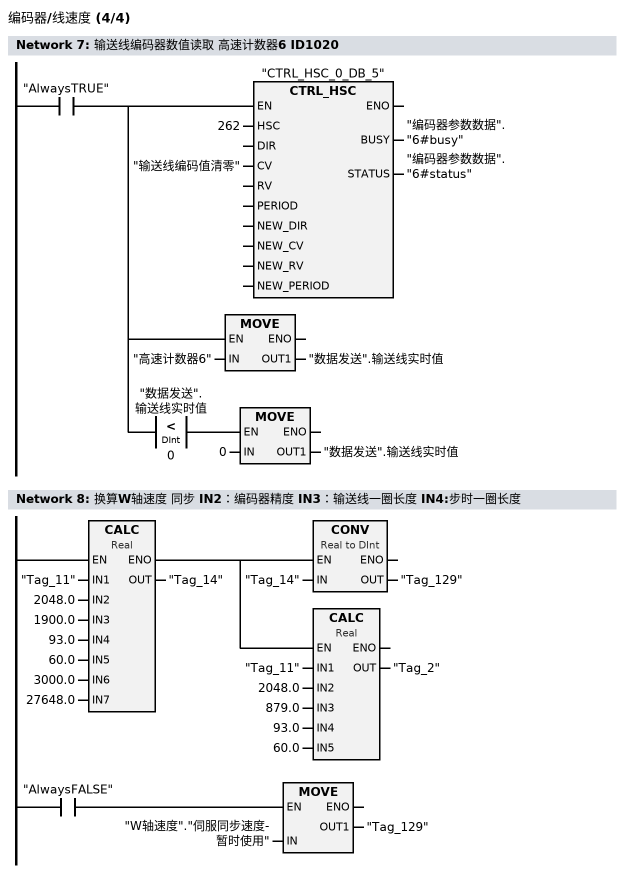
   #_w1 := "AlwaysTRUE";
   IF #_w1 THEN
       "CTRL_HSC_0_DB_5"(HSC := 262, CV := "输送线编码值清零", BUSY => "编码器参数数据"."6#busy", STATUS => "编码器参数数据"."6#status");   // CTRL_HSC
       "数据发送".输送线实时值 := "高速计数器6";
   END_IF;
   IF #_w1 AND ("数据发送".输送线实时值 < 0) THEN "数据发送".输送线实时值 := 0; END_IF;
END_REGION

REGION Network 8: 换算W轴速度 同步 IN2：编码器精度 IN3：输送线一圈长度 IN4:步时一圈长度
   CALC(in1 := "Tag_11",
        in2 := 2048.0,
        in3 := 1900.0,
        in4 := 93.0,
        in5 := 60.0,
        in6 := 3000.0,
        in7 := 27648.0,
        out => "Tag_14");
   "Tag_129" := REAL_TO_DINT("Tag_14");
   CALC(in1 := "Tag_11", in2 := 2048.0, in3 := 879.0, in4 := 93.0, in5 := 60.0, out => "Tag_2");
   IF "AlwaysFALSE" THEN "Tag_129" := "W轴速度"."伺服同步速度-暂时使用"; END_IF;
END_REGION
END_FUNCTION

FUNCTION "2#手" : Void   // FC13, LAD
{ S7_Optimized_Access := 'TRUE' }
VERSION : 0.1
   VAR_TEMP   // added for the SCL form of the ladder/FBD networks
      _w1 : Bool;
   END_VAR
BEGIN

REGION Network 1: 2#机械手库位动作流程
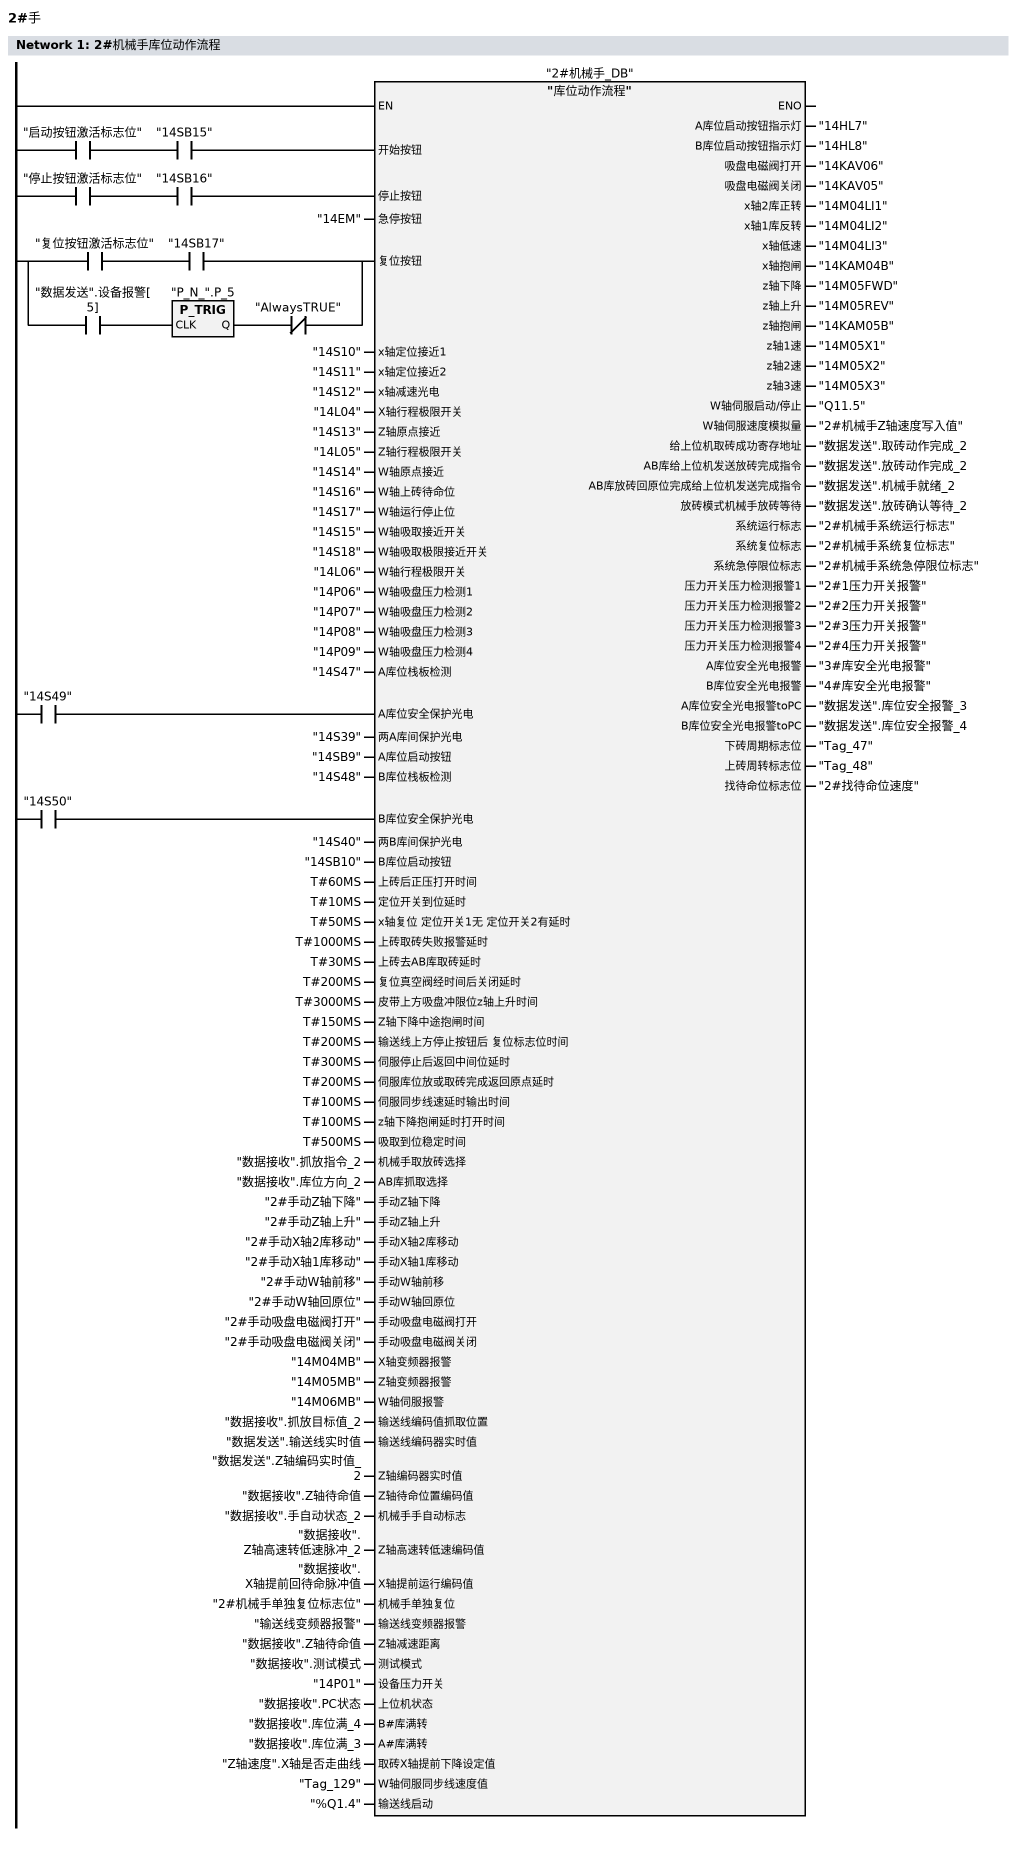
   RUNG wire#powerrail
      "2#机械手_DB"(开始按钮 := wire#w1, 停止按钮 := wire#w2, 复位按钮 := wire#w3, A库位安全保护光电 := wire#w4, B库位安全保护光电 := wire#w5, 急停按钮 := "14EM", x轴定位接近1 := "14S10", x轴定位接近2 := "14S11", x轴减速光电 := "14S12", X轴行程极限开关 := "14L04", Z轴原点接近 := "14S13", Z轴行程极限开关 := "14L05", W轴原点接近 := "14S14", W轴上砖待命位 := "14S16", W轴运行停止位 := "14S17", W轴吸取接近开关 := "14S15", W轴吸取极限接近开关 := "14S18", W轴行程极限开关 := "14L06", W轴吸盘压力检测1 := "14P06", W轴吸盘压力检测2 := "14P07", W轴吸盘压力检测3 := "14P08", W轴吸盘压力检测4 := "14P09", A库位栈板检测 := "14S47", 两A库间保护光电 := "14S39", A库位启动按钮 := "14SB9", B库位栈板检测 := "14S48", 两B库间保护光电 := "14S40", B库位启动按钮 := "14SB10", 上砖后正压打开时间 := T#60MS, 定位开关到位延时 := T#10MS, "x轴复位 定位开关1无 定位开关2有延时" := T#50MS, 上砖取砖失败报警延时 := T#1000MS, 上砖去AB库取砖延时 := T#30MS, 复位真空阀经时间后关闭延时 := T#200MS, 皮带上方吸盘冲限位z轴上升时间 := T#3000MS, Z轴下降中途抱闸时间 := T#150MS, "输送线上方停止按钮后 复位标志位时间" := T#200MS, 伺服停止后返回中间位延时 := T#300MS, 伺服库位放或取砖完成返回原点延时 := T#200MS, 伺服同步线速延时输出时间 := T#100MS, z轴下降抱闸延时打开时间 := T#100MS, 吸取到位稳定时间 := T#500MS, 机械手取放砖选择 := "数据接收".抓放指令_2, AB库抓取选择 := "数据接收".库位方向_2, 手动Z轴下降 := "2#手动Z轴下降", 手动Z轴上升 := "2#手动Z轴上升", 手动X轴2库移动 := "2#手动X轴2库移动", 手动X轴1库移动 := "2#手动X轴1库移动", 手动W轴前移 := "2#手动W轴前移", 手动W轴回原位 := "2#手动W轴回原位", 手动吸盘电磁阀打开 := "2#手动吸盘电磁阀打开", 手动吸盘电磁阀关闭 := "2#手动吸盘电磁阀关闭", X轴变频器报警 := "14M04MB", Z轴变频器报警 := "14M05MB", W轴伺服报警 := "14M06MB", 输送线编码值抓取位置 := "数据接收".抓放目标值_2, 输送线编码器实时值 := "数据发送".输送线实时值, Z轴编码器实时值 := "数据发送".Z轴编码实时值_2, Z轴待命位置编码值 := "数据接收".Z轴待命值, 机械手手自动标志 := "数据接收".手自动状态_2, Z轴高速转低速编码值 := "数据接收".Z轴高速转低速脉冲_2, X轴提前运行编码值 := "数据接收".X轴提前回待命脉冲值, 机械手单独复位 := "2#机械手单独复位标志位", 输送线变频器报警 := "输送线变频器报警", Z轴减速距离 := "数据接收".Z轴待命值, 测试模式 := "数据接收".测试模式, 设备压力开关 := "14P01", 上位机状态 := "数据接收".PC状态, "B#库满转" := "数据接收".库位满_4, "A#库满转" := "数据接收".库位满_3, 取砖X轴提前下降设定值 := "Z轴速度".X轴是否走曲线, W轴伺服同步线速度值 := "Tag_129", 输送线启动 := "%Q1.4", A库位启动按钮指示灯 => "14HL7", B库位启动按钮指示灯 => "14HL8", 吸盘电磁阀打开 => "14KAV06", 吸盘电磁阀关闭 => "14KAV05", x轴2库正转 => "14M04LI1", x轴1库反转 => "14M04LI2", x轴低速 => "14M04LI3", x轴抱闸 => "14KAM04B", z轴下降 => "14M05FWD", z轴上升 => "14M05REV", z轴抱闸 => "14KAM05B", z轴1速 => "14M05X1", z轴2速 => "14M05X2", z轴3速 => "14M05X3", "W轴伺服启动/停止" => "Q11.5", W轴伺服速度模拟量 => "2#机械手Z轴速度写入值", 给上位机取砖成功寄存地址 => "数据发送".取砖动作完成_2, AB库给上位机发送放砖完成指令 => "数据发送".放砖动作完成_2, AB库放砖回原位完成给上位机发送完成指令 => "数据发送".机械手就绪_2, 放砖模式机械手放砖等待 => "数据发送".放砖确认等待_2, 系统运行标志 => "2#机械手系统运行标志", 系统复位标志 => "2#机械手系统复位标志", 系统急停限位标志 => "2#机械手系统急停限位标志", 压力开关压力检测报警1 => "2#1压力开关报警", 压力开关压力检测报警2 => "2#2压力开关报警", 压力开关压力检测报警3 => "2#3压力开关报警", 压力开关压力检测报警4 => "2#4压力开关报警", A库位安全光电报警 => "3#库安全光电报警", B库位安全光电报警 => "4#库安全光电报警", A库位安全光电报警toPC => "数据发送".库位安全报警_3, B库位安全光电报警toPC => "数据发送".库位安全报警_4, 下砖周期标志位 => "Tag_47", 上砖周转标志位 => "Tag_48", 找待命位标志位 => "2#找待命位速度")
   END_RUNG
   RUNG wire#powerrail
      Contact( "启动按钮激活标志位" )
      Contact( "14SB15" )
   END_RUNG wire#w1
   RUNG wire#powerrail
      Contact( "停止按钮激活标志位" )
      Contact( "14SB16" )
   END_RUNG wire#w2
   RUNG wire#powerrail
      Contact( "复位按钮激活标志位" )
      Contact( "14SB17" )
   END_RUNG wire#w3
   RUNG wire#powerrail
      Contact( "数据发送".设备报警[5] )
      P_Trig( "P_N_".P_5 )
      I_Contact( "AlwaysTRUE" )
   END_RUNG wire#w3
   RUNG wire#powerrail
      Contact( "14S49" )
   END_RUNG wire#w4
   RUNG wire#powerrail
      Contact( "14S50" )
   END_RUNG wire#w5
   // the same network as SCL:
   #_w1 := "数据发送".设备报警[5] AND NOT "P_N_".P_5;   // rising edge
   "P_N_".P_5 := "数据发送".设备报警[5];
   "2#机械手_DB"(开始按钮 := "启动按钮激活标志位" AND "14SB15",   // "库位动作流程"
              停止按钮 := "停止按钮激活标志位" AND "14SB16",
              急停按钮 := "14EM",
              复位按钮 := ("复位按钮激活标志位" AND "14SB17") OR (#_w1 AND NOT "AlwaysTRUE"),
              x轴定位接近1 := "14S10",
              x轴定位接近2 := "14S11",
              x轴减速光电 := "14S12",
              X轴行程极限开关 := "14L04",
              Z轴原点接近 := "14S13",
              Z轴行程极限开关 := "14L05",
              W轴原点接近 := "14S14",
              W轴上砖待命位 := "14S16",
              W轴运行停止位 := "14S17",
              W轴吸取接近开关 := "14S15",
              W轴吸取极限接近开关 := "14S18",
              W轴行程极限开关 := "14L06",
              W轴吸盘压力检测1 := "14P06",
              W轴吸盘压力检测2 := "14P07",
              W轴吸盘压力检测3 := "14P08",
              W轴吸盘压力检测4 := "14P09",
              A库位栈板检测 := "14S47",
              A库位安全保护光电 := "14S49",
              两A库间保护光电 := "14S39",
              A库位启动按钮 := "14SB9",
              B库位栈板检测 := "14S48",
              B库位安全保护光电 := "14S50",
              两B库间保护光电 := "14S40",
              B库位启动按钮 := "14SB10",
              上砖后正压打开时间 := T#60MS,
              定位开关到位延时 := T#10MS,
              "x轴复位 定位开关1无 定位开关2有延时" := T#50MS,
              上砖取砖失败报警延时 := T#1000MS,
              上砖去AB库取砖延时 := T#30MS,
              复位真空阀经时间后关闭延时 := T#200MS,
              皮带上方吸盘冲限位z轴上升时间 := T#3000MS,
              Z轴下降中途抱闸时间 := T#150MS,
              "输送线上方停止按钮后 复位标志位时间" := T#200MS,
              伺服停止后返回中间位延时 := T#300MS,
              伺服库位放或取砖完成返回原点延时 := T#200MS,
              伺服同步线速延时输出时间 := T#100MS,
              z轴下降抱闸延时打开时间 := T#100MS,
              吸取到位稳定时间 := T#500MS,
              机械手取放砖选择 := "数据接收".抓放指令_2,
              AB库抓取选择 := "数据接收".库位方向_2,
              手动Z轴下降 := "2#手动Z轴下降",
              手动Z轴上升 := "2#手动Z轴上升",
              手动X轴2库移动 := "2#手动X轴2库移动",
              手动X轴1库移动 := "2#手动X轴1库移动",
              手动W轴前移 := "2#手动W轴前移",
              手动W轴回原位 := "2#手动W轴回原位",
              手动吸盘电磁阀打开 := "2#手动吸盘电磁阀打开",
              手动吸盘电磁阀关闭 := "2#手动吸盘电磁阀关闭",
              X轴变频器报警 := "14M04MB",
              Z轴变频器报警 := "14M05MB",
              W轴伺服报警 := "14M06MB",
              输送线编码值抓取位置 := "数据接收".抓放目标值_2,
              输送线编码器实时值 := "数据发送".输送线实时值,
              Z轴编码器实时值 := "数据发送".Z轴编码实时值_2,
              Z轴待命位置编码值 := "数据接收".Z轴待命值,
              机械手手自动标志 := "数据接收".手自动状态_2,
              Z轴高速转低速编码值 := "数据接收".Z轴高速转低速脉冲_2,
              X轴提前运行编码值 := "数据接收".X轴提前回待命脉冲值,
              机械手单独复位 := "2#机械手单独复位标志位",
              输送线变频器报警 := "输送线变频器报警",
              Z轴减速距离 := "数据接收".Z轴待命值,
              测试模式 := "数据接收".测试模式,
              设备压力开关 := "14P01",
              上位机状态 := "数据接收".PC状态,
              "B#库满转" := "数据接收".库位满_4,
              "A#库满转" := "数据接收".库位满_3,
              取砖X轴提前下降设定值 := "Z轴速度".X轴是否走曲线,
              W轴伺服同步线速度值 := "Tag_129",
              输送线启动 := "%Q1.4",
              A库位启动按钮指示灯 => "14HL7",
              B库位启动按钮指示灯 => "14HL8",
              吸盘电磁阀打开 => "14KAV06",
              吸盘电磁阀关闭 => "14KAV05",
              x轴2库正转 => "14M04LI1",
              x轴1库反转 => "14M04LI2",
              x轴低速 => "14M04LI3",
              x轴抱闸 => "14KAM04B",
              z轴下降 => "14M05FWD",
              z轴上升 => "14M05REV",
              z轴抱闸 => "14KAM05B",
              z轴1速 => "14M05X1",
              z轴2速 => "14M05X2",
              z轴3速 => "14M05X3",
              "W轴伺服启动/停止" => "Q11.5",
              W轴伺服速度模拟量 => "2#机械手Z轴速度写入值",
              给上位机取砖成功寄存地址 => "数据发送".取砖动作完成_2,
              AB库给上位机发送放砖完成指令 => "数据发送".放砖动作完成_2,
              AB库放砖回原位完成给上位机发送完成指令 => "数据发送".机械手就绪_2,
              放砖模式机械手放砖等待 => "数据发送".放砖确认等待_2,
              系统运行标志 => "2#机械手系统运行标志",
              系统复位标志 => "2#机械手系统复位标志",
              系统急停限位标志 => "2#机械手系统急停限位标志",
              压力开关压力检测报警1 => "2#1压力开关报警",
              压力开关压力检测报警2 => "2#2压力开关报警",
              压力开关压力检测报警3 => "2#3压力开关报警",
              压力开关压力检测报警4 => "2#4压力开关报警",
              A库位安全光电报警 => "3#库安全光电报警",
              B库位安全光电报警 => "4#库安全光电报警",
              A库位安全光电报警toPC => "数据发送".库位安全报警_3,
              B库位安全光电报警toPC => "数据发送".库位安全报警_4,
              下砖周期标志位 => "Tag_47",
              上砖周转标志位 => "Tag_48",
              找待命位标志位 => "2#找待命位速度");
END_REGION
END_FUNCTION

FUNCTION "3#手" : Void   // FC14, LAD
{ S7_Optimized_Access := 'TRUE' }
VERSION : 0.1
   VAR_TEMP   // added for the SCL form of the ladder/FBD networks
      _w1 : Bool;
   END_VAR
BEGIN

REGION Network 1: 3#机械手库位动作流程
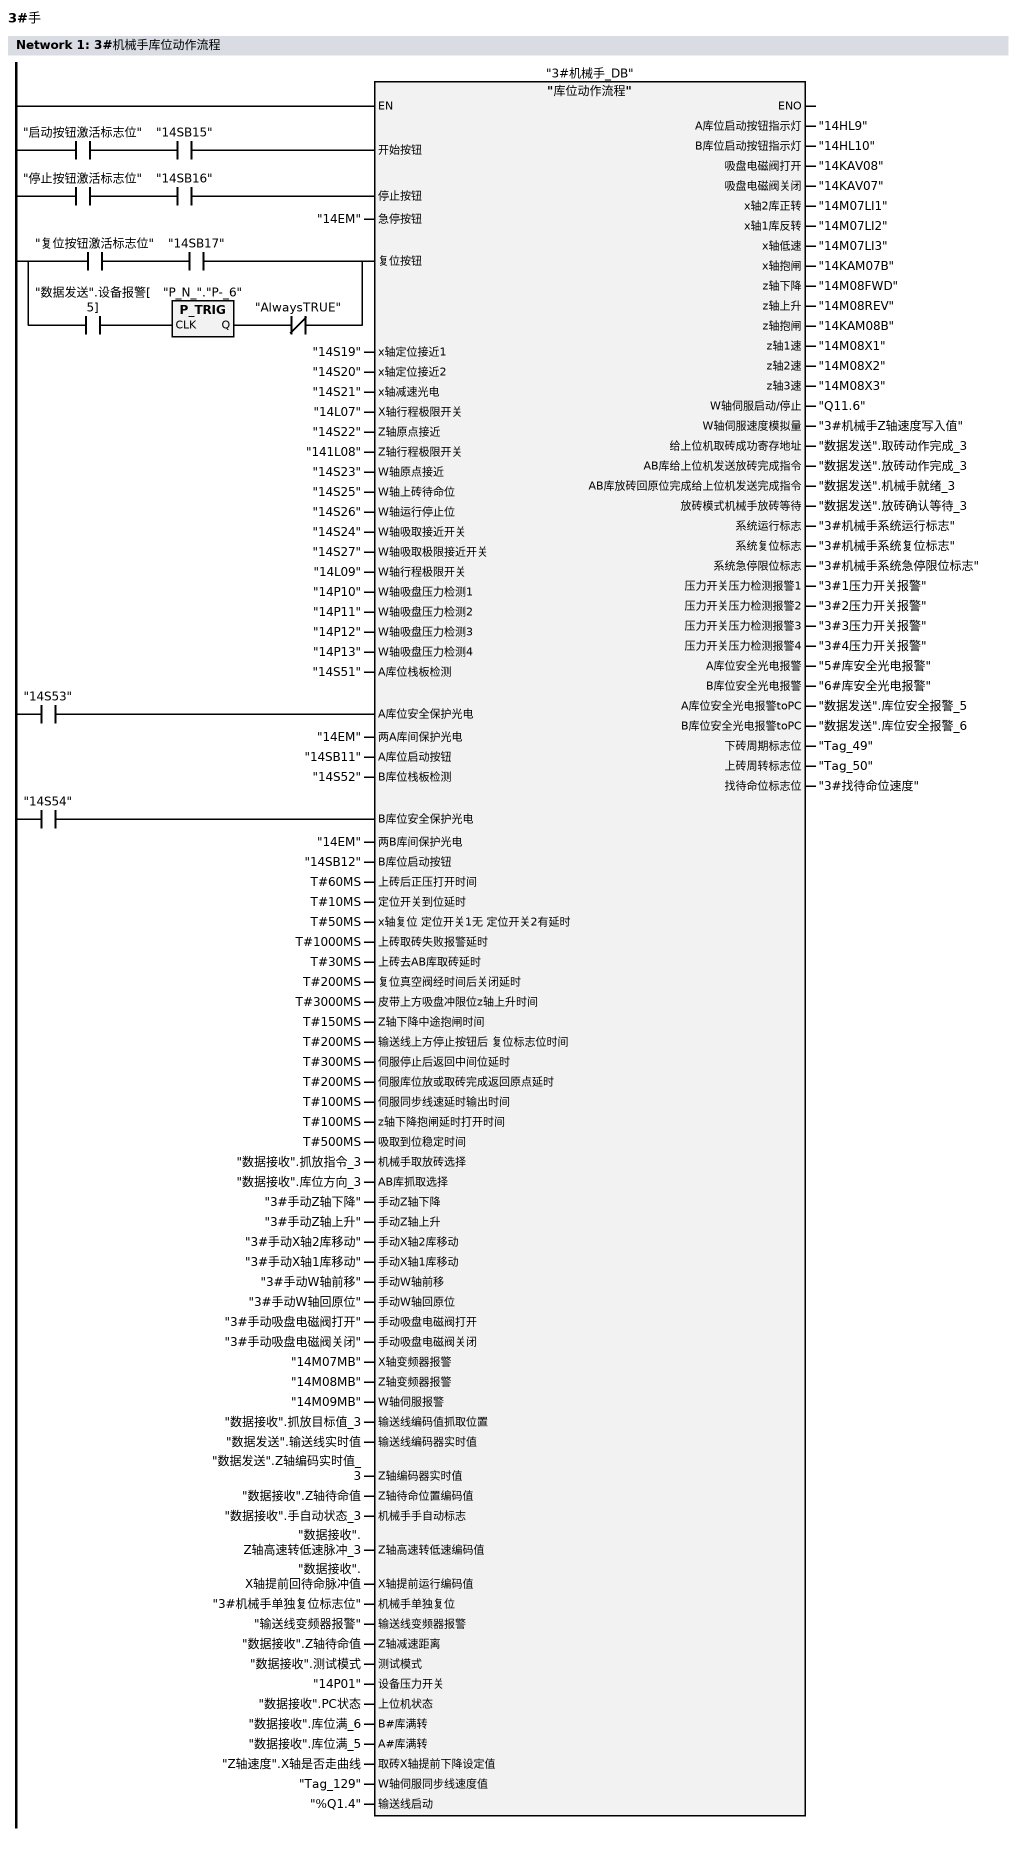
   RUNG wire#powerrail
      "3#机械手_DB"(开始按钮 := wire#w1, 停止按钮 := wire#w2, 复位按钮 := wire#w3, A库位安全保护光电 := wire#w4, B库位安全保护光电 := wire#w5, 急停按钮 := "14EM", x轴定位接近1 := "14S19", x轴定位接近2 := "14S20", x轴减速光电 := "14S21", X轴行程极限开关 := "14L07", Z轴原点接近 := "14S22", Z轴行程极限开关 := "141L08", W轴原点接近 := "14S23", W轴上砖待命位 := "14S25", W轴运行停止位 := "14S26", W轴吸取接近开关 := "14S24", W轴吸取极限接近开关 := "14S27", W轴行程极限开关 := "14L09", W轴吸盘压力检测1 := "14P10", W轴吸盘压力检测2 := "14P11", W轴吸盘压力检测3 := "14P12", W轴吸盘压力检测4 := "14P13", A库位栈板检测 := "14S51", 两A库间保护光电 := "14EM", A库位启动按钮 := "14SB11", B库位栈板检测 := "14S52", 两B库间保护光电 := "14EM", B库位启动按钮 := "14SB12", 上砖后正压打开时间 := T#60MS, 定位开关到位延时 := T#10MS, "x轴复位 定位开关1无 定位开关2有延时" := T#50MS, 上砖取砖失败报警延时 := T#1000MS, 上砖去AB库取砖延时 := T#30MS, 复位真空阀经时间后关闭延时 := T#200MS, 皮带上方吸盘冲限位z轴上升时间 := T#3000MS, Z轴下降中途抱闸时间 := T#150MS, "输送线上方停止按钮后 复位标志位时间" := T#200MS, 伺服停止后返回中间位延时 := T#300MS, 伺服库位放或取砖完成返回原点延时 := T#200MS, 伺服同步线速延时输出时间 := T#100MS, z轴下降抱闸延时打开时间 := T#100MS, 吸取到位稳定时间 := T#500MS, 机械手取放砖选择 := "数据接收".抓放指令_3, AB库抓取选择 := "数据接收".库位方向_3, 手动Z轴下降 := "3#手动Z轴下降", 手动Z轴上升 := "3#手动Z轴上升", 手动X轴2库移动 := "3#手动X轴2库移动", 手动X轴1库移动 := "3#手动X轴1库移动", 手动W轴前移 := "3#手动W轴前移", 手动W轴回原位 := "3#手动W轴回原位", 手动吸盘电磁阀打开 := "3#手动吸盘电磁阀打开", 手动吸盘电磁阀关闭 := "3#手动吸盘电磁阀关闭", X轴变频器报警 := "14M07MB", Z轴变频器报警 := "14M08MB", W轴伺服报警 := "14M09MB", 输送线编码值抓取位置 := "数据接收".抓放目标值_3, 输送线编码器实时值 := "数据发送".输送线实时值, Z轴编码器实时值 := "数据发送".Z轴编码实时值_3, Z轴待命位置编码值 := "数据接收".Z轴待命值, 机械手手自动标志 := "数据接收".手自动状态_3, Z轴高速转低速编码值 := "数据接收".Z轴高速转低速脉冲_3, X轴提前运行编码值 := "数据接收".X轴提前回待命脉冲值, 机械手单独复位 := "3#机械手单独复位标志位", 输送线变频器报警 := "输送线变频器报警", Z轴减速距离 := "数据接收".Z轴待命值, 测试模式 := "数据接收".测试模式, 设备压力开关 := "14P01", 上位机状态 := "数据接收".PC状态, "B#库满转" := "数据接收".库位满_6, "A#库满转" := "数据接收".库位满_5, 取砖X轴提前下降设定值 := "Z轴速度".X轴是否走曲线, W轴伺服同步线速度值 := "Tag_129", 输送线启动 := "%Q1.4", A库位启动按钮指示灯 => "14HL9", B库位启动按钮指示灯 => "14HL10", 吸盘电磁阀打开 => "14KAV08", 吸盘电磁阀关闭 => "14KAV07", x轴2库正转 => "14M07LI1", x轴1库反转 => "14M07LI2", x轴低速 => "14M07LI3", x轴抱闸 => "14KAM07B", z轴下降 => "14M08FWD", z轴上升 => "14M08REV", z轴抱闸 => "14KAM08B", z轴1速 => "14M08X1", z轴2速 => "14M08X2", z轴3速 => "14M08X3", "W轴伺服启动/停止" => "Q11.6", W轴伺服速度模拟量 => "3#机械手Z轴速度写入值", 给上位机取砖成功寄存地址 => "数据发送".取砖动作完成_3, AB库给上位机发送放砖完成指令 => "数据发送".放砖动作完成_3, AB库放砖回原位完成给上位机发送完成指令 => "数据发送".机械手就绪_3, 放砖模式机械手放砖等待 => "数据发送".放砖确认等待_3, 系统运行标志 => "3#机械手系统运行标志", 系统复位标志 => "3#机械手系统复位标志", 系统急停限位标志 => "3#机械手系统急停限位标志", 压力开关压力检测报警1 => "3#1压力开关报警", 压力开关压力检测报警2 => "3#2压力开关报警", 压力开关压力检测报警3 => "3#3压力开关报警", 压力开关压力检测报警4 => "3#4压力开关报警", A库位安全光电报警 => "5#库安全光电报警", B库位安全光电报警 => "6#库安全光电报警", A库位安全光电报警toPC => "数据发送".库位安全报警_5, B库位安全光电报警toPC => "数据发送".库位安全报警_6, 下砖周期标志位 => "Tag_49", 上砖周转标志位 => "Tag_50", 找待命位标志位 => "3#找待命位速度")
   END_RUNG
   RUNG wire#powerrail
      Contact( "启动按钮激活标志位" )
      Contact( "14SB15" )
   END_RUNG wire#w1
   RUNG wire#powerrail
      Contact( "停止按钮激活标志位" )
      Contact( "14SB16" )
   END_RUNG wire#w2
   RUNG wire#powerrail
      Contact( "复位按钮激活标志位" )
      Contact( "14SB17" )
   END_RUNG wire#w3
   RUNG wire#powerrail
      Contact( "数据发送".设备报警[5] )
      P_Trig( "P_N_"."P-_6" )
      I_Contact( "AlwaysTRUE" )
   END_RUNG wire#w3
   RUNG wire#powerrail
      Contact( "14S53" )
   END_RUNG wire#w4
   RUNG wire#powerrail
      Contact( "14S54" )
   END_RUNG wire#w5
   // the same network as SCL:
   #_w1 := "数据发送".设备报警[5] AND NOT "P_N_"."P-_6";   // rising edge
   "P_N_"."P-_6" := "数据发送".设备报警[5];
   "3#机械手_DB"(开始按钮 := "启动按钮激活标志位" AND "14SB15",   // "库位动作流程"
              停止按钮 := "停止按钮激活标志位" AND "14SB16",
              急停按钮 := "14EM",
              复位按钮 := ("复位按钮激活标志位" AND "14SB17") OR (#_w1 AND NOT "AlwaysTRUE"),
              x轴定位接近1 := "14S19",
              x轴定位接近2 := "14S20",
              x轴减速光电 := "14S21",
              X轴行程极限开关 := "14L07",
              Z轴原点接近 := "14S22",
              Z轴行程极限开关 := "141L08",
              W轴原点接近 := "14S23",
              W轴上砖待命位 := "14S25",
              W轴运行停止位 := "14S26",
              W轴吸取接近开关 := "14S24",
              W轴吸取极限接近开关 := "14S27",
              W轴行程极限开关 := "14L09",
              W轴吸盘压力检测1 := "14P10",
              W轴吸盘压力检测2 := "14P11",
              W轴吸盘压力检测3 := "14P12",
              W轴吸盘压力检测4 := "14P13",
              A库位栈板检测 := "14S51",
              A库位安全保护光电 := "14S53",
              两A库间保护光电 := "14EM",
              A库位启动按钮 := "14SB11",
              B库位栈板检测 := "14S52",
              B库位安全保护光电 := "14S54",
              两B库间保护光电 := "14EM",
              B库位启动按钮 := "14SB12",
              上砖后正压打开时间 := T#60MS,
              定位开关到位延时 := T#10MS,
              "x轴复位 定位开关1无 定位开关2有延时" := T#50MS,
              上砖取砖失败报警延时 := T#1000MS,
              上砖去AB库取砖延时 := T#30MS,
              复位真空阀经时间后关闭延时 := T#200MS,
              皮带上方吸盘冲限位z轴上升时间 := T#3000MS,
              Z轴下降中途抱闸时间 := T#150MS,
              "输送线上方停止按钮后 复位标志位时间" := T#200MS,
              伺服停止后返回中间位延时 := T#300MS,
              伺服库位放或取砖完成返回原点延时 := T#200MS,
              伺服同步线速延时输出时间 := T#100MS,
              z轴下降抱闸延时打开时间 := T#100MS,
              吸取到位稳定时间 := T#500MS,
              机械手取放砖选择 := "数据接收".抓放指令_3,
              AB库抓取选择 := "数据接收".库位方向_3,
              手动Z轴下降 := "3#手动Z轴下降",
              手动Z轴上升 := "3#手动Z轴上升",
              手动X轴2库移动 := "3#手动X轴2库移动",
              手动X轴1库移动 := "3#手动X轴1库移动",
              手动W轴前移 := "3#手动W轴前移",
              手动W轴回原位 := "3#手动W轴回原位",
              手动吸盘电磁阀打开 := "3#手动吸盘电磁阀打开",
              手动吸盘电磁阀关闭 := "3#手动吸盘电磁阀关闭",
              X轴变频器报警 := "14M07MB",
              Z轴变频器报警 := "14M08MB",
              W轴伺服报警 := "14M09MB",
              输送线编码值抓取位置 := "数据接收".抓放目标值_3,
              输送线编码器实时值 := "数据发送".输送线实时值,
              Z轴编码器实时值 := "数据发送".Z轴编码实时值_3,
              Z轴待命位置编码值 := "数据接收".Z轴待命值,
              机械手手自动标志 := "数据接收".手自动状态_3,
              Z轴高速转低速编码值 := "数据接收".Z轴高速转低速脉冲_3,
              X轴提前运行编码值 := "数据接收".X轴提前回待命脉冲值,
              机械手单独复位 := "3#机械手单独复位标志位",
              输送线变频器报警 := "输送线变频器报警",
              Z轴减速距离 := "数据接收".Z轴待命值,
              测试模式 := "数据接收".测试模式,
              设备压力开关 := "14P01",
              上位机状态 := "数据接收".PC状态,
              "B#库满转" := "数据接收".库位满_6,
              "A#库满转" := "数据接收".库位满_5,
              取砖X轴提前下降设定值 := "Z轴速度".X轴是否走曲线,
              W轴伺服同步线速度值 := "Tag_129",
              输送线启动 := "%Q1.4",
              A库位启动按钮指示灯 => "14HL9",
              B库位启动按钮指示灯 => "14HL10",
              吸盘电磁阀打开 => "14KAV08",
              吸盘电磁阀关闭 => "14KAV07",
              x轴2库正转 => "14M07LI1",
              x轴1库反转 => "14M07LI2",
              x轴低速 => "14M07LI3",
              x轴抱闸 => "14KAM07B",
              z轴下降 => "14M08FWD",
              z轴上升 => "14M08REV",
              z轴抱闸 => "14KAM08B",
              z轴1速 => "14M08X1",
              z轴2速 => "14M08X2",
              z轴3速 => "14M08X3",
              "W轴伺服启动/停止" => "Q11.6",
              W轴伺服速度模拟量 => "3#机械手Z轴速度写入值",
              给上位机取砖成功寄存地址 => "数据发送".取砖动作完成_3,
              AB库给上位机发送放砖完成指令 => "数据发送".放砖动作完成_3,
              AB库放砖回原位完成给上位机发送完成指令 => "数据发送".机械手就绪_3,
              放砖模式机械手放砖等待 => "数据发送".放砖确认等待_3,
              系统运行标志 => "3#机械手系统运行标志",
              系统复位标志 => "3#机械手系统复位标志",
              系统急停限位标志 => "3#机械手系统急停限位标志",
              压力开关压力检测报警1 => "3#1压力开关报警",
              压力开关压力检测报警2 => "3#2压力开关报警",
              压力开关压力检测报警3 => "3#3压力开关报警",
              压力开关压力检测报警4 => "3#4压力开关报警",
              A库位安全光电报警 => "5#库安全光电报警",
              B库位安全光电报警 => "6#库安全光电报警",
              A库位安全光电报警toPC => "数据发送".库位安全报警_5,
              B库位安全光电报警toPC => "数据发送".库位安全报警_6,
              下砖周期标志位 => "Tag_49",
              上砖周转标志位 => "Tag_50",
              找待命位标志位 => "3#找待命位速度");
END_REGION
END_FUNCTION

FUNCTION "4#手" : Void   // FC15, LAD
{ S7_Optimized_Access := 'TRUE' }
VERSION : 0.1
   VAR_TEMP   // added for the SCL form of the ladder/FBD networks
      _w1 : Bool;
   END_VAR
BEGIN

REGION Network 1: 4#机械手库位动作流程
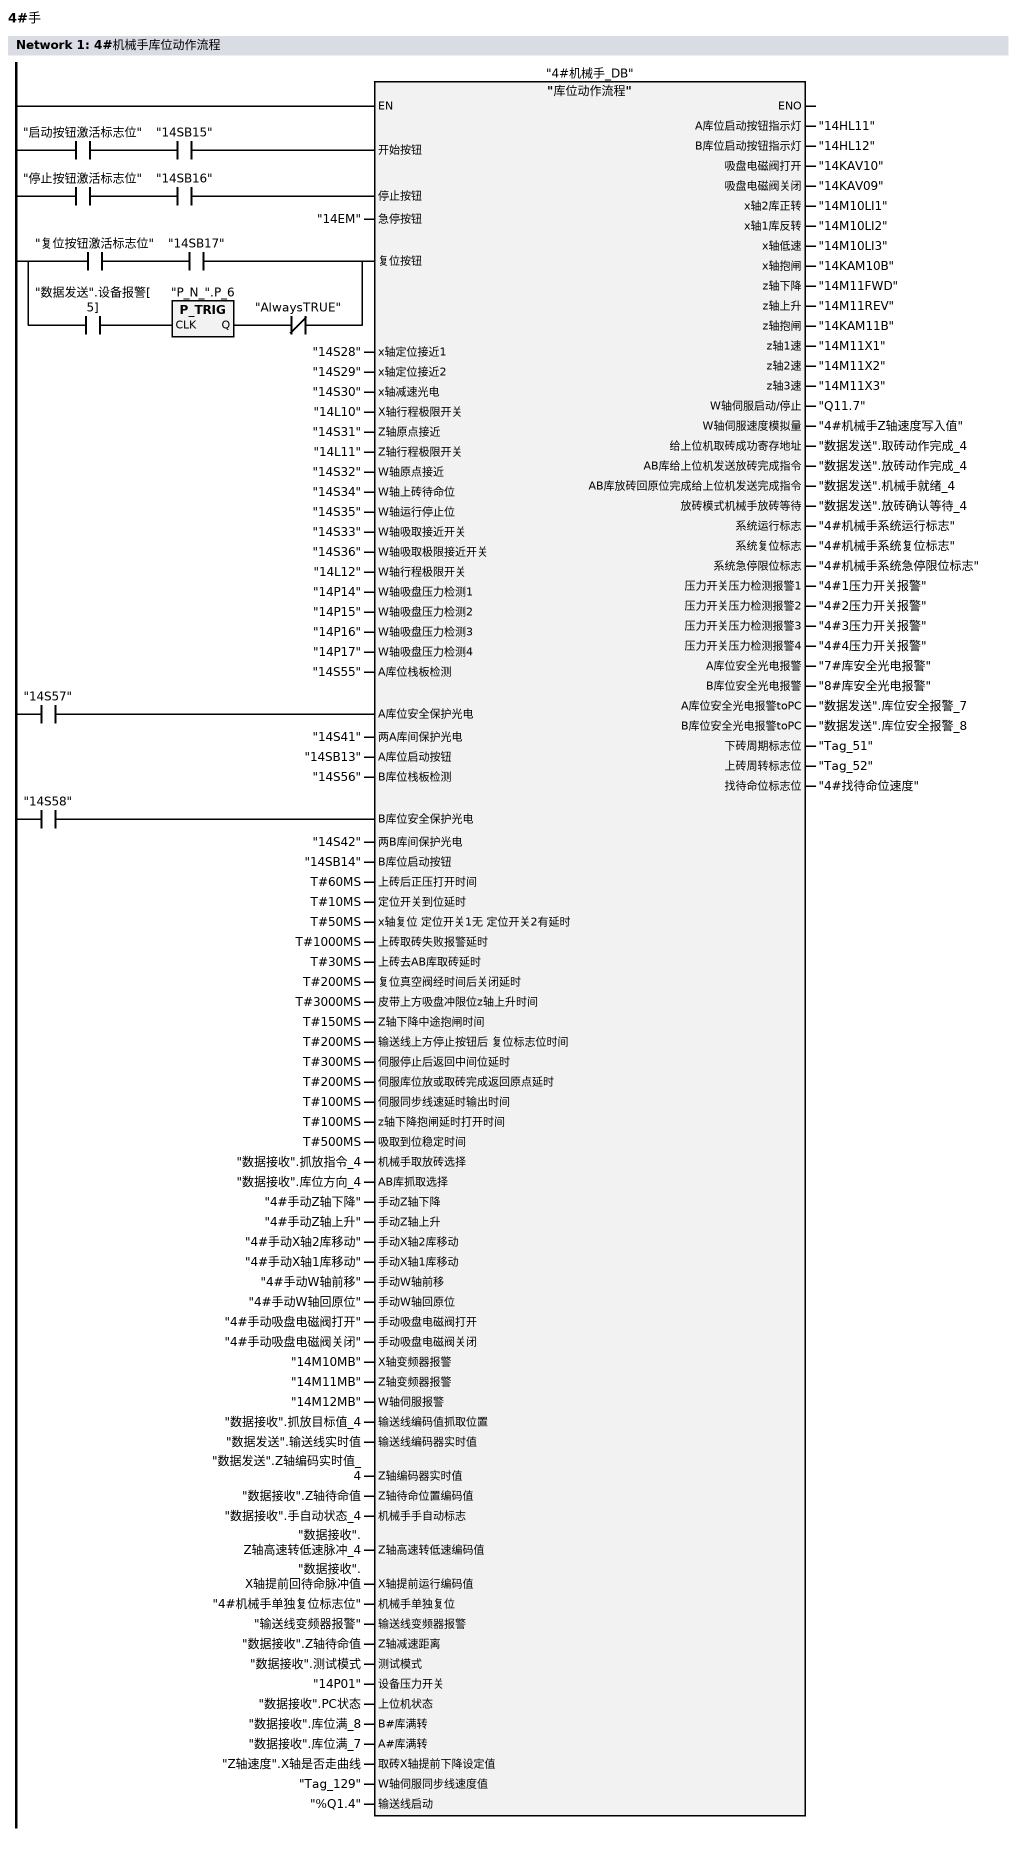
   RUNG wire#powerrail
      "4#机械手_DB"(开始按钮 := wire#w1, 停止按钮 := wire#w2, 复位按钮 := wire#w3, A库位安全保护光电 := wire#w4, B库位安全保护光电 := wire#w5, 急停按钮 := "14EM", x轴定位接近1 := "14S28", x轴定位接近2 := "14S29", x轴减速光电 := "14S30", X轴行程极限开关 := "14L10", Z轴原点接近 := "14S31", Z轴行程极限开关 := "14L11", W轴原点接近 := "14S32", W轴上砖待命位 := "14S34", W轴运行停止位 := "14S35", W轴吸取接近开关 := "14S33", W轴吸取极限接近开关 := "14S36", W轴行程极限开关 := "14L12", W轴吸盘压力检测1 := "14P14", W轴吸盘压力检测2 := "14P15", W轴吸盘压力检测3 := "14P16", W轴吸盘压力检测4 := "14P17", A库位栈板检测 := "14S55", 两A库间保护光电 := "14S41", A库位启动按钮 := "14SB13", B库位栈板检测 := "14S56", 两B库间保护光电 := "14S42", B库位启动按钮 := "14SB14", 上砖后正压打开时间 := T#60MS, 定位开关到位延时 := T#10MS, "x轴复位 定位开关1无 定位开关2有延时" := T#50MS, 上砖取砖失败报警延时 := T#1000MS, 上砖去AB库取砖延时 := T#30MS, 复位真空阀经时间后关闭延时 := T#200MS, 皮带上方吸盘冲限位z轴上升时间 := T#3000MS, Z轴下降中途抱闸时间 := T#150MS, "输送线上方停止按钮后 复位标志位时间" := T#200MS, 伺服停止后返回中间位延时 := T#300MS, 伺服库位放或取砖完成返回原点延时 := T#200MS, 伺服同步线速延时输出时间 := T#100MS, z轴下降抱闸延时打开时间 := T#100MS, 吸取到位稳定时间 := T#500MS, 机械手取放砖选择 := "数据接收".抓放指令_4, AB库抓取选择 := "数据接收".库位方向_4, 手动Z轴下降 := "4#手动Z轴下降", 手动Z轴上升 := "4#手动Z轴上升", 手动X轴2库移动 := "4#手动X轴2库移动", 手动X轴1库移动 := "4#手动X轴1库移动", 手动W轴前移 := "4#手动W轴前移", 手动W轴回原位 := "4#手动W轴回原位", 手动吸盘电磁阀打开 := "4#手动吸盘电磁阀打开", 手动吸盘电磁阀关闭 := "4#手动吸盘电磁阀关闭", X轴变频器报警 := "14M10MB", Z轴变频器报警 := "14M11MB", W轴伺服报警 := "14M12MB", 输送线编码值抓取位置 := "数据接收".抓放目标值_4, 输送线编码器实时值 := "数据发送".输送线实时值, Z轴编码器实时值 := "数据发送".Z轴编码实时值_4, Z轴待命位置编码值 := "数据接收".Z轴待命值, 机械手手自动标志 := "数据接收".手自动状态_4, Z轴高速转低速编码值 := "数据接收".Z轴高速转低速脉冲_4, X轴提前运行编码值 := "数据接收".X轴提前回待命脉冲值, 机械手单独复位 := "4#机械手单独复位标志位", 输送线变频器报警 := "输送线变频器报警", Z轴减速距离 := "数据接收".Z轴待命值, 测试模式 := "数据接收".测试模式, 设备压力开关 := "14P01", 上位机状态 := "数据接收".PC状态, "B#库满转" := "数据接收".库位满_8, "A#库满转" := "数据接收".库位满_7, 取砖X轴提前下降设定值 := "Z轴速度".X轴是否走曲线, W轴伺服同步线速度值 := "Tag_129", 输送线启动 := "%Q1.4", A库位启动按钮指示灯 => "14HL11", B库位启动按钮指示灯 => "14HL12", 吸盘电磁阀打开 => "14KAV10", 吸盘电磁阀关闭 => "14KAV09", x轴2库正转 => "14M10LI1", x轴1库反转 => "14M10LI2", x轴低速 => "14M10LI3", x轴抱闸 => "14KAM10B", z轴下降 => "14M11FWD", z轴上升 => "14M11REV", z轴抱闸 => "14KAM11B", z轴1速 => "14M11X1", z轴2速 => "14M11X2", z轴3速 => "14M11X3", "W轴伺服启动/停止" => "Q11.7", W轴伺服速度模拟量 => "4#机械手Z轴速度写入值", 给上位机取砖成功寄存地址 => "数据发送".取砖动作完成_4, AB库给上位机发送放砖完成指令 => "数据发送".放砖动作完成_4, AB库放砖回原位完成给上位机发送完成指令 => "数据发送".机械手就绪_4, 放砖模式机械手放砖等待 => "数据发送".放砖确认等待_4, 系统运行标志 => "4#机械手系统运行标志", 系统复位标志 => "4#机械手系统复位标志", 系统急停限位标志 => "4#机械手系统急停限位标志", 压力开关压力检测报警1 => "4#1压力开关报警", 压力开关压力检测报警2 => "4#2压力开关报警", 压力开关压力检测报警3 => "4#3压力开关报警", 压力开关压力检测报警4 => "4#4压力开关报警", A库位安全光电报警 => "7#库安全光电报警", B库位安全光电报警 => "8#库安全光电报警", A库位安全光电报警toPC => "数据发送".库位安全报警_7, B库位安全光电报警toPC => "数据发送".库位安全报警_8, 下砖周期标志位 => "Tag_51", 上砖周转标志位 => "Tag_52", 找待命位标志位 => "4#找待命位速度")
   END_RUNG
   RUNG wire#powerrail
      Contact( "启动按钮激活标志位" )
      Contact( "14SB15" )
   END_RUNG wire#w1
   RUNG wire#powerrail
      Contact( "停止按钮激活标志位" )
      Contact( "14SB16" )
   END_RUNG wire#w2
   RUNG wire#powerrail
      Contact( "复位按钮激活标志位" )
      Contact( "14SB17" )
   END_RUNG wire#w3
   RUNG wire#powerrail
      Contact( "数据发送".设备报警[5] )
      P_Trig( "P_N_".P_6 )
      I_Contact( "AlwaysTRUE" )
   END_RUNG wire#w3
   RUNG wire#powerrail
      Contact( "14S57" )
   END_RUNG wire#w4
   RUNG wire#powerrail
      Contact( "14S58" )
   END_RUNG wire#w5
   // the same network as SCL:
   #_w1 := "数据发送".设备报警[5] AND NOT "P_N_".P_6;   // rising edge
   "P_N_".P_6 := "数据发送".设备报警[5];
   "4#机械手_DB"(开始按钮 := "启动按钮激活标志位" AND "14SB15",   // "库位动作流程"
              停止按钮 := "停止按钮激活标志位" AND "14SB16",
              急停按钮 := "14EM",
              复位按钮 := ("复位按钮激活标志位" AND "14SB17") OR (#_w1 AND NOT "AlwaysTRUE"),
              x轴定位接近1 := "14S28",
              x轴定位接近2 := "14S29",
              x轴减速光电 := "14S30",
              X轴行程极限开关 := "14L10",
              Z轴原点接近 := "14S31",
              Z轴行程极限开关 := "14L11",
              W轴原点接近 := "14S32",
              W轴上砖待命位 := "14S34",
              W轴运行停止位 := "14S35",
              W轴吸取接近开关 := "14S33",
              W轴吸取极限接近开关 := "14S36",
              W轴行程极限开关 := "14L12",
              W轴吸盘压力检测1 := "14P14",
              W轴吸盘压力检测2 := "14P15",
              W轴吸盘压力检测3 := "14P16",
              W轴吸盘压力检测4 := "14P17",
              A库位栈板检测 := "14S55",
              A库位安全保护光电 := "14S57",
              两A库间保护光电 := "14S41",
              A库位启动按钮 := "14SB13",
              B库位栈板检测 := "14S56",
              B库位安全保护光电 := "14S58",
              两B库间保护光电 := "14S42",
              B库位启动按钮 := "14SB14",
              上砖后正压打开时间 := T#60MS,
              定位开关到位延时 := T#10MS,
              "x轴复位 定位开关1无 定位开关2有延时" := T#50MS,
              上砖取砖失败报警延时 := T#1000MS,
              上砖去AB库取砖延时 := T#30MS,
              复位真空阀经时间后关闭延时 := T#200MS,
              皮带上方吸盘冲限位z轴上升时间 := T#3000MS,
              Z轴下降中途抱闸时间 := T#150MS,
              "输送线上方停止按钮后 复位标志位时间" := T#200MS,
              伺服停止后返回中间位延时 := T#300MS,
              伺服库位放或取砖完成返回原点延时 := T#200MS,
              伺服同步线速延时输出时间 := T#100MS,
              z轴下降抱闸延时打开时间 := T#100MS,
              吸取到位稳定时间 := T#500MS,
              机械手取放砖选择 := "数据接收".抓放指令_4,
              AB库抓取选择 := "数据接收".库位方向_4,
              手动Z轴下降 := "4#手动Z轴下降",
              手动Z轴上升 := "4#手动Z轴上升",
              手动X轴2库移动 := "4#手动X轴2库移动",
              手动X轴1库移动 := "4#手动X轴1库移动",
              手动W轴前移 := "4#手动W轴前移",
              手动W轴回原位 := "4#手动W轴回原位",
              手动吸盘电磁阀打开 := "4#手动吸盘电磁阀打开",
              手动吸盘电磁阀关闭 := "4#手动吸盘电磁阀关闭",
              X轴变频器报警 := "14M10MB",
              Z轴变频器报警 := "14M11MB",
              W轴伺服报警 := "14M12MB",
              输送线编码值抓取位置 := "数据接收".抓放目标值_4,
              输送线编码器实时值 := "数据发送".输送线实时值,
              Z轴编码器实时值 := "数据发送".Z轴编码实时值_4,
              Z轴待命位置编码值 := "数据接收".Z轴待命值,
              机械手手自动标志 := "数据接收".手自动状态_4,
              Z轴高速转低速编码值 := "数据接收".Z轴高速转低速脉冲_4,
              X轴提前运行编码值 := "数据接收".X轴提前回待命脉冲值,
              机械手单独复位 := "4#机械手单独复位标志位",
              输送线变频器报警 := "输送线变频器报警",
              Z轴减速距离 := "数据接收".Z轴待命值,
              测试模式 := "数据接收".测试模式,
              设备压力开关 := "14P01",
              上位机状态 := "数据接收".PC状态,
              "B#库满转" := "数据接收".库位满_8,
              "A#库满转" := "数据接收".库位满_7,
              取砖X轴提前下降设定值 := "Z轴速度".X轴是否走曲线,
              W轴伺服同步线速度值 := "Tag_129",
              输送线启动 := "%Q1.4",
              A库位启动按钮指示灯 => "14HL11",
              B库位启动按钮指示灯 => "14HL12",
              吸盘电磁阀打开 => "14KAV10",
              吸盘电磁阀关闭 => "14KAV09",
              x轴2库正转 => "14M10LI1",
              x轴1库反转 => "14M10LI2",
              x轴低速 => "14M10LI3",
              x轴抱闸 => "14KAM10B",
              z轴下降 => "14M11FWD",
              z轴上升 => "14M11REV",
              z轴抱闸 => "14KAM11B",
              z轴1速 => "14M11X1",
              z轴2速 => "14M11X2",
              z轴3速 => "14M11X3",
              "W轴伺服启动/停止" => "Q11.7",
              W轴伺服速度模拟量 => "4#机械手Z轴速度写入值",
              给上位机取砖成功寄存地址 => "数据发送".取砖动作完成_4,
              AB库给上位机发送放砖完成指令 => "数据发送".放砖动作完成_4,
              AB库放砖回原位完成给上位机发送完成指令 => "数据发送".机械手就绪_4,
              放砖模式机械手放砖等待 => "数据发送".放砖确认等待_4,
              系统运行标志 => "4#机械手系统运行标志",
              系统复位标志 => "4#机械手系统复位标志",
              系统急停限位标志 => "4#机械手系统急停限位标志",
              压力开关压力检测报警1 => "4#1压力开关报警",
              压力开关压力检测报警2 => "4#2压力开关报警",
              压力开关压力检测报警3 => "4#3压力开关报警",
              压力开关压力检测报警4 => "4#4压力开关报警",
              A库位安全光电报警 => "7#库安全光电报警",
              B库位安全光电报警 => "8#库安全光电报警",
              A库位安全光电报警toPC => "数据发送".库位安全报警_7,
              B库位安全光电报警toPC => "数据发送".库位安全报警_8,
              下砖周期标志位 => "Tag_51",
              上砖周转标志位 => "Tag_52",
              找待命位标志位 => "4#找待命位速度");
END_REGION
END_FUNCTION

FUNCTION "手动位转换" : Void   // FC17, LAD
TITLE = M位 10-20位手动
{ S7_Optimized_Access := 'TRUE' }
VERSION : 0.1
   VAR_TEMP   // added for the SCL form of the ladder/FBD networks
      _w1 : Bool;
   END_VAR
BEGIN

REGION Network 1: 1#机械手 手动
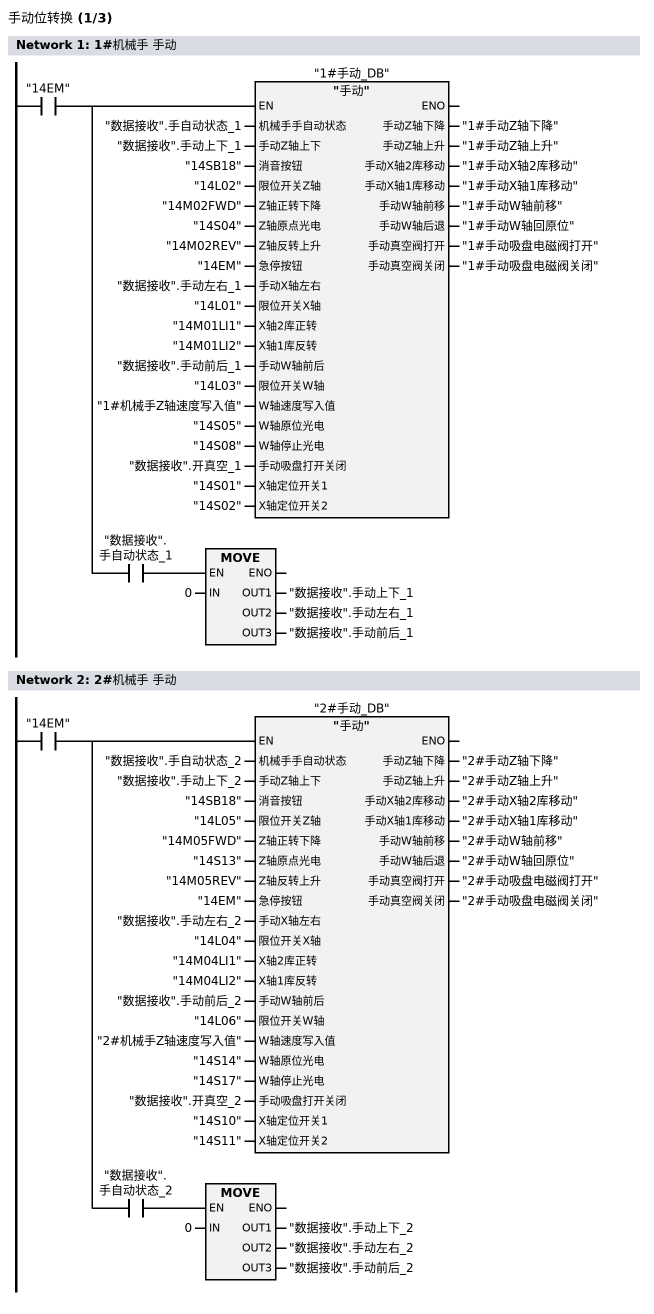
   RUNG wire#powerrail
      Contact( "14EM" )
      wire#w1
      "1#手动_DB"(机械手手自动状态 := "数据接收".手自动状态_1, 手动Z轴上下 := "数据接收".手动上下_1, 消音按钮 := "14SB18", 限位开关Z轴 := "14L02", Z轴正转下降 := "14M02FWD", Z轴原点光电 := "14S04", Z轴反转上升 := "14M02REV", 急停按钮 := "14EM", 手动X轴左右 := "数据接收".手动左右_1, 限位开关X轴 := "14L01", X轴2库正转 := "14M01LI1", X轴1库反转 := "14M01LI2", 手动W轴前后 := "数据接收".手动前后_1, 限位开关W轴 := "14L03", W轴速度写入值 := "1#机械手Z轴速度写入值", W轴原位光电 := "14S05", W轴停止光电 := "14S08", 手动吸盘打开关闭 := "数据接收".开真空_1, X轴定位开关1 := "14S01", X轴定位开关2 := "14S02", 手动Z轴下降 => "1#手动Z轴下降", 手动Z轴上升 => "1#手动Z轴上升", 手动X轴2库移动 => "1#手动X轴2库移动", 手动X轴1库移动 => "1#手动X轴1库移动", 手动W轴前移 => "1#手动W轴前移", 手动W轴后退 => "1#手动W轴回原位", 手动真空阀打开 => "1#手动吸盘电磁阀打开", 手动真空阀关闭 => "1#手动吸盘电磁阀关闭")
   END_RUNG
   RUNG wire#w1
      Contact( "数据接收".手自动状态_1 )
      Move(in := 0, out1 => "数据接收".手动上下_1, out2 => "数据接收".手动左右_1, out3 => "数据接收".手动前后_1)
   END_RUNG
   // the same network as SCL:
   #_w1 := "14EM";
   IF #_w1 THEN
       "1#手动_DB"(机械手手自动状态 := "数据接收".手自动状态_1,   // "手动"
                 手动Z轴上下 := "数据接收".手动上下_1,
                 消音按钮 := "14SB18",
                 限位开关Z轴 := "14L02",
                 Z轴正转下降 := "14M02FWD",
                 Z轴原点光电 := "14S04",
                 Z轴反转上升 := "14M02REV",
                 急停按钮 := "14EM",
                 手动X轴左右 := "数据接收".手动左右_1,
                 限位开关X轴 := "14L01",
                 X轴2库正转 := "14M01LI1",
                 X轴1库反转 := "14M01LI2",
                 手动W轴前后 := "数据接收".手动前后_1,
                 限位开关W轴 := "14L03",
                 W轴速度写入值 := "1#机械手Z轴速度写入值",
                 W轴原位光电 := "14S05",
                 W轴停止光电 := "14S08",
                 手动吸盘打开关闭 := "数据接收".开真空_1,
                 X轴定位开关1 := "14S01",
                 X轴定位开关2 := "14S02",
                 手动Z轴下降 => "1#手动Z轴下降",
                 手动Z轴上升 => "1#手动Z轴上升",
                 手动X轴2库移动 => "1#手动X轴2库移动",
                 手动X轴1库移动 => "1#手动X轴1库移动",
                 手动W轴前移 => "1#手动W轴前移",
                 手动W轴后退 => "1#手动W轴回原位",
                 手动真空阀打开 => "1#手动吸盘电磁阀打开",
                 手动真空阀关闭 => "1#手动吸盘电磁阀关闭");
   END_IF;
   IF #_w1 AND "数据接收".手自动状态_1 THEN
       "数据接收".手动上下_1 := 0;
       "数据接收".手动左右_1 := 0;
       "数据接收".手动前后_1 := 0;
   END_IF;
END_REGION

REGION Network 2: 2#机械手 手动
   RUNG wire#powerrail
      Contact( "14EM" )
      wire#w1
      "2#手动_DB"(机械手手自动状态 := "数据接收".手自动状态_2, 手动Z轴上下 := "数据接收".手动上下_2, 消音按钮 := "14SB18", 限位开关Z轴 := "14L05", Z轴正转下降 := "14M05FWD", Z轴原点光电 := "14S13", Z轴反转上升 := "14M05REV", 急停按钮 := "14EM", 手动X轴左右 := "数据接收".手动左右_2, 限位开关X轴 := "14L04", X轴2库正转 := "14M04LI1", X轴1库反转 := "14M04LI2", 手动W轴前后 := "数据接收".手动前后_2, 限位开关W轴 := "14L06", W轴速度写入值 := "2#机械手Z轴速度写入值", W轴原位光电 := "14S14", W轴停止光电 := "14S17", 手动吸盘打开关闭 := "数据接收".开真空_2, X轴定位开关1 := "14S10", X轴定位开关2 := "14S11", 手动Z轴下降 => "2#手动Z轴下降", 手动Z轴上升 => "2#手动Z轴上升", 手动X轴2库移动 => "2#手动X轴2库移动", 手动X轴1库移动 => "2#手动X轴1库移动", 手动W轴前移 => "2#手动W轴前移", 手动W轴后退 => "2#手动W轴回原位", 手动真空阀打开 => "2#手动吸盘电磁阀打开", 手动真空阀关闭 => "2#手动吸盘电磁阀关闭")
   END_RUNG
   RUNG wire#w1
      Contact( "数据接收".手自动状态_2 )
      Move(in := 0, out1 => "数据接收".手动上下_2, out2 => "数据接收".手动左右_2, out3 => "数据接收".手动前后_2)
   END_RUNG
   // the same network as SCL:
   #_w1 := "14EM";
   IF #_w1 THEN
       "2#手动_DB"(机械手手自动状态 := "数据接收".手自动状态_2,   // "手动"
                 手动Z轴上下 := "数据接收".手动上下_2,
                 消音按钮 := "14SB18",
                 限位开关Z轴 := "14L05",
                 Z轴正转下降 := "14M05FWD",
                 Z轴原点光电 := "14S13",
                 Z轴反转上升 := "14M05REV",
                 急停按钮 := "14EM",
                 手动X轴左右 := "数据接收".手动左右_2,
                 限位开关X轴 := "14L04",
                 X轴2库正转 := "14M04LI1",
                 X轴1库反转 := "14M04LI2",
                 手动W轴前后 := "数据接收".手动前后_2,
                 限位开关W轴 := "14L06",
                 W轴速度写入值 := "2#机械手Z轴速度写入值",
                 W轴原位光电 := "14S14",
                 W轴停止光电 := "14S17",
                 手动吸盘打开关闭 := "数据接收".开真空_2,
                 X轴定位开关1 := "14S10",
                 X轴定位开关2 := "14S11",
                 手动Z轴下降 => "2#手动Z轴下降",
                 手动Z轴上升 => "2#手动Z轴上升",
                 手动X轴2库移动 => "2#手动X轴2库移动",
                 手动X轴1库移动 => "2#手动X轴1库移动",
                 手动W轴前移 => "2#手动W轴前移",
                 手动W轴后退 => "2#手动W轴回原位",
                 手动真空阀打开 => "2#手动吸盘电磁阀打开",
                 手动真空阀关闭 => "2#手动吸盘电磁阀关闭");
   END_IF;
   IF #_w1 AND "数据接收".手自动状态_2 THEN
       "数据接收".手动上下_2 := 0;
       "数据接收".手动左右_2 := 0;
       "数据接收".手动前后_2 := 0;
   END_IF;
END_REGION

REGION Network 3: 3#机械手 手动
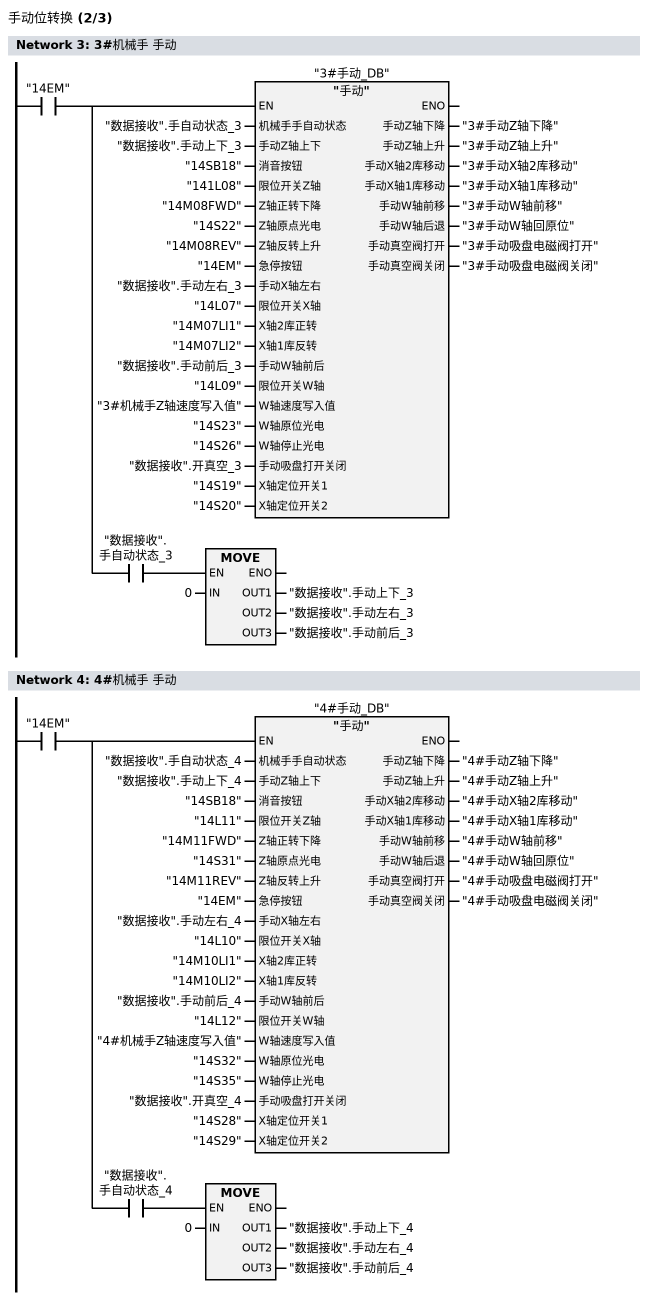
   RUNG wire#powerrail
      Contact( "14EM" )
      wire#w1
      "3#手动_DB"(机械手手自动状态 := "数据接收".手自动状态_3, 手动Z轴上下 := "数据接收".手动上下_3, 消音按钮 := "14SB18", 限位开关Z轴 := "141L08", Z轴正转下降 := "14M08FWD", Z轴原点光电 := "14S22", Z轴反转上升 := "14M08REV", 急停按钮 := "14EM", 手动X轴左右 := "数据接收".手动左右_3, 限位开关X轴 := "14L07", X轴2库正转 := "14M07LI1", X轴1库反转 := "14M07LI2", 手动W轴前后 := "数据接收".手动前后_3, 限位开关W轴 := "14L09", W轴速度写入值 := "3#机械手Z轴速度写入值", W轴原位光电 := "14S23", W轴停止光电 := "14S26", 手动吸盘打开关闭 := "数据接收".开真空_3, X轴定位开关1 := "14S19", X轴定位开关2 := "14S20", 手动Z轴下降 => "3#手动Z轴下降", 手动Z轴上升 => "3#手动Z轴上升", 手动X轴2库移动 => "3#手动X轴2库移动", 手动X轴1库移动 => "3#手动X轴1库移动", 手动W轴前移 => "3#手动W轴前移", 手动W轴后退 => "3#手动W轴回原位", 手动真空阀打开 => "3#手动吸盘电磁阀打开", 手动真空阀关闭 => "3#手动吸盘电磁阀关闭")
   END_RUNG
   RUNG wire#w1
      Contact( "数据接收".手自动状态_3 )
      Move(in := 0, out1 => "数据接收".手动上下_3, out2 => "数据接收".手动左右_3, out3 => "数据接收".手动前后_3)
   END_RUNG
   // the same network as SCL:
   #_w1 := "14EM";
   IF #_w1 THEN
       "3#手动_DB"(机械手手自动状态 := "数据接收".手自动状态_3,   // "手动"
                 手动Z轴上下 := "数据接收".手动上下_3,
                 消音按钮 := "14SB18",
                 限位开关Z轴 := "141L08",
                 Z轴正转下降 := "14M08FWD",
                 Z轴原点光电 := "14S22",
                 Z轴反转上升 := "14M08REV",
                 急停按钮 := "14EM",
                 手动X轴左右 := "数据接收".手动左右_3,
                 限位开关X轴 := "14L07",
                 X轴2库正转 := "14M07LI1",
                 X轴1库反转 := "14M07LI2",
                 手动W轴前后 := "数据接收".手动前后_3,
                 限位开关W轴 := "14L09",
                 W轴速度写入值 := "3#机械手Z轴速度写入值",
                 W轴原位光电 := "14S23",
                 W轴停止光电 := "14S26",
                 手动吸盘打开关闭 := "数据接收".开真空_3,
                 X轴定位开关1 := "14S19",
                 X轴定位开关2 := "14S20",
                 手动Z轴下降 => "3#手动Z轴下降",
                 手动Z轴上升 => "3#手动Z轴上升",
                 手动X轴2库移动 => "3#手动X轴2库移动",
                 手动X轴1库移动 => "3#手动X轴1库移动",
                 手动W轴前移 => "3#手动W轴前移",
                 手动W轴后退 => "3#手动W轴回原位",
                 手动真空阀打开 => "3#手动吸盘电磁阀打开",
                 手动真空阀关闭 => "3#手动吸盘电磁阀关闭");
   END_IF;
   IF #_w1 AND "数据接收".手自动状态_3 THEN
       "数据接收".手动上下_3 := 0;
       "数据接收".手动左右_3 := 0;
       "数据接收".手动前后_3 := 0;
   END_IF;
END_REGION

REGION Network 4: 4#机械手 手动
   RUNG wire#powerrail
      Contact( "14EM" )
      wire#w1
      "4#手动_DB"(机械手手自动状态 := "数据接收".手自动状态_4, 手动Z轴上下 := "数据接收".手动上下_4, 消音按钮 := "14SB18", 限位开关Z轴 := "14L11", Z轴正转下降 := "14M11FWD", Z轴原点光电 := "14S31", Z轴反转上升 := "14M11REV", 急停按钮 := "14EM", 手动X轴左右 := "数据接收".手动左右_4, 限位开关X轴 := "14L10", X轴2库正转 := "14M10LI1", X轴1库反转 := "14M10LI2", 手动W轴前后 := "数据接收".手动前后_4, 限位开关W轴 := "14L12", W轴速度写入值 := "4#机械手Z轴速度写入值", W轴原位光电 := "14S32", W轴停止光电 := "14S35", 手动吸盘打开关闭 := "数据接收".开真空_4, X轴定位开关1 := "14S28", X轴定位开关2 := "14S29", 手动Z轴下降 => "4#手动Z轴下降", 手动Z轴上升 => "4#手动Z轴上升", 手动X轴2库移动 => "4#手动X轴2库移动", 手动X轴1库移动 => "4#手动X轴1库移动", 手动W轴前移 => "4#手动W轴前移", 手动W轴后退 => "4#手动W轴回原位", 手动真空阀打开 => "4#手动吸盘电磁阀打开", 手动真空阀关闭 => "4#手动吸盘电磁阀关闭")
   END_RUNG
   RUNG wire#w1
      Contact( "数据接收".手自动状态_4 )
      Move(in := 0, out1 => "数据接收".手动上下_4, out2 => "数据接收".手动左右_4, out3 => "数据接收".手动前后_4)
   END_RUNG
   // the same network as SCL:
   #_w1 := "14EM";
   IF #_w1 THEN
       "4#手动_DB"(机械手手自动状态 := "数据接收".手自动状态_4,   // "手动"
                 手动Z轴上下 := "数据接收".手动上下_4,
                 消音按钮 := "14SB18",
                 限位开关Z轴 := "14L11",
                 Z轴正转下降 := "14M11FWD",
                 Z轴原点光电 := "14S31",
                 Z轴反转上升 := "14M11REV",
                 急停按钮 := "14EM",
                 手动X轴左右 := "数据接收".手动左右_4,
                 限位开关X轴 := "14L10",
                 X轴2库正转 := "14M10LI1",
                 X轴1库反转 := "14M10LI2",
                 手动W轴前后 := "数据接收".手动前后_4,
                 限位开关W轴 := "14L12",
                 W轴速度写入值 := "4#机械手Z轴速度写入值",
                 W轴原位光电 := "14S32",
                 W轴停止光电 := "14S35",
                 手动吸盘打开关闭 := "数据接收".开真空_4,
                 X轴定位开关1 := "14S28",
                 X轴定位开关2 := "14S29",
                 手动Z轴下降 => "4#手动Z轴下降",
                 手动Z轴上升 => "4#手动Z轴上升",
                 手动X轴2库移动 => "4#手动X轴2库移动",
                 手动X轴1库移动 => "4#手动X轴1库移动",
                 手动W轴前移 => "4#手动W轴前移",
                 手动W轴后退 => "4#手动W轴回原位",
                 手动真空阀打开 => "4#手动吸盘电磁阀打开",
                 手动真空阀关闭 => "4#手动吸盘电磁阀关闭");
   END_IF;
   IF #_w1 AND "数据接收".手自动状态_4 THEN
       "数据接收".手动上下_4 := 0;
       "数据接收".手动左右_4 := 0;
       "数据接收".手动前后_4 := 0;
   END_IF;
END_REGION

REGION Network 5: 5#机械手 手动
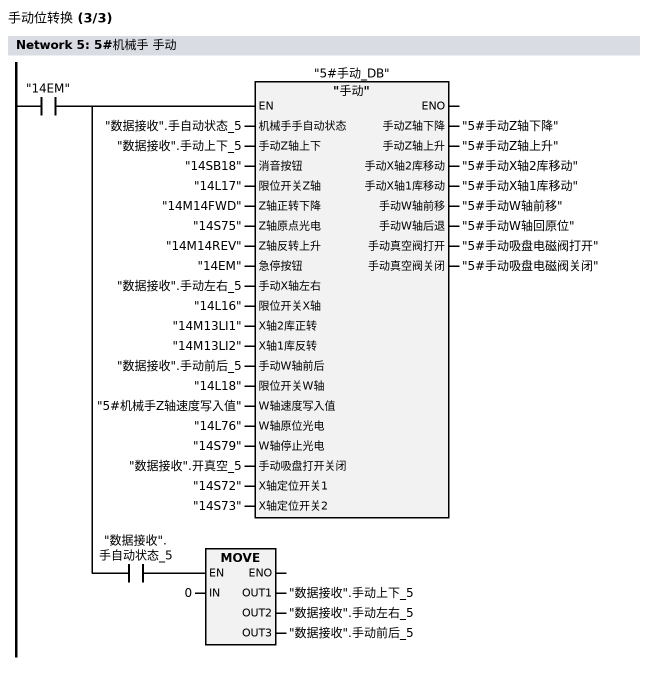
   RUNG wire#powerrail
      Contact( "14EM" )
      wire#w1
      "5#手动_DB"(机械手手自动状态 := "数据接收".手自动状态_5, 手动Z轴上下 := "数据接收".手动上下_5, 消音按钮 := "14SB18", 限位开关Z轴 := "14L17", Z轴正转下降 := "14M14FWD", Z轴原点光电 := "14S75", Z轴反转上升 := "14M14REV", 急停按钮 := "14EM", 手动X轴左右 := "数据接收".手动左右_5, 限位开关X轴 := "14L16", X轴2库正转 := "14M13LI1", X轴1库反转 := "14M13LI2", 手动W轴前后 := "数据接收".手动前后_5, 限位开关W轴 := "14L18", W轴速度写入值 := "5#机械手Z轴速度写入值", W轴原位光电 := "14L76", W轴停止光电 := "14S79", 手动吸盘打开关闭 := "数据接收".开真空_5, X轴定位开关1 := "14S72", X轴定位开关2 := "14S73", 手动Z轴下降 => "5#手动Z轴下降", 手动Z轴上升 => "5#手动Z轴上升", 手动X轴2库移动 => "5#手动X轴2库移动", 手动X轴1库移动 => "5#手动X轴1库移动", 手动W轴前移 => "5#手动W轴前移", 手动W轴后退 => "5#手动W轴回原位", 手动真空阀打开 => "5#手动吸盘电磁阀打开", 手动真空阀关闭 => "5#手动吸盘电磁阀关闭")
   END_RUNG
   RUNG wire#w1
      Contact( "数据接收".手自动状态_5 )
      Move(in := 0, out1 => "数据接收".手动上下_5, out2 => "数据接收".手动左右_5, out3 => "数据接收".手动前后_5)
   END_RUNG
   // the same network as SCL:
   #_w1 := "14EM";
   IF #_w1 THEN
       "5#手动_DB"(机械手手自动状态 := "数据接收".手自动状态_5,   // "手动"
                 手动Z轴上下 := "数据接收".手动上下_5,
                 消音按钮 := "14SB18",
                 限位开关Z轴 := "14L17",
                 Z轴正转下降 := "14M14FWD",
                 Z轴原点光电 := "14S75",
                 Z轴反转上升 := "14M14REV",
                 急停按钮 := "14EM",
                 手动X轴左右 := "数据接收".手动左右_5,
                 限位开关X轴 := "14L16",
                 X轴2库正转 := "14M13LI1",
                 X轴1库反转 := "14M13LI2",
                 手动W轴前后 := "数据接收".手动前后_5,
                 限位开关W轴 := "14L18",
                 W轴速度写入值 := "5#机械手Z轴速度写入值",
                 W轴原位光电 := "14L76",
                 W轴停止光电 := "14S79",
                 手动吸盘打开关闭 := "数据接收".开真空_5,
                 X轴定位开关1 := "14S72",
                 X轴定位开关2 := "14S73",
                 手动Z轴下降 => "5#手动Z轴下降",
                 手动Z轴上升 => "5#手动Z轴上升",
                 手动X轴2库移动 => "5#手动X轴2库移动",
                 手动X轴1库移动 => "5#手动X轴1库移动",
                 手动W轴前移 => "5#手动W轴前移",
                 手动W轴后退 => "5#手动W轴回原位",
                 手动真空阀打开 => "5#手动吸盘电磁阀打开",
                 手动真空阀关闭 => "5#手动吸盘电磁阀关闭");
   END_IF;
   IF #_w1 AND "数据接收".手自动状态_5 THEN
       "数据接收".手动上下_5 := 0;
       "数据接收".手动左右_5 := 0;
       "数据接收".手动前后_5 := 0;
   END_IF;
END_REGION
END_FUNCTION

FUNCTION "灯定义/按钮激活" : Void   // FC18, LAD
{ S7_Optimized_Access := 'TRUE' }
VERSION : 0.1
   VAR_TEMP   // added for the SCL form of the ladder/FBD networks
      _w1 : Bool;
      _w2 : Bool;
      _w3 : Bool;
   END_VAR
BEGIN

REGION Network 1: 设备急停 上位机断开连接
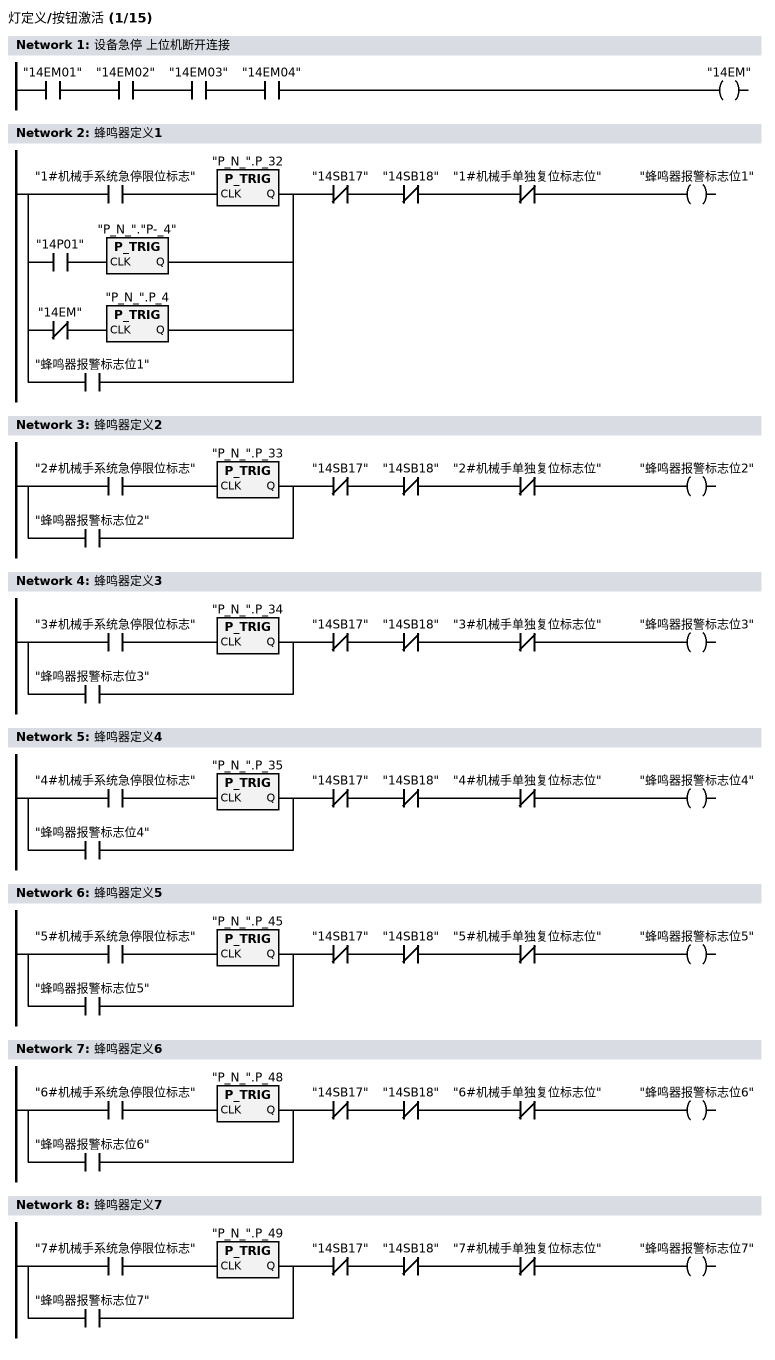
   RUNG wire#powerrail
      Contact( "14EM01" )
      Contact( "14EM02" )
      Contact( "14EM03" )
      Contact( "14EM04" )
      Coil( "14EM" )
   END_RUNG
   // the same network as SCL:
   "14EM" := "14EM01" AND "14EM02" AND "14EM03" AND "14EM04";
END_REGION

REGION Network 2: 蜂鸣器定义1
   RUNG wire#powerrail
      Contact( "1#机械手系统急停限位标志" )
      P_Trig( "P_N_".P_32 )
      wire#w1
      I_Contact( "14SB17" )
      I_Contact( "14SB18" )
      I_Contact( "1#机械手单独复位标志位" )
      Coil( "蜂鸣器报警标志位1" )
   END_RUNG
   RUNG wire#powerrail
      Contact( "14P01" )
      P_Trig( "P_N_"."P-_4" )
   END_RUNG wire#w1
   RUNG wire#powerrail
      I_Contact( "14EM" )
      P_Trig( "P_N_".P_4 )
   END_RUNG wire#w1
   RUNG wire#powerrail
      Contact( "蜂鸣器报警标志位1" )
   END_RUNG wire#w1
   // the same network as SCL:
   #_w1 := "1#机械手系统急停限位标志" AND NOT "P_N_".P_32;   // rising edge
   "P_N_".P_32 := "1#机械手系统急停限位标志";
   #_w2 := "14P01" AND NOT "P_N_"."P-_4";   // rising edge
   "P_N_"."P-_4" := "14P01";
   #_w3 := NOT "14EM" AND NOT "P_N_".P_4;   // rising edge
   "P_N_".P_4 := NOT "14EM";
   "蜂鸣器报警标志位1" := (#_w1 OR #_w2 OR #_w3 OR "蜂鸣器报警标志位1") AND NOT "14SB17" AND NOT "14SB18" AND NOT "1#机械手单独复位标志位";
END_REGION

REGION Network 3: 蜂鸣器定义2
   RUNG wire#powerrail
      Contact( "2#机械手系统急停限位标志" )
      P_Trig( "P_N_".P_33 )
      wire#w1
      I_Contact( "14SB17" )
      I_Contact( "14SB18" )
      I_Contact( "2#机械手单独复位标志位" )
      Coil( "蜂鸣器报警标志位2" )
   END_RUNG
   RUNG wire#powerrail
      Contact( "蜂鸣器报警标志位2" )
   END_RUNG wire#w1
   // the same network as SCL:
   #_w1 := "2#机械手系统急停限位标志" AND NOT "P_N_".P_33;   // rising edge
   "P_N_".P_33 := "2#机械手系统急停限位标志";
   "蜂鸣器报警标志位2" := (#_w1 OR "蜂鸣器报警标志位2") AND NOT "14SB17" AND NOT "14SB18" AND NOT "2#机械手单独复位标志位";
END_REGION

REGION Network 4: 蜂鸣器定义3
   RUNG wire#powerrail
      Contact( "3#机械手系统急停限位标志" )
      P_Trig( "P_N_".P_34 )
      wire#w1
      I_Contact( "14SB17" )
      I_Contact( "14SB18" )
      I_Contact( "3#机械手单独复位标志位" )
      Coil( "蜂鸣器报警标志位3" )
   END_RUNG
   RUNG wire#powerrail
      Contact( "蜂鸣器报警标志位3" )
   END_RUNG wire#w1
   // the same network as SCL:
   #_w1 := "3#机械手系统急停限位标志" AND NOT "P_N_".P_34;   // rising edge
   "P_N_".P_34 := "3#机械手系统急停限位标志";
   "蜂鸣器报警标志位3" := (#_w1 OR "蜂鸣器报警标志位3") AND NOT "14SB17" AND NOT "14SB18" AND NOT "3#机械手单独复位标志位";
END_REGION

REGION Network 5: 蜂鸣器定义4
   RUNG wire#powerrail
      Contact( "4#机械手系统急停限位标志" )
      P_Trig( "P_N_".P_35 )
      wire#w1
      I_Contact( "14SB17" )
      I_Contact( "14SB18" )
      I_Contact( "4#机械手单独复位标志位" )
      Coil( "蜂鸣器报警标志位4" )
   END_RUNG
   RUNG wire#powerrail
      Contact( "蜂鸣器报警标志位4" )
   END_RUNG wire#w1
   // the same network as SCL:
   #_w1 := "4#机械手系统急停限位标志" AND NOT "P_N_".P_35;   // rising edge
   "P_N_".P_35 := "4#机械手系统急停限位标志";
   "蜂鸣器报警标志位4" := (#_w1 OR "蜂鸣器报警标志位4") AND NOT "14SB17" AND NOT "14SB18" AND NOT "4#机械手单独复位标志位";
END_REGION

REGION Network 6: 蜂鸣器定义5
   RUNG wire#powerrail
      Contact( "5#机械手系统急停限位标志" )
      P_Trig( "P_N_".P_45 )
      wire#w1
      I_Contact( "14SB17" )
      I_Contact( "14SB18" )
      I_Contact( "5#机械手单独复位标志位" )
      Coil( "蜂鸣器报警标志位5" )
   END_RUNG
   RUNG wire#powerrail
      Contact( "蜂鸣器报警标志位5" )
   END_RUNG wire#w1
   // the same network as SCL:
   #_w1 := "5#机械手系统急停限位标志" AND NOT "P_N_".P_45;   // rising edge
   "P_N_".P_45 := "5#机械手系统急停限位标志";
   "蜂鸣器报警标志位5" := (#_w1 OR "蜂鸣器报警标志位5") AND NOT "14SB17" AND NOT "14SB18" AND NOT "5#机械手单独复位标志位";
END_REGION

REGION Network 7: 蜂鸣器定义6
   RUNG wire#powerrail
      Contact( "6#机械手系统急停限位标志" )
      P_Trig( "P_N_".P_48 )
      wire#w1
      I_Contact( "14SB17" )
      I_Contact( "14SB18" )
      I_Contact( "6#机械手单独复位标志位" )
      Coil( "蜂鸣器报警标志位6" )
   END_RUNG
   RUNG wire#powerrail
      Contact( "蜂鸣器报警标志位6" )
   END_RUNG wire#w1
   // the same network as SCL:
   #_w1 := "6#机械手系统急停限位标志" AND NOT "P_N_".P_48;   // rising edge
   "P_N_".P_48 := "6#机械手系统急停限位标志";
   "蜂鸣器报警标志位6" := (#_w1 OR "蜂鸣器报警标志位6") AND NOT "14SB17" AND NOT "14SB18" AND NOT "6#机械手单独复位标志位";
END_REGION

REGION Network 8: 蜂鸣器定义7
   RUNG wire#powerrail
      Contact( "7#机械手系统急停限位标志" )
      P_Trig( "P_N_".P_49 )
      wire#w1
      I_Contact( "14SB17" )
      I_Contact( "14SB18" )
      I_Contact( "7#机械手单独复位标志位" )
      Coil( "蜂鸣器报警标志位7" )
   END_RUNG
   RUNG wire#powerrail
      Contact( "蜂鸣器报警标志位7" )
   END_RUNG wire#w1
   // the same network as SCL:
   #_w1 := "7#机械手系统急停限位标志" AND NOT "P_N_".P_49;   // rising edge
   "P_N_".P_49 := "7#机械手系统急停限位标志";
   "蜂鸣器报警标志位7" := (#_w1 OR "蜂鸣器报警标志位7") AND NOT "14SB17" AND NOT "14SB18" AND NOT "7#机械手单独复位标志位";
END_REGION

REGION Network 9: 启动按钮激活
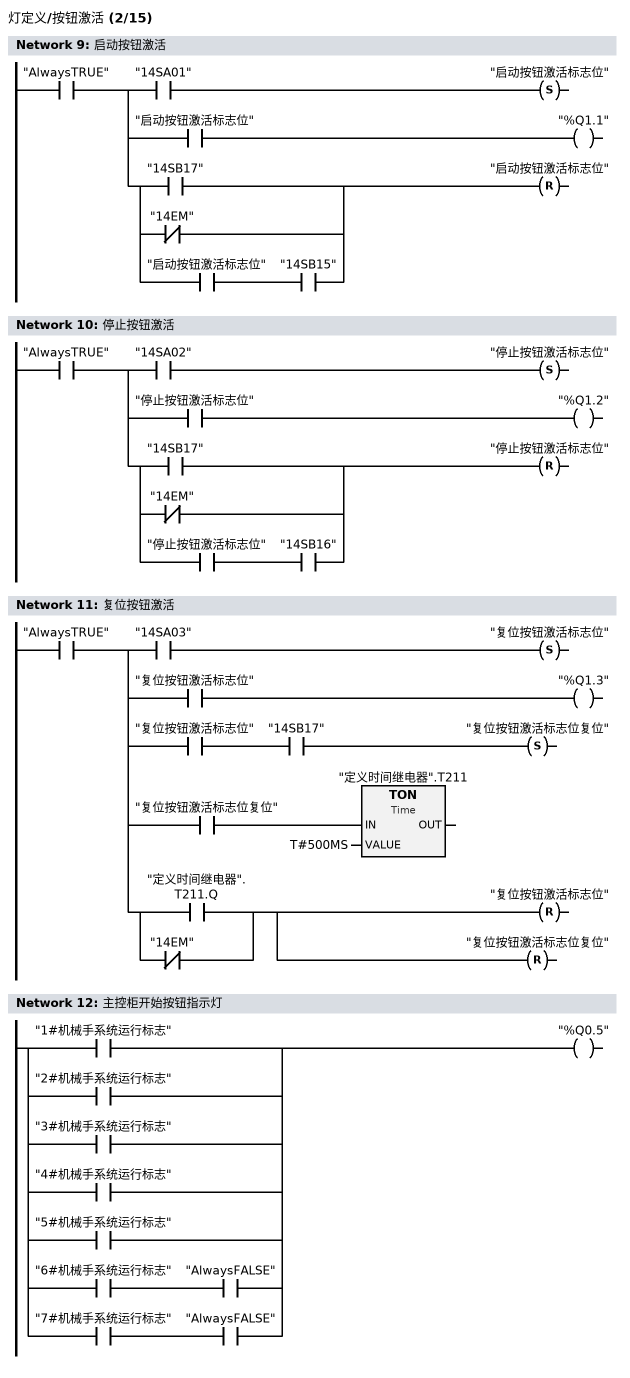
   RUNG wire#powerrail
      Contact( "AlwaysTRUE" )
      wire#w1
      Contact( "14SA01" )
      S_Coil( "启动按钮激活标志位" )
   END_RUNG
   RUNG wire#w1
      Contact( "启动按钮激活标志位" )
      Coil( "%Q1.1" )
   END_RUNG
   RUNG wire#w1
      Contact( "14SB17" )
      wire#w2
      R_Coil( "启动按钮激活标志位" )
   END_RUNG
   RUNG wire#w1
      I_Contact( "14EM" )
   END_RUNG wire#w2
   RUNG wire#w1
      Contact( "启动按钮激活标志位" )
      Contact( "14SB15" )
   END_RUNG wire#w2
   // the same network as SCL:
   IF "AlwaysTRUE" AND "14SA01" THEN "启动按钮激活标志位" := TRUE; END_IF;
   "%Q1.1" := "AlwaysTRUE" AND "启动按钮激活标志位";
   IF "AlwaysTRUE" AND ("14SB17" OR NOT "14EM" OR ("启动按钮激活标志位" AND "14SB15")) THEN
       "启动按钮激活标志位" := FALSE;
   END_IF;
END_REGION

REGION Network 10: 停止按钮激活
   RUNG wire#powerrail
      Contact( "AlwaysTRUE" )
      wire#w1
      Contact( "14SA02" )
      S_Coil( "停止按钮激活标志位" )
   END_RUNG
   RUNG wire#w1
      Contact( "停止按钮激活标志位" )
      Coil( "%Q1.2" )
   END_RUNG
   RUNG wire#w1
      Contact( "14SB17" )
      wire#w2
      R_Coil( "停止按钮激活标志位" )
   END_RUNG
   RUNG wire#w1
      I_Contact( "14EM" )
   END_RUNG wire#w2
   RUNG wire#w1
      Contact( "停止按钮激活标志位" )
      Contact( "14SB16" )
   END_RUNG wire#w2
   // the same network as SCL:
   IF "AlwaysTRUE" AND "14SA02" THEN "停止按钮激活标志位" := TRUE; END_IF;
   "%Q1.2" := "AlwaysTRUE" AND "停止按钮激活标志位";
   IF "AlwaysTRUE" AND ("14SB17" OR NOT "14EM" OR ("停止按钮激活标志位" AND "14SB16")) THEN
       "停止按钮激活标志位" := FALSE;
   END_IF;
END_REGION

REGION Network 11: 复位按钮激活
   IF "AlwaysTRUE" AND "14SA03" THEN "复位按钮激活标志位" := TRUE; END_IF;
   "%Q1.3" := "AlwaysTRUE" AND "复位按钮激活标志位";
   IF "AlwaysTRUE" AND "复位按钮激活标志位" AND "14SB17" THEN "复位按钮激活标志位复位" := TRUE; END_IF;
   "定义时间继电器".T211.TON(IN := "AlwaysTRUE" AND "复位按钮激活标志位复位", PT := T#500MS);   // TON coil
   IF "AlwaysTRUE" AND ("定义时间继电器".T211.Q OR NOT "14EM") THEN
       "复位按钮激活标志位" := FALSE;
       "复位按钮激活标志位复位" := FALSE;
   END_IF;
END_REGION

REGION Network 12: 主控柜开始按钮指示灯
   RUNG wire#powerrail
      Contact( "1#机械手系统运行标志" )
      wire#w1
      Coil( "%Q0.5" )
   END_RUNG
   RUNG wire#powerrail
      Contact( "2#机械手系统运行标志" )
   END_RUNG wire#w1
   RUNG wire#powerrail
      Contact( "3#机械手系统运行标志" )
   END_RUNG wire#w1
   RUNG wire#powerrail
      Contact( "4#机械手系统运行标志" )
   END_RUNG wire#w1
   RUNG wire#powerrail
      Contact( "5#机械手系统运行标志" )
   END_RUNG wire#w1
   RUNG wire#powerrail
      Contact( "6#机械手系统运行标志" )
      Contact( "AlwaysFALSE" )
   END_RUNG wire#w1
   RUNG wire#powerrail
      Contact( "7#机械手系统运行标志" )
      Contact( "AlwaysFALSE" )
   END_RUNG wire#w1
   // the same network as SCL:
   "%Q0.5" := "1#机械手系统运行标志" OR "2#机械手系统运行标志" OR "3#机械手系统运行标志" OR "4#机械手系统运行标志" OR "5#机械手系统运行标志" OR ("6#机械手系统运行标志" AND "AlwaysFALSE") OR ("7#机械手系统运行标志" AND "AlwaysFALSE");
END_REGION

REGION Network 13: 主控柜停止按钮指示灯
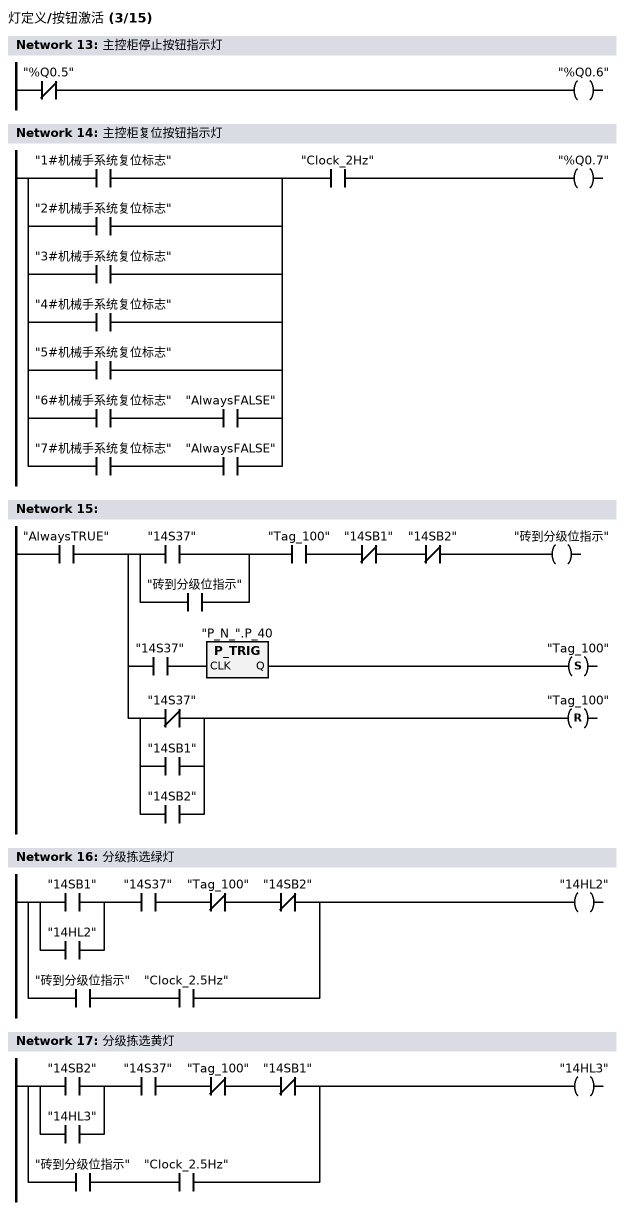
   RUNG wire#powerrail
      I_Contact( "%Q0.5" )
      Coil( "%Q0.6" )
   END_RUNG
   // the same network as SCL:
   "%Q0.6" := NOT "%Q0.5";
END_REGION

REGION Network 14: 主控柜复位按钮指示灯
   RUNG wire#powerrail
      Contact( "1#机械手系统复位标志" )
      wire#w1
      Contact( "Clock_2Hz" )
      Coil( "%Q0.7" )
   END_RUNG
   RUNG wire#powerrail
      Contact( "2#机械手系统复位标志" )
   END_RUNG wire#w1
   RUNG wire#powerrail
      Contact( "3#机械手系统复位标志" )
   END_RUNG wire#w1
   RUNG wire#powerrail
      Contact( "4#机械手系统复位标志" )
   END_RUNG wire#w1
   RUNG wire#powerrail
      Contact( "5#机械手系统复位标志" )
   END_RUNG wire#w1
   RUNG wire#powerrail
      Contact( "6#机械手系统复位标志" )
      Contact( "AlwaysFALSE" )
   END_RUNG wire#w1
   RUNG wire#powerrail
      Contact( "7#机械手系统复位标志" )
      Contact( "AlwaysFALSE" )
   END_RUNG wire#w1
   // the same network as SCL:
   "%Q0.7" := ("1#机械手系统复位标志" OR "2#机械手系统复位标志" OR "3#机械手系统复位标志" OR "4#机械手系统复位标志" OR "5#机械手系统复位标志" OR ("6#机械手系统复位标志" AND "AlwaysFALSE") OR ("7#机械手系统复位标志" AND "AlwaysFALSE")) AND "Clock_2Hz";
END_REGION

REGION Network 15
   RUNG wire#powerrail
      Contact( "AlwaysTRUE" )
      wire#w1
      Contact( "14S37" )
      wire#w2
      Contact( "Tag_100" )
      I_Contact( "14SB1" )
      I_Contact( "14SB2" )
      Coil( "砖到分级位指示" )
   END_RUNG
   RUNG wire#w1
      Contact( "砖到分级位指示" )
   END_RUNG wire#w2
   RUNG wire#w1
      Contact( "14S37" )
      P_Trig( "P_N_".P_40 )
      S_Coil( "Tag_100" )
   END_RUNG
   RUNG wire#w1
      I_Contact( "14S37" )
      wire#w3
      R_Coil( "Tag_100" )
   END_RUNG
   RUNG wire#w1
      Contact( "14SB1" )
   END_RUNG wire#w3
   RUNG wire#w1
      Contact( "14SB2" )
   END_RUNG wire#w3
   // the same network as SCL:
   "砖到分级位指示" := "AlwaysTRUE" AND ("14S37" OR "砖到分级位指示") AND "Tag_100" AND NOT "14SB1" AND NOT "14SB2";
   #_w1 := "AlwaysTRUE" AND "14S37";
   #_w2 := #_w1 AND NOT "P_N_".P_40;   // rising edge
   "P_N_".P_40 := #_w1;
   IF #_w2 THEN "Tag_100" := TRUE; END_IF;
   IF "AlwaysTRUE" AND (NOT "14S37" OR "14SB1" OR "14SB2") THEN "Tag_100" := FALSE; END_IF;
END_REGION

REGION Network 16: 分级拣选绿灯
   RUNG wire#powerrail
      Contact( "14SB1" )
      wire#w1
      Contact( "14S37" )
      I_Contact( "Tag_100" )
      I_Contact( "14SB2" )
      wire#w2
      Coil( "14HL2" )
   END_RUNG
   RUNG wire#powerrail
      Contact( "14HL2" )
   END_RUNG wire#w1
   RUNG wire#powerrail
      Contact( "砖到分级位指示" )
      Contact( "Clock_2.5Hz" )
   END_RUNG wire#w2
   // the same network as SCL:
   "14HL2" := (("14SB1" OR "14HL2") AND "14S37" AND NOT "Tag_100" AND NOT "14SB2") OR ("砖到分级位指示" AND "Clock_2.5Hz");
END_REGION

REGION Network 17: 分级拣选黄灯
   RUNG wire#powerrail
      Contact( "14SB2" )
      wire#w1
      Contact( "14S37" )
      I_Contact( "Tag_100" )
      I_Contact( "14SB1" )
      wire#w2
      Coil( "14HL3" )
   END_RUNG
   RUNG wire#powerrail
      Contact( "14HL3" )
   END_RUNG wire#w1
   RUNG wire#powerrail
      Contact( "砖到分级位指示" )
      Contact( "Clock_2.5Hz" )
   END_RUNG wire#w2
   // the same network as SCL:
   "14HL3" := (("14SB2" OR "14HL3") AND "14S37" AND NOT "Tag_100" AND NOT "14SB1") OR ("砖到分级位指示" AND "Clock_2.5Hz");
END_REGION

REGION Network 18: 换花色红色指示灯
END_REGION

REGION Network 19: 四色红灯 DB2.DBX16.5 上位机通讯断开 DB2.DBX16.6与18PLC断开
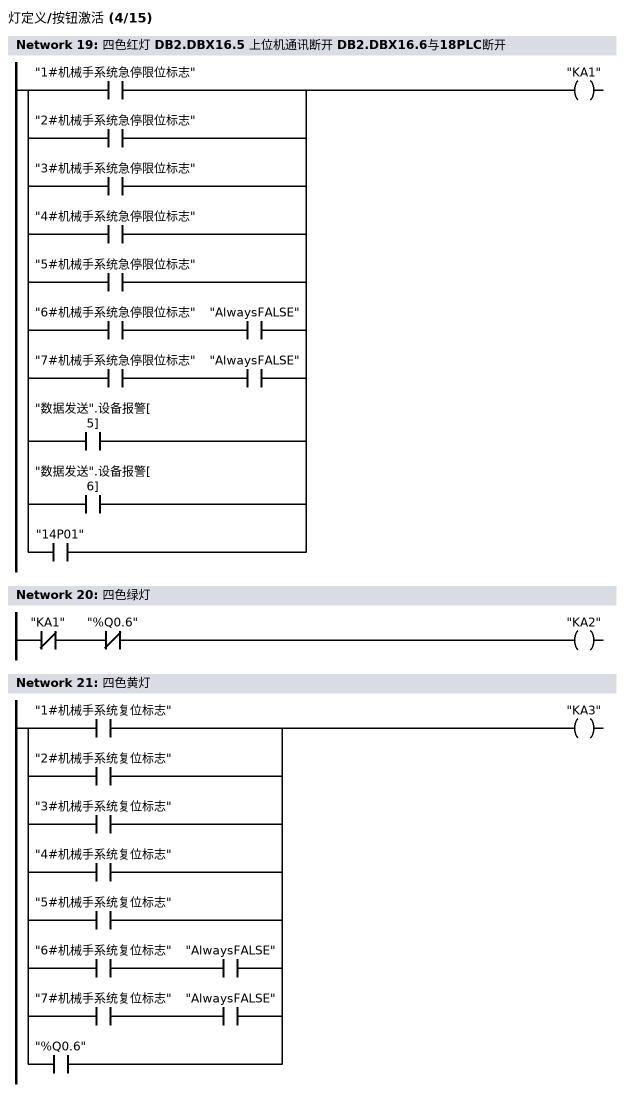
   RUNG wire#powerrail
      Contact( "1#机械手系统急停限位标志" )
      wire#w1
      Coil( "KA1" )
   END_RUNG
   RUNG wire#powerrail
      Contact( "2#机械手系统急停限位标志" )
   END_RUNG wire#w1
   RUNG wire#powerrail
      Contact( "3#机械手系统急停限位标志" )
   END_RUNG wire#w1
   RUNG wire#powerrail
      Contact( "4#机械手系统急停限位标志" )
   END_RUNG wire#w1
   RUNG wire#powerrail
      Contact( "5#机械手系统急停限位标志" )
   END_RUNG wire#w1
   RUNG wire#powerrail
      Contact( "6#机械手系统急停限位标志" )
      Contact( "AlwaysFALSE" )
   END_RUNG wire#w1
   RUNG wire#powerrail
      Contact( "7#机械手系统急停限位标志" )
      Contact( "AlwaysFALSE" )
   END_RUNG wire#w1
   RUNG wire#powerrail
      Contact( "数据发送".设备报警[5] )
   END_RUNG wire#w1
   RUNG wire#powerrail
      Contact( "数据发送".设备报警[6] )
   END_RUNG wire#w1
   RUNG wire#powerrail
      Contact( "14P01" )
   END_RUNG wire#w1
   // the same network as SCL:
   "KA1" := "1#机械手系统急停限位标志" OR "2#机械手系统急停限位标志" OR "3#机械手系统急停限位标志" OR "4#机械手系统急停限位标志" OR "5#机械手系统急停限位标志" OR ("6#机械手系统急停限位标志" AND "AlwaysFALSE") OR ("7#机械手系统急停限位标志" AND "AlwaysFALSE") OR "数据发送".设备报警[5] OR "数据发送".设备报警[6] OR "14P01";
END_REGION

REGION Network 20: 四色绿灯
   RUNG wire#powerrail
      I_Contact( "KA1" )
      I_Contact( "%Q0.6" )
      Coil( "KA2" )
   END_RUNG
   // the same network as SCL:
   "KA2" := NOT "KA1" AND NOT "%Q0.6";
END_REGION

REGION Network 21: 四色黄灯
   RUNG wire#powerrail
      Contact( "1#机械手系统复位标志" )
      wire#w1
      Coil( "KA3" )
   END_RUNG
   RUNG wire#powerrail
      Contact( "2#机械手系统复位标志" )
   END_RUNG wire#w1
   RUNG wire#powerrail
      Contact( "3#机械手系统复位标志" )
   END_RUNG wire#w1
   RUNG wire#powerrail
      Contact( "4#机械手系统复位标志" )
   END_RUNG wire#w1
   RUNG wire#powerrail
      Contact( "5#机械手系统复位标志" )
   END_RUNG wire#w1
   RUNG wire#powerrail
      Contact( "6#机械手系统复位标志" )
      Contact( "AlwaysFALSE" )
   END_RUNG wire#w1
   RUNG wire#powerrail
      Contact( "7#机械手系统复位标志" )
      Contact( "AlwaysFALSE" )
   END_RUNG wire#w1
   RUNG wire#powerrail
      Contact( "%Q0.6" )
   END_RUNG wire#w1
   // the same network as SCL:
   "KA3" := "1#机械手系统复位标志" OR "2#机械手系统复位标志" OR "3#机械手系统复位标志" OR "4#机械手系统复位标志" OR "5#机械手系统复位标志" OR ("6#机械手系统复位标志" AND "AlwaysFALSE") OR ("7#机械手系统复位标志" AND "AlwaysFALSE") OR "%Q0.6";
END_REGION

REGION Network 22: 四色蓝灯
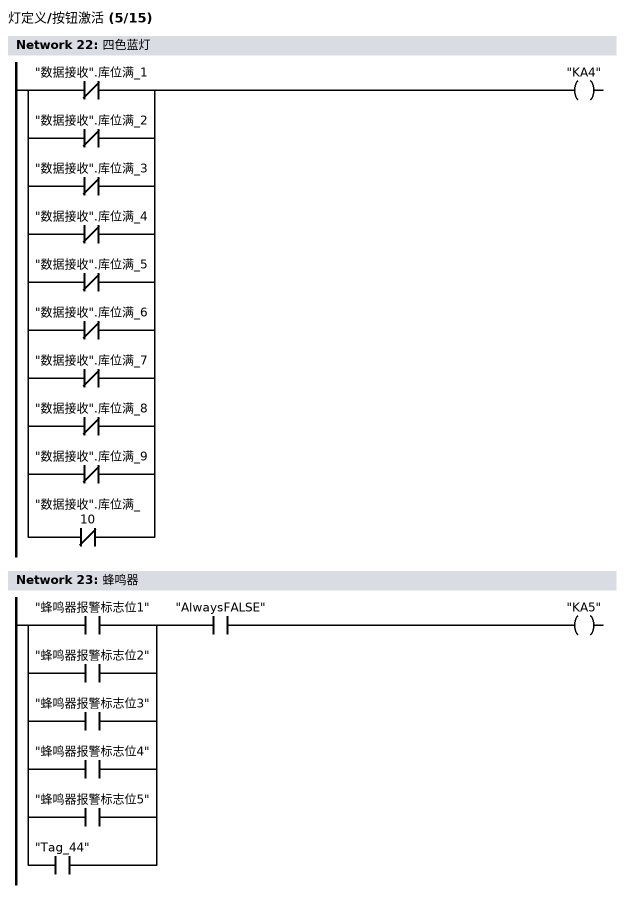
   RUNG wire#powerrail
      I_Contact( "数据接收".库位满_1 )
      wire#w1
      Coil( "KA4" )
   END_RUNG
   RUNG wire#powerrail
      I_Contact( "数据接收".库位满_2 )
   END_RUNG wire#w1
   RUNG wire#powerrail
      I_Contact( "数据接收".库位满_3 )
   END_RUNG wire#w1
   RUNG wire#powerrail
      I_Contact( "数据接收".库位满_4 )
   END_RUNG wire#w1
   RUNG wire#powerrail
      I_Contact( "数据接收".库位满_5 )
   END_RUNG wire#w1
   RUNG wire#powerrail
      I_Contact( "数据接收".库位满_6 )
   END_RUNG wire#w1
   RUNG wire#powerrail
      I_Contact( "数据接收".库位满_7 )
   END_RUNG wire#w1
   RUNG wire#powerrail
      I_Contact( "数据接收".库位满_8 )
   END_RUNG wire#w1
   RUNG wire#powerrail
      I_Contact( "数据接收".库位满_9 )
   END_RUNG wire#w1
   RUNG wire#powerrail
      I_Contact( "数据接收".库位满_10 )
   END_RUNG wire#w1
   // the same network as SCL:
   "KA4" := NOT "数据接收".库位满_1 OR NOT "数据接收".库位满_2 OR NOT "数据接收".库位满_3 OR NOT "数据接收".库位满_4 OR NOT "数据接收".库位满_5 OR NOT "数据接收".库位满_6 OR NOT "数据接收".库位满_7 OR NOT "数据接收".库位满_8 OR NOT "数据接收".库位满_9 OR NOT "数据接收".库位满_10;
END_REGION

REGION Network 23: 蜂鸣器
   RUNG wire#powerrail
      Contact( "蜂鸣器报警标志位1" )
      wire#w1
      Contact( "AlwaysFALSE" )
      Coil( "KA5" )
   END_RUNG
   RUNG wire#powerrail
      Contact( "蜂鸣器报警标志位2" )
   END_RUNG wire#w1
   RUNG wire#powerrail
      Contact( "蜂鸣器报警标志位3" )
   END_RUNG wire#w1
   RUNG wire#powerrail
      Contact( "蜂鸣器报警标志位4" )
   END_RUNG wire#w1
   RUNG wire#powerrail
      Contact( "蜂鸣器报警标志位5" )
   END_RUNG wire#w1
   RUNG wire#powerrail
      Contact( "Tag_44" )
   END_RUNG wire#w1
   // the same network as SCL:
   "KA5" := ("蜂鸣器报警标志位1" OR "蜂鸣器报警标志位2" OR "蜂鸣器报警标志位3" OR "蜂鸣器报警标志位4" OR "蜂鸣器报警标志位5" OR "Tag_44") AND "AlwaysFALSE";
END_REGION

REGION Network 24: 1号库位红灯
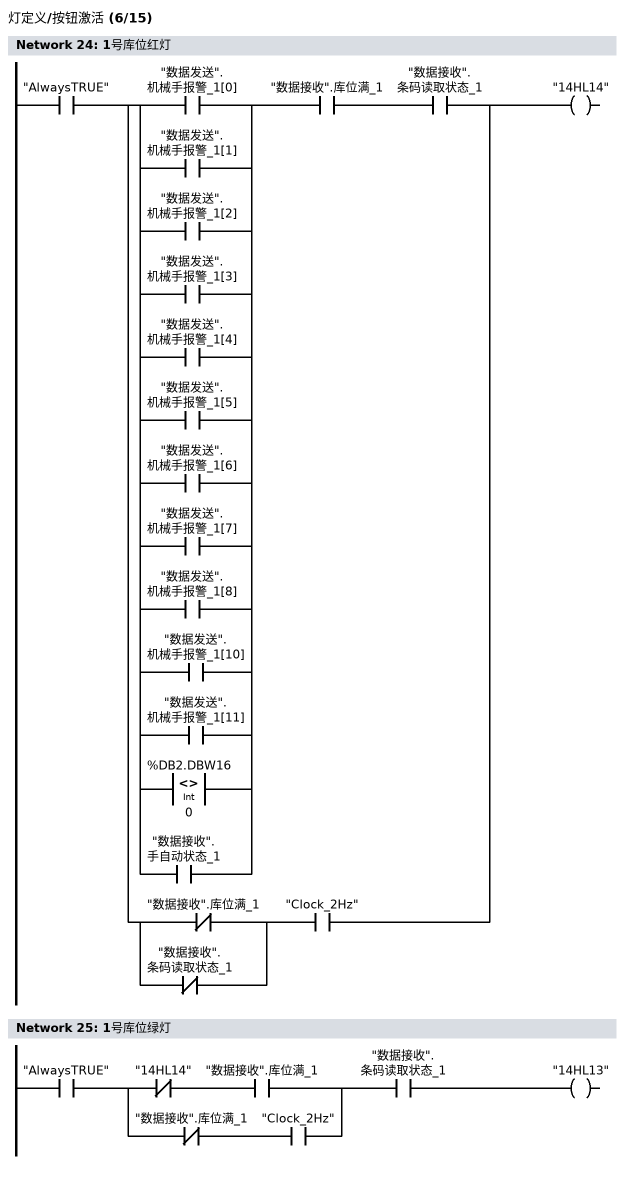
   RUNG wire#powerrail
      Contact( "AlwaysTRUE" )
      wire#w1
      Contact( "数据发送".机械手报警_1[0] )
      wire#w2
      Contact( "数据接收".库位满_1 )
      Contact( "数据接收".条码读取状态_1 )
      wire#w3
      Coil( "14HL14" )
   END_RUNG
   RUNG wire#w1
      Contact( "数据发送".机械手报警_1[1] )
   END_RUNG wire#w2
   RUNG wire#w1
      Contact( "数据发送".机械手报警_1[2] )
   END_RUNG wire#w2
   RUNG wire#w1
      Contact( "数据发送".机械手报警_1[3] )
   END_RUNG wire#w2
   RUNG wire#w1
      Contact( "数据发送".机械手报警_1[4] )
   END_RUNG wire#w2
   RUNG wire#w1
      Contact( "数据发送".机械手报警_1[5] )
   END_RUNG wire#w2
   RUNG wire#w1
      Contact( "数据发送".机械手报警_1[6] )
   END_RUNG wire#w2
   RUNG wire#w1
      Contact( "数据发送".机械手报警_1[7] )
   END_RUNG wire#w2
   RUNG wire#w1
      Contact( "数据发送".机械手报警_1[8] )
   END_RUNG wire#w2
   RUNG wire#w1
      Contact( "数据发送".机械手报警_1[10] )
   END_RUNG wire#w2
   RUNG wire#w1
      Contact( "数据发送".机械手报警_1[11] )
   END_RUNG wire#w2
   RUNG wire#w1
      { S7_Templates := "SrcType := Int" } NE_Contact(in1 := %DB2.DBW16, in2 := 0)
   END_RUNG wire#w2
   RUNG wire#w1
      Contact( "数据接收".手自动状态_1 )
   END_RUNG wire#w2
   RUNG wire#w1
      I_Contact( "数据接收".库位满_1 )
      wire#w4
      Contact( "Clock_2Hz" )
   END_RUNG wire#w3
   RUNG wire#w1
      I_Contact( "数据接收".条码读取状态_1 )
   END_RUNG wire#w4
   // the same network as SCL:
   "14HL14" := "AlwaysTRUE" AND ((("数据发送".机械手报警_1[0] OR "数据发送".机械手报警_1[1] OR "数据发送".机械手报警_1[2] OR "数据发送".机械手报警_1[3] OR "数据发送".机械手报警_1[4] OR "数据发送".机械手报警_1[5] OR "数据发送".机械手报警_1[6] OR "数据发送".机械手报警_1[7] OR "数据发送".机械手报警_1[8] OR "数据发送".机械手报警_1[10] OR "数据发送".机械手报警_1[11] OR (%DB2.DBW16 <> 0) OR "数据接收".手自动状态_1) AND "数据接收".库位满_1 AND "数据接收".条码读取状态_1) OR ((NOT "数据接收".库位满_1 OR NOT "数据接收".条码读取状态_1) AND "Clock_2Hz"));
END_REGION

REGION Network 25: 1号库位绿灯
   RUNG wire#powerrail
      Contact( "AlwaysTRUE" )
      wire#w1
      I_Contact( "14HL14" )
      Contact( "数据接收".库位满_1 )
      wire#w2
      Contact( "数据接收".条码读取状态_1 )
      Coil( "14HL13" )
   END_RUNG
   RUNG wire#w1
      I_Contact( "数据接收".库位满_1 )
      Contact( "Clock_2Hz" )
   END_RUNG wire#w2
   // the same network as SCL:
   "14HL13" := "AlwaysTRUE" AND ((NOT "14HL14" AND "数据接收".库位满_1) OR (NOT "数据接收".库位满_1 AND "Clock_2Hz")) AND "数据接收".条码读取状态_1;
END_REGION

REGION Network 26: 2号库位红灯
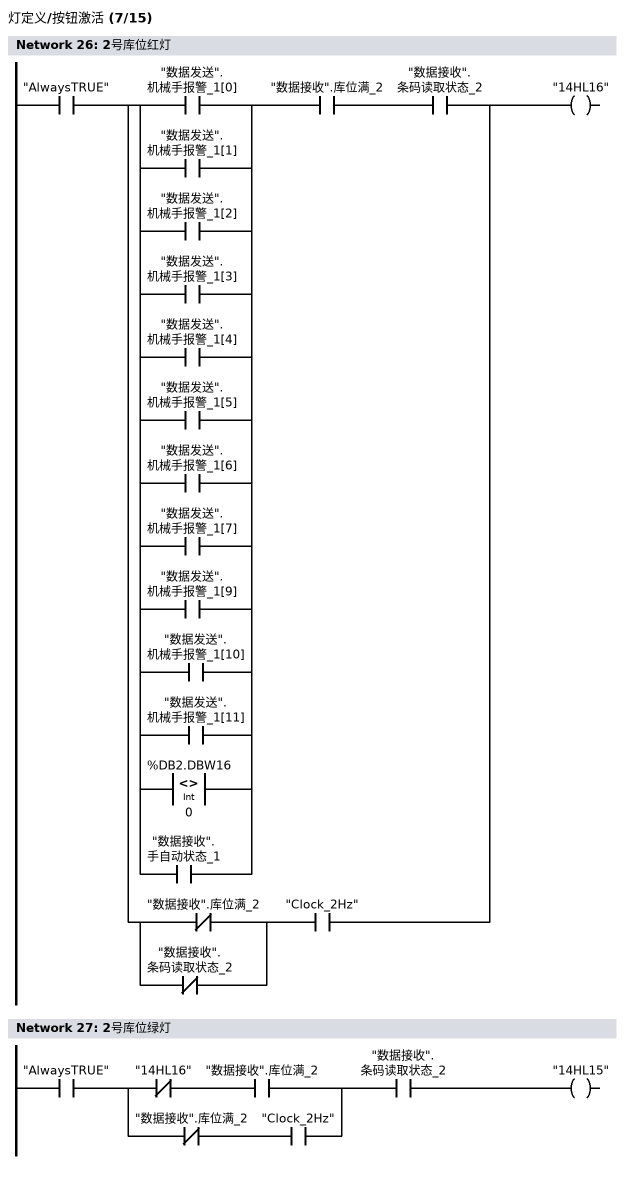
   RUNG wire#powerrail
      Contact( "AlwaysTRUE" )
      wire#w1
      Contact( "数据发送".机械手报警_1[0] )
      wire#w2
      Contact( "数据接收".库位满_2 )
      Contact( "数据接收".条码读取状态_2 )
      wire#w3
      Coil( "14HL16" )
   END_RUNG
   RUNG wire#w1
      Contact( "数据发送".机械手报警_1[1] )
   END_RUNG wire#w2
   RUNG wire#w1
      Contact( "数据发送".机械手报警_1[2] )
   END_RUNG wire#w2
   RUNG wire#w1
      Contact( "数据发送".机械手报警_1[3] )
   END_RUNG wire#w2
   RUNG wire#w1
      Contact( "数据发送".机械手报警_1[4] )
   END_RUNG wire#w2
   RUNG wire#w1
      Contact( "数据发送".机械手报警_1[5] )
   END_RUNG wire#w2
   RUNG wire#w1
      Contact( "数据发送".机械手报警_1[6] )
   END_RUNG wire#w2
   RUNG wire#w1
      Contact( "数据发送".机械手报警_1[7] )
   END_RUNG wire#w2
   RUNG wire#w1
      Contact( "数据发送".机械手报警_1[9] )
   END_RUNG wire#w2
   RUNG wire#w1
      Contact( "数据发送".机械手报警_1[10] )
   END_RUNG wire#w2
   RUNG wire#w1
      Contact( "数据发送".机械手报警_1[11] )
   END_RUNG wire#w2
   RUNG wire#w1
      { S7_Templates := "SrcType := Int" } NE_Contact(in1 := %DB2.DBW16, in2 := 0)
   END_RUNG wire#w2
   RUNG wire#w1
      Contact( "数据接收".手自动状态_1 )
   END_RUNG wire#w2
   RUNG wire#w1
      I_Contact( "数据接收".库位满_2 )
      wire#w4
      Contact( "Clock_2Hz" )
   END_RUNG wire#w3
   RUNG wire#w1
      I_Contact( "数据接收".条码读取状态_2 )
   END_RUNG wire#w4
   // the same network as SCL:
   "14HL16" := "AlwaysTRUE" AND ((("数据发送".机械手报警_1[0] OR "数据发送".机械手报警_1[1] OR "数据发送".机械手报警_1[2] OR "数据发送".机械手报警_1[3] OR "数据发送".机械手报警_1[4] OR "数据发送".机械手报警_1[5] OR "数据发送".机械手报警_1[6] OR "数据发送".机械手报警_1[7] OR "数据发送".机械手报警_1[9] OR "数据发送".机械手报警_1[10] OR "数据发送".机械手报警_1[11] OR (%DB2.DBW16 <> 0) OR "数据接收".手自动状态_1) AND "数据接收".库位满_2 AND "数据接收".条码读取状态_2) OR ((NOT "数据接收".库位满_2 OR NOT "数据接收".条码读取状态_2) AND "Clock_2Hz"));
END_REGION

REGION Network 27: 2号库位绿灯
   RUNG wire#powerrail
      Contact( "AlwaysTRUE" )
      wire#w1
      I_Contact( "14HL16" )
      Contact( "数据接收".库位满_2 )
      wire#w2
      Contact( "数据接收".条码读取状态_2 )
      Coil( "14HL15" )
   END_RUNG
   RUNG wire#w1
      I_Contact( "数据接收".库位满_2 )
      Contact( "Clock_2Hz" )
   END_RUNG wire#w2
   // the same network as SCL:
   "14HL15" := "AlwaysTRUE" AND ((NOT "14HL16" AND "数据接收".库位满_2) OR (NOT "数据接收".库位满_2 AND "Clock_2Hz")) AND "数据接收".条码读取状态_2;
END_REGION

REGION Network 28: 3号库位红灯
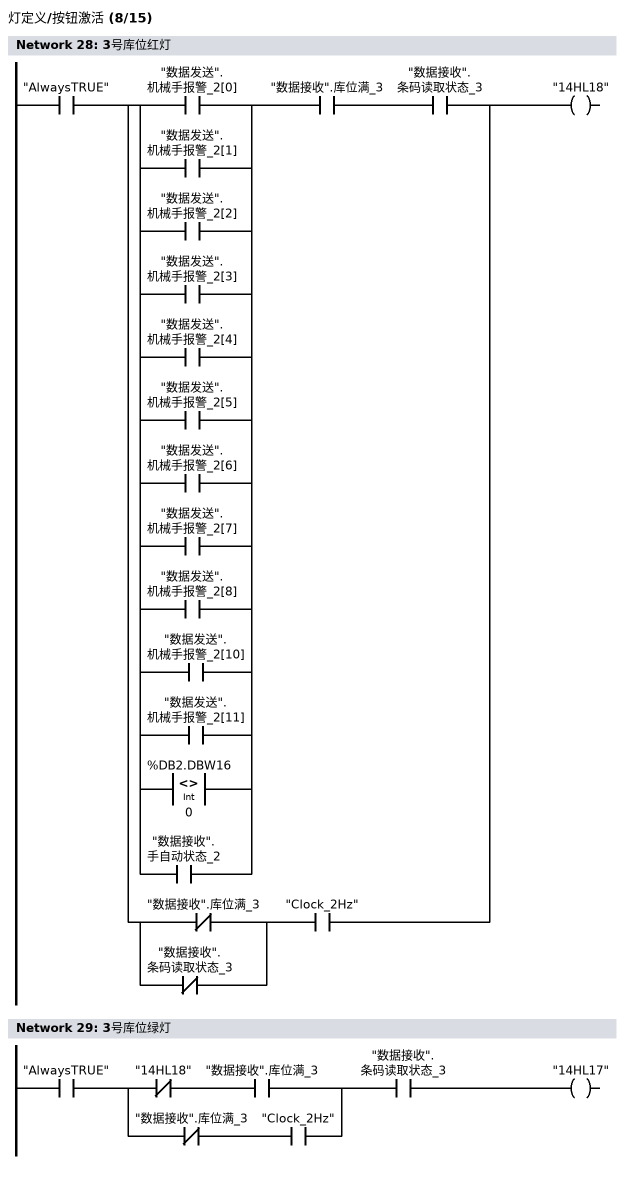
   RUNG wire#powerrail
      Contact( "AlwaysTRUE" )
      wire#w1
      Contact( "数据发送".机械手报警_2[0] )
      wire#w2
      Contact( "数据接收".库位满_3 )
      Contact( "数据接收".条码读取状态_3 )
      wire#w3
      Coil( "14HL18" )
   END_RUNG
   RUNG wire#w1
      Contact( "数据发送".机械手报警_2[1] )
   END_RUNG wire#w2
   RUNG wire#w1
      Contact( "数据发送".机械手报警_2[2] )
   END_RUNG wire#w2
   RUNG wire#w1
      Contact( "数据发送".机械手报警_2[3] )
   END_RUNG wire#w2
   RUNG wire#w1
      Contact( "数据发送".机械手报警_2[4] )
   END_RUNG wire#w2
   RUNG wire#w1
      Contact( "数据发送".机械手报警_2[5] )
   END_RUNG wire#w2
   RUNG wire#w1
      Contact( "数据发送".机械手报警_2[6] )
   END_RUNG wire#w2
   RUNG wire#w1
      Contact( "数据发送".机械手报警_2[7] )
   END_RUNG wire#w2
   RUNG wire#w1
      Contact( "数据发送".机械手报警_2[8] )
   END_RUNG wire#w2
   RUNG wire#w1
      Contact( "数据发送".机械手报警_2[10] )
   END_RUNG wire#w2
   RUNG wire#w1
      Contact( "数据发送".机械手报警_2[11] )
   END_RUNG wire#w2
   RUNG wire#w1
      { S7_Templates := "SrcType := Int" } NE_Contact(in1 := %DB2.DBW16, in2 := 0)
   END_RUNG wire#w2
   RUNG wire#w1
      Contact( "数据接收".手自动状态_2 )
   END_RUNG wire#w2
   RUNG wire#w1
      I_Contact( "数据接收".库位满_3 )
      wire#w4
      Contact( "Clock_2Hz" )
   END_RUNG wire#w3
   RUNG wire#w1
      I_Contact( "数据接收".条码读取状态_3 )
   END_RUNG wire#w4
   // the same network as SCL:
   "14HL18" := "AlwaysTRUE" AND ((("数据发送".机械手报警_2[0] OR "数据发送".机械手报警_2[1] OR "数据发送".机械手报警_2[2] OR "数据发送".机械手报警_2[3] OR "数据发送".机械手报警_2[4] OR "数据发送".机械手报警_2[5] OR "数据发送".机械手报警_2[6] OR "数据发送".机械手报警_2[7] OR "数据发送".机械手报警_2[8] OR "数据发送".机械手报警_2[10] OR "数据发送".机械手报警_2[11] OR (%DB2.DBW16 <> 0) OR "数据接收".手自动状态_2) AND "数据接收".库位满_3 AND "数据接收".条码读取状态_3) OR ((NOT "数据接收".库位满_3 OR NOT "数据接收".条码读取状态_3) AND "Clock_2Hz"));
END_REGION

REGION Network 29: 3号库位绿灯
   RUNG wire#powerrail
      Contact( "AlwaysTRUE" )
      wire#w1
      I_Contact( "14HL18" )
      Contact( "数据接收".库位满_3 )
      wire#w2
      Contact( "数据接收".条码读取状态_3 )
      Coil( "14HL17" )
   END_RUNG
   RUNG wire#w1
      I_Contact( "数据接收".库位满_3 )
      Contact( "Clock_2Hz" )
   END_RUNG wire#w2
   // the same network as SCL:
   "14HL17" := "AlwaysTRUE" AND ((NOT "14HL18" AND "数据接收".库位满_3) OR (NOT "数据接收".库位满_3 AND "Clock_2Hz")) AND "数据接收".条码读取状态_3;
END_REGION

REGION Network 30: 4号库位红灯
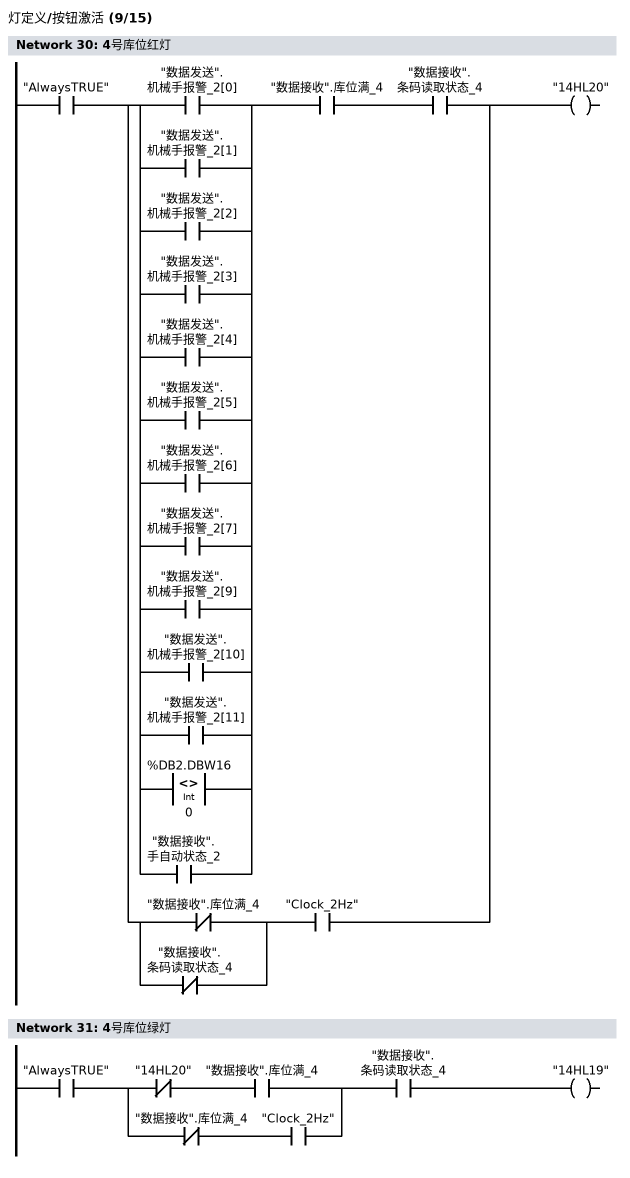
   RUNG wire#powerrail
      Contact( "AlwaysTRUE" )
      wire#w1
      Contact( "数据发送".机械手报警_2[0] )
      wire#w2
      Contact( "数据接收".库位满_4 )
      Contact( "数据接收".条码读取状态_4 )
      wire#w3
      Coil( "14HL20" )
   END_RUNG
   RUNG wire#w1
      Contact( "数据发送".机械手报警_2[1] )
   END_RUNG wire#w2
   RUNG wire#w1
      Contact( "数据发送".机械手报警_2[2] )
   END_RUNG wire#w2
   RUNG wire#w1
      Contact( "数据发送".机械手报警_2[3] )
   END_RUNG wire#w2
   RUNG wire#w1
      Contact( "数据发送".机械手报警_2[4] )
   END_RUNG wire#w2
   RUNG wire#w1
      Contact( "数据发送".机械手报警_2[5] )
   END_RUNG wire#w2
   RUNG wire#w1
      Contact( "数据发送".机械手报警_2[6] )
   END_RUNG wire#w2
   RUNG wire#w1
      Contact( "数据发送".机械手报警_2[7] )
   END_RUNG wire#w2
   RUNG wire#w1
      Contact( "数据发送".机械手报警_2[9] )
   END_RUNG wire#w2
   RUNG wire#w1
      Contact( "数据发送".机械手报警_2[10] )
   END_RUNG wire#w2
   RUNG wire#w1
      Contact( "数据发送".机械手报警_2[11] )
   END_RUNG wire#w2
   RUNG wire#w1
      { S7_Templates := "SrcType := Int" } NE_Contact(in1 := %DB2.DBW16, in2 := 0)
   END_RUNG wire#w2
   RUNG wire#w1
      Contact( "数据接收".手自动状态_2 )
   END_RUNG wire#w2
   RUNG wire#w1
      I_Contact( "数据接收".库位满_4 )
      wire#w4
      Contact( "Clock_2Hz" )
   END_RUNG wire#w3
   RUNG wire#w1
      I_Contact( "数据接收".条码读取状态_4 )
   END_RUNG wire#w4
   // the same network as SCL:
   "14HL20" := "AlwaysTRUE" AND ((("数据发送".机械手报警_2[0] OR "数据发送".机械手报警_2[1] OR "数据发送".机械手报警_2[2] OR "数据发送".机械手报警_2[3] OR "数据发送".机械手报警_2[4] OR "数据发送".机械手报警_2[5] OR "数据发送".机械手报警_2[6] OR "数据发送".机械手报警_2[7] OR "数据发送".机械手报警_2[9] OR "数据发送".机械手报警_2[10] OR "数据发送".机械手报警_2[11] OR (%DB2.DBW16 <> 0) OR "数据接收".手自动状态_2) AND "数据接收".库位满_4 AND "数据接收".条码读取状态_4) OR ((NOT "数据接收".库位满_4 OR NOT "数据接收".条码读取状态_4) AND "Clock_2Hz"));
END_REGION

REGION Network 31: 4号库位绿灯
   RUNG wire#powerrail
      Contact( "AlwaysTRUE" )
      wire#w1
      I_Contact( "14HL20" )
      Contact( "数据接收".库位满_4 )
      wire#w2
      Contact( "数据接收".条码读取状态_4 )
      Coil( "14HL19" )
   END_RUNG
   RUNG wire#w1
      I_Contact( "数据接收".库位满_4 )
      Contact( "Clock_2Hz" )
   END_RUNG wire#w2
   // the same network as SCL:
   "14HL19" := "AlwaysTRUE" AND ((NOT "14HL20" AND "数据接收".库位满_4) OR (NOT "数据接收".库位满_4 AND "Clock_2Hz")) AND "数据接收".条码读取状态_4;
END_REGION

REGION Network 32: 5号库位红灯
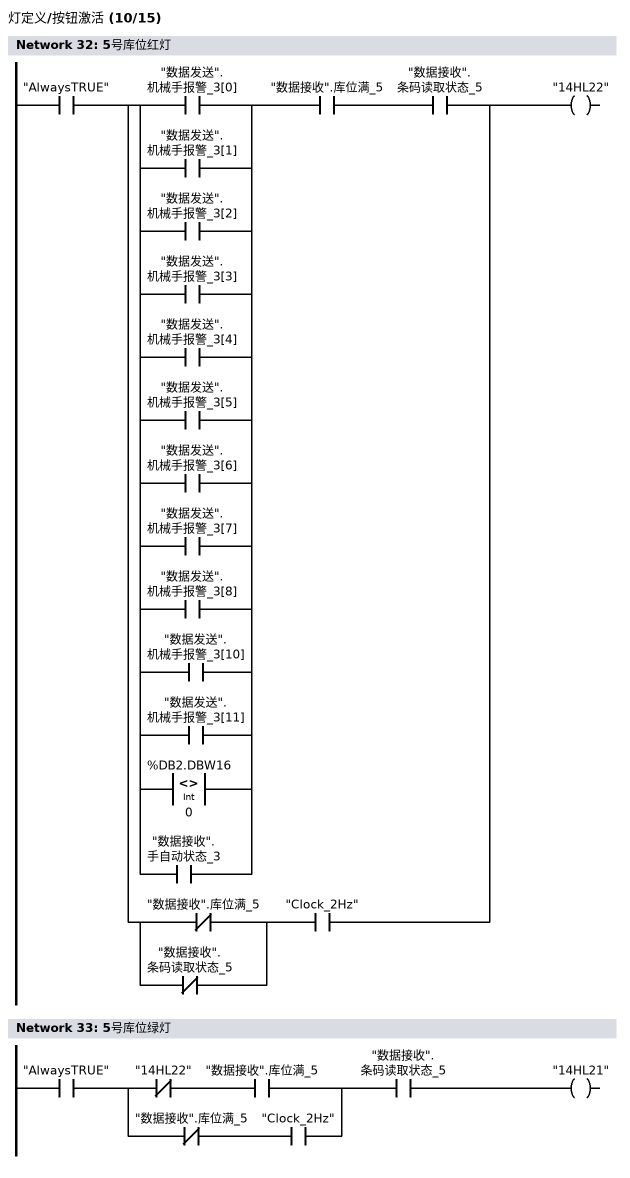
   RUNG wire#powerrail
      Contact( "AlwaysTRUE" )
      wire#w1
      Contact( "数据发送".机械手报警_3[0] )
      wire#w2
      Contact( "数据接收".库位满_5 )
      Contact( "数据接收".条码读取状态_5 )
      wire#w3
      Coil( "14HL22" )
   END_RUNG
   RUNG wire#w1
      Contact( "数据发送".机械手报警_3[1] )
   END_RUNG wire#w2
   RUNG wire#w1
      Contact( "数据发送".机械手报警_3[2] )
   END_RUNG wire#w2
   RUNG wire#w1
      Contact( "数据发送".机械手报警_3[3] )
   END_RUNG wire#w2
   RUNG wire#w1
      Contact( "数据发送".机械手报警_3[4] )
   END_RUNG wire#w2
   RUNG wire#w1
      Contact( "数据发送".机械手报警_3[5] )
   END_RUNG wire#w2
   RUNG wire#w1
      Contact( "数据发送".机械手报警_3[6] )
   END_RUNG wire#w2
   RUNG wire#w1
      Contact( "数据发送".机械手报警_3[7] )
   END_RUNG wire#w2
   RUNG wire#w1
      Contact( "数据发送".机械手报警_3[8] )
   END_RUNG wire#w2
   RUNG wire#w1
      Contact( "数据发送".机械手报警_3[10] )
   END_RUNG wire#w2
   RUNG wire#w1
      Contact( "数据发送".机械手报警_3[11] )
   END_RUNG wire#w2
   RUNG wire#w1
      { S7_Templates := "SrcType := Int" } NE_Contact(in1 := %DB2.DBW16, in2 := 0)
   END_RUNG wire#w2
   RUNG wire#w1
      Contact( "数据接收".手自动状态_3 )
   END_RUNG wire#w2
   RUNG wire#w1
      I_Contact( "数据接收".库位满_5 )
      wire#w4
      Contact( "Clock_2Hz" )
   END_RUNG wire#w3
   RUNG wire#w1
      I_Contact( "数据接收".条码读取状态_5 )
   END_RUNG wire#w4
   // the same network as SCL:
   "14HL22" := "AlwaysTRUE" AND ((("数据发送".机械手报警_3[0] OR "数据发送".机械手报警_3[1] OR "数据发送".机械手报警_3[2] OR "数据发送".机械手报警_3[3] OR "数据发送".机械手报警_3[4] OR "数据发送".机械手报警_3[5] OR "数据发送".机械手报警_3[6] OR "数据发送".机械手报警_3[7] OR "数据发送".机械手报警_3[8] OR "数据发送".机械手报警_3[10] OR "数据发送".机械手报警_3[11] OR (%DB2.DBW16 <> 0) OR "数据接收".手自动状态_3) AND "数据接收".库位满_5 AND "数据接收".条码读取状态_5) OR ((NOT "数据接收".库位满_5 OR NOT "数据接收".条码读取状态_5) AND "Clock_2Hz"));
END_REGION

REGION Network 33: 5号库位绿灯
   RUNG wire#powerrail
      Contact( "AlwaysTRUE" )
      wire#w1
      I_Contact( "14HL22" )
      Contact( "数据接收".库位满_5 )
      wire#w2
      Contact( "数据接收".条码读取状态_5 )
      Coil( "14HL21" )
   END_RUNG
   RUNG wire#w1
      I_Contact( "数据接收".库位满_5 )
      Contact( "Clock_2Hz" )
   END_RUNG wire#w2
   // the same network as SCL:
   "14HL21" := "AlwaysTRUE" AND ((NOT "14HL22" AND "数据接收".库位满_5) OR (NOT "数据接收".库位满_5 AND "Clock_2Hz")) AND "数据接收".条码读取状态_5;
END_REGION

REGION Network 34: 6号库位红灯
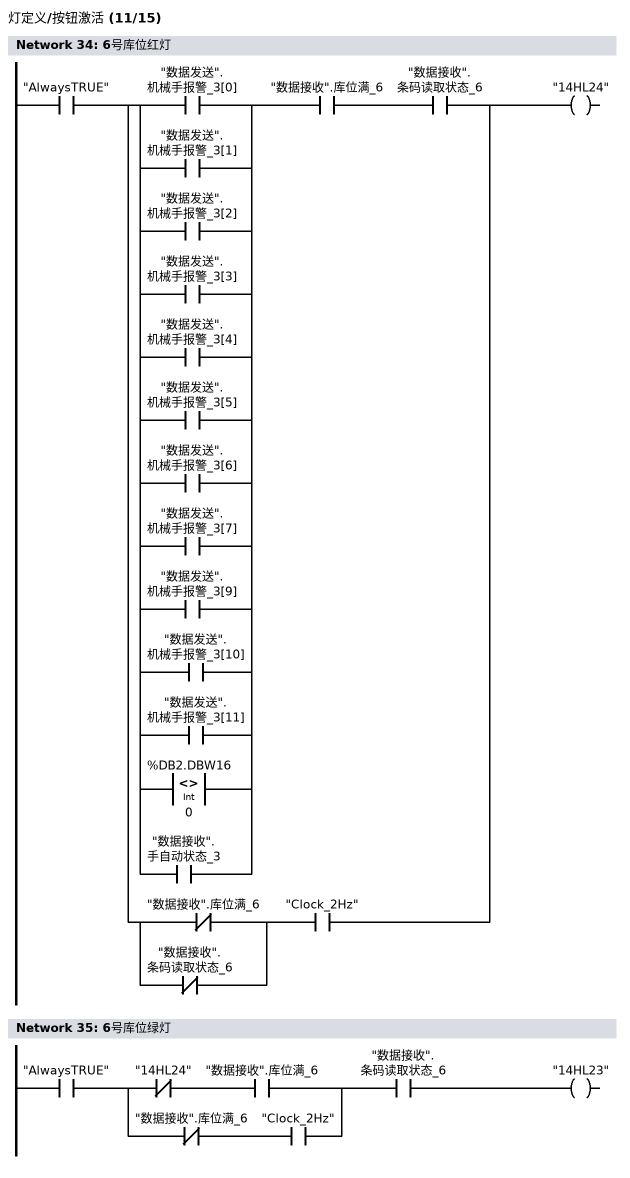
   RUNG wire#powerrail
      Contact( "AlwaysTRUE" )
      wire#w1
      Contact( "数据发送".机械手报警_3[0] )
      wire#w2
      Contact( "数据接收".库位满_6 )
      Contact( "数据接收".条码读取状态_6 )
      wire#w3
      Coil( "14HL24" )
   END_RUNG
   RUNG wire#w1
      Contact( "数据发送".机械手报警_3[1] )
   END_RUNG wire#w2
   RUNG wire#w1
      Contact( "数据发送".机械手报警_3[2] )
   END_RUNG wire#w2
   RUNG wire#w1
      Contact( "数据发送".机械手报警_3[3] )
   END_RUNG wire#w2
   RUNG wire#w1
      Contact( "数据发送".机械手报警_3[4] )
   END_RUNG wire#w2
   RUNG wire#w1
      Contact( "数据发送".机械手报警_3[5] )
   END_RUNG wire#w2
   RUNG wire#w1
      Contact( "数据发送".机械手报警_3[6] )
   END_RUNG wire#w2
   RUNG wire#w1
      Contact( "数据发送".机械手报警_3[7] )
   END_RUNG wire#w2
   RUNG wire#w1
      Contact( "数据发送".机械手报警_3[9] )
   END_RUNG wire#w2
   RUNG wire#w1
      Contact( "数据发送".机械手报警_3[10] )
   END_RUNG wire#w2
   RUNG wire#w1
      Contact( "数据发送".机械手报警_3[11] )
   END_RUNG wire#w2
   RUNG wire#w1
      { S7_Templates := "SrcType := Int" } NE_Contact(in1 := %DB2.DBW16, in2 := 0)
   END_RUNG wire#w2
   RUNG wire#w1
      Contact( "数据接收".手自动状态_3 )
   END_RUNG wire#w2
   RUNG wire#w1
      I_Contact( "数据接收".库位满_6 )
      wire#w4
      Contact( "Clock_2Hz" )
   END_RUNG wire#w3
   RUNG wire#w1
      I_Contact( "数据接收".条码读取状态_6 )
   END_RUNG wire#w4
   // the same network as SCL:
   "14HL24" := "AlwaysTRUE" AND ((("数据发送".机械手报警_3[0] OR "数据发送".机械手报警_3[1] OR "数据发送".机械手报警_3[2] OR "数据发送".机械手报警_3[3] OR "数据发送".机械手报警_3[4] OR "数据发送".机械手报警_3[5] OR "数据发送".机械手报警_3[6] OR "数据发送".机械手报警_3[7] OR "数据发送".机械手报警_3[9] OR "数据发送".机械手报警_3[10] OR "数据发送".机械手报警_3[11] OR (%DB2.DBW16 <> 0) OR "数据接收".手自动状态_3) AND "数据接收".库位满_6 AND "数据接收".条码读取状态_6) OR ((NOT "数据接收".库位满_6 OR NOT "数据接收".条码读取状态_6) AND "Clock_2Hz"));
END_REGION

REGION Network 35: 6号库位绿灯
   RUNG wire#powerrail
      Contact( "AlwaysTRUE" )
      wire#w1
      I_Contact( "14HL24" )
      Contact( "数据接收".库位满_6 )
      wire#w2
      Contact( "数据接收".条码读取状态_6 )
      Coil( "14HL23" )
   END_RUNG
   RUNG wire#w1
      I_Contact( "数据接收".库位满_6 )
      Contact( "Clock_2Hz" )
   END_RUNG wire#w2
   // the same network as SCL:
   "14HL23" := "AlwaysTRUE" AND ((NOT "14HL24" AND "数据接收".库位满_6) OR (NOT "数据接收".库位满_6 AND "Clock_2Hz")) AND "数据接收".条码读取状态_6;
END_REGION

REGION Network 36: 7号库位红灯
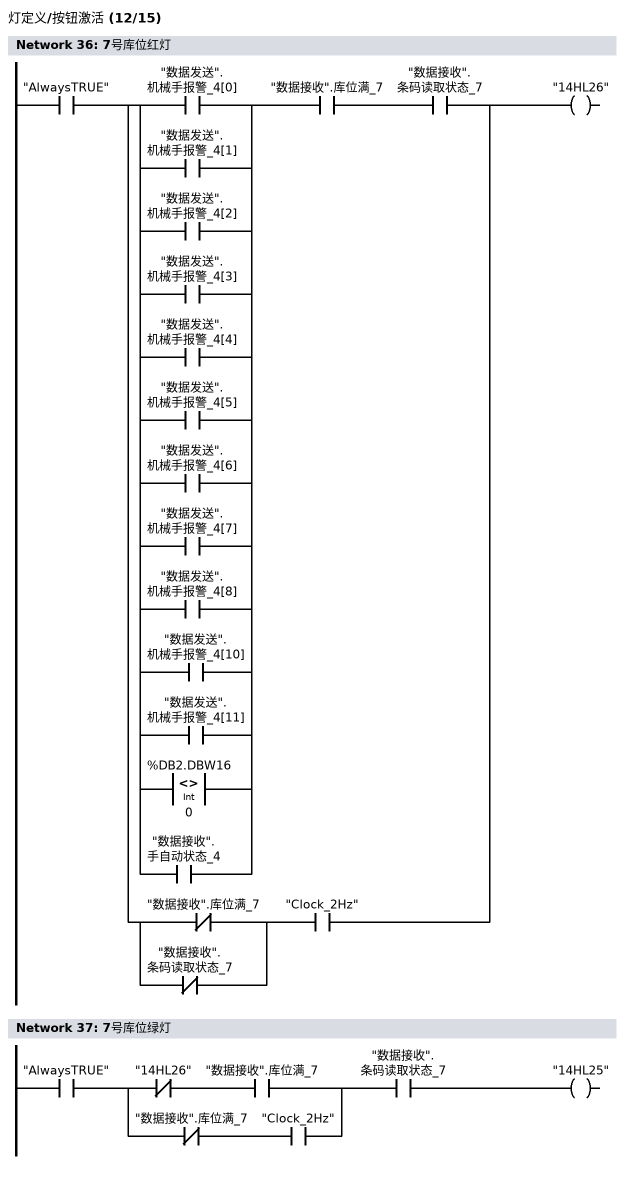
   RUNG wire#powerrail
      Contact( "AlwaysTRUE" )
      wire#w1
      Contact( "数据发送".机械手报警_4[0] )
      wire#w2
      Contact( "数据接收".库位满_7 )
      Contact( "数据接收".条码读取状态_7 )
      wire#w3
      Coil( "14HL26" )
   END_RUNG
   RUNG wire#w1
      Contact( "数据发送".机械手报警_4[1] )
   END_RUNG wire#w2
   RUNG wire#w1
      Contact( "数据发送".机械手报警_4[2] )
   END_RUNG wire#w2
   RUNG wire#w1
      Contact( "数据发送".机械手报警_4[3] )
   END_RUNG wire#w2
   RUNG wire#w1
      Contact( "数据发送".机械手报警_4[4] )
   END_RUNG wire#w2
   RUNG wire#w1
      Contact( "数据发送".机械手报警_4[5] )
   END_RUNG wire#w2
   RUNG wire#w1
      Contact( "数据发送".机械手报警_4[6] )
   END_RUNG wire#w2
   RUNG wire#w1
      Contact( "数据发送".机械手报警_4[7] )
   END_RUNG wire#w2
   RUNG wire#w1
      Contact( "数据发送".机械手报警_4[8] )
   END_RUNG wire#w2
   RUNG wire#w1
      Contact( "数据发送".机械手报警_4[10] )
   END_RUNG wire#w2
   RUNG wire#w1
      Contact( "数据发送".机械手报警_4[11] )
   END_RUNG wire#w2
   RUNG wire#w1
      { S7_Templates := "SrcType := Int" } NE_Contact(in1 := %DB2.DBW16, in2 := 0)
   END_RUNG wire#w2
   RUNG wire#w1
      Contact( "数据接收".手自动状态_4 )
   END_RUNG wire#w2
   RUNG wire#w1
      I_Contact( "数据接收".库位满_7 )
      wire#w4
      Contact( "Clock_2Hz" )
   END_RUNG wire#w3
   RUNG wire#w1
      I_Contact( "数据接收".条码读取状态_7 )
   END_RUNG wire#w4
   // the same network as SCL:
   "14HL26" := "AlwaysTRUE" AND ((("数据发送".机械手报警_4[0] OR "数据发送".机械手报警_4[1] OR "数据发送".机械手报警_4[2] OR "数据发送".机械手报警_4[3] OR "数据发送".机械手报警_4[4] OR "数据发送".机械手报警_4[5] OR "数据发送".机械手报警_4[6] OR "数据发送".机械手报警_4[7] OR "数据发送".机械手报警_4[8] OR "数据发送".机械手报警_4[10] OR "数据发送".机械手报警_4[11] OR (%DB2.DBW16 <> 0) OR "数据接收".手自动状态_4) AND "数据接收".库位满_7 AND "数据接收".条码读取状态_7) OR ((NOT "数据接收".库位满_7 OR NOT "数据接收".条码读取状态_7) AND "Clock_2Hz"));
END_REGION

REGION Network 37: 7号库位绿灯
   RUNG wire#powerrail
      Contact( "AlwaysTRUE" )
      wire#w1
      I_Contact( "14HL26" )
      Contact( "数据接收".库位满_7 )
      wire#w2
      Contact( "数据接收".条码读取状态_7 )
      Coil( "14HL25" )
   END_RUNG
   RUNG wire#w1
      I_Contact( "数据接收".库位满_7 )
      Contact( "Clock_2Hz" )
   END_RUNG wire#w2
   // the same network as SCL:
   "14HL25" := "AlwaysTRUE" AND ((NOT "14HL26" AND "数据接收".库位满_7) OR (NOT "数据接收".库位满_7 AND "Clock_2Hz")) AND "数据接收".条码读取状态_7;
END_REGION

REGION Network 38: 8号库位红灯
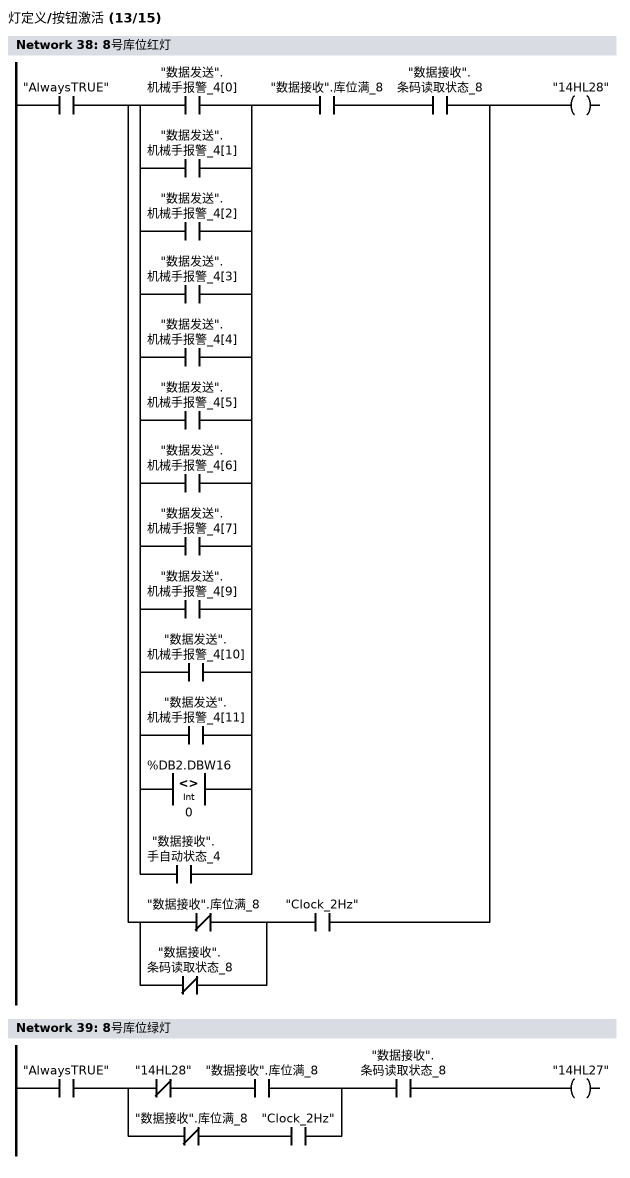
   RUNG wire#powerrail
      Contact( "AlwaysTRUE" )
      wire#w1
      Contact( "数据发送".机械手报警_4[0] )
      wire#w2
      Contact( "数据接收".库位满_8 )
      Contact( "数据接收".条码读取状态_8 )
      wire#w3
      Coil( "14HL28" )
   END_RUNG
   RUNG wire#w1
      Contact( "数据发送".机械手报警_4[1] )
   END_RUNG wire#w2
   RUNG wire#w1
      Contact( "数据发送".机械手报警_4[2] )
   END_RUNG wire#w2
   RUNG wire#w1
      Contact( "数据发送".机械手报警_4[3] )
   END_RUNG wire#w2
   RUNG wire#w1
      Contact( "数据发送".机械手报警_4[4] )
   END_RUNG wire#w2
   RUNG wire#w1
      Contact( "数据发送".机械手报警_4[5] )
   END_RUNG wire#w2
   RUNG wire#w1
      Contact( "数据发送".机械手报警_4[6] )
   END_RUNG wire#w2
   RUNG wire#w1
      Contact( "数据发送".机械手报警_4[7] )
   END_RUNG wire#w2
   RUNG wire#w1
      Contact( "数据发送".机械手报警_4[9] )
   END_RUNG wire#w2
   RUNG wire#w1
      Contact( "数据发送".机械手报警_4[10] )
   END_RUNG wire#w2
   RUNG wire#w1
      Contact( "数据发送".机械手报警_4[11] )
   END_RUNG wire#w2
   RUNG wire#w1
      { S7_Templates := "SrcType := Int" } NE_Contact(in1 := %DB2.DBW16, in2 := 0)
   END_RUNG wire#w2
   RUNG wire#w1
      Contact( "数据接收".手自动状态_4 )
   END_RUNG wire#w2
   RUNG wire#w1
      I_Contact( "数据接收".库位满_8 )
      wire#w4
      Contact( "Clock_2Hz" )
   END_RUNG wire#w3
   RUNG wire#w1
      I_Contact( "数据接收".条码读取状态_8 )
   END_RUNG wire#w4
   // the same network as SCL:
   "14HL28" := "AlwaysTRUE" AND ((("数据发送".机械手报警_4[0] OR "数据发送".机械手报警_4[1] OR "数据发送".机械手报警_4[2] OR "数据发送".机械手报警_4[3] OR "数据发送".机械手报警_4[4] OR "数据发送".机械手报警_4[5] OR "数据发送".机械手报警_4[6] OR "数据发送".机械手报警_4[7] OR "数据发送".机械手报警_4[9] OR "数据发送".机械手报警_4[10] OR "数据发送".机械手报警_4[11] OR (%DB2.DBW16 <> 0) OR "数据接收".手自动状态_4) AND "数据接收".库位满_8 AND "数据接收".条码读取状态_8) OR ((NOT "数据接收".库位满_8 OR NOT "数据接收".条码读取状态_8) AND "Clock_2Hz"));
END_REGION

REGION Network 39: 8号库位绿灯
   RUNG wire#powerrail
      Contact( "AlwaysTRUE" )
      wire#w1
      I_Contact( "14HL28" )
      Contact( "数据接收".库位满_8 )
      wire#w2
      Contact( "数据接收".条码读取状态_8 )
      Coil( "14HL27" )
   END_RUNG
   RUNG wire#w1
      I_Contact( "数据接收".库位满_8 )
      Contact( "Clock_2Hz" )
   END_RUNG wire#w2
   // the same network as SCL:
   "14HL27" := "AlwaysTRUE" AND ((NOT "14HL28" AND "数据接收".库位满_8) OR (NOT "数据接收".库位满_8 AND "Clock_2Hz")) AND "数据接收".条码读取状态_8;
END_REGION

REGION Network 40: 9号库位红灯
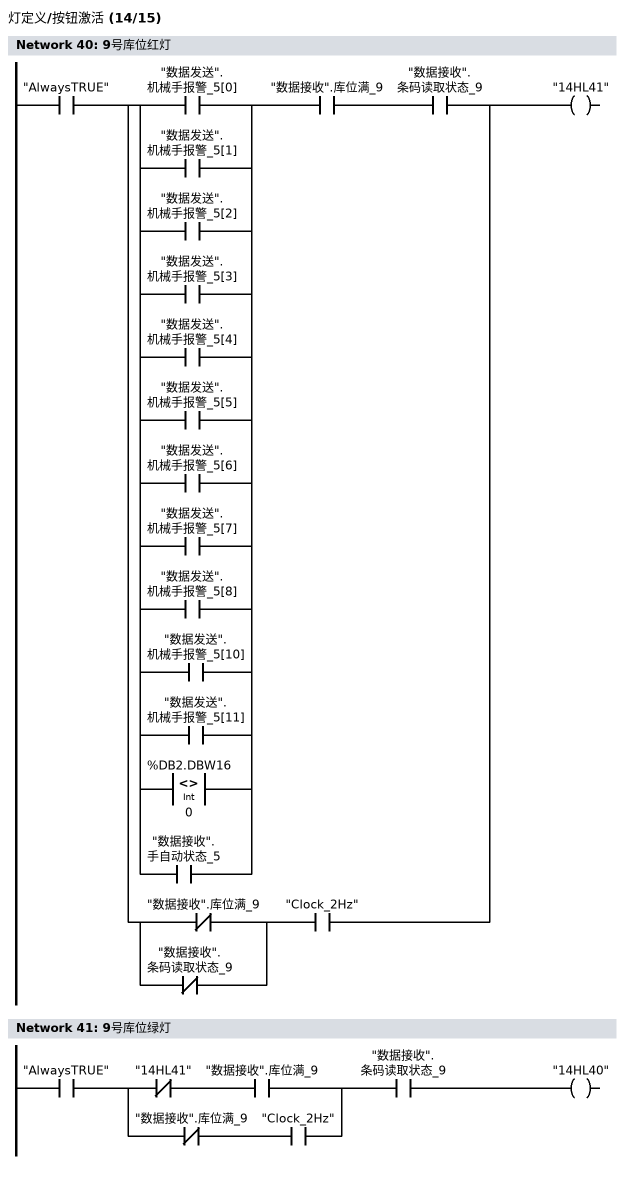
   RUNG wire#powerrail
      Contact( "AlwaysTRUE" )
      wire#w1
      Contact( "数据发送".机械手报警_5[0] )
      wire#w2
      Contact( "数据接收".库位满_9 )
      Contact( "数据接收".条码读取状态_9 )
      wire#w3
      Coil( "14HL41" )
   END_RUNG
   RUNG wire#w1
      Contact( "数据发送".机械手报警_5[1] )
   END_RUNG wire#w2
   RUNG wire#w1
      Contact( "数据发送".机械手报警_5[2] )
   END_RUNG wire#w2
   RUNG wire#w1
      Contact( "数据发送".机械手报警_5[3] )
   END_RUNG wire#w2
   RUNG wire#w1
      Contact( "数据发送".机械手报警_5[4] )
   END_RUNG wire#w2
   RUNG wire#w1
      Contact( "数据发送".机械手报警_5[5] )
   END_RUNG wire#w2
   RUNG wire#w1
      Contact( "数据发送".机械手报警_5[6] )
   END_RUNG wire#w2
   RUNG wire#w1
      Contact( "数据发送".机械手报警_5[7] )
   END_RUNG wire#w2
   RUNG wire#w1
      Contact( "数据发送".机械手报警_5[8] )
   END_RUNG wire#w2
   RUNG wire#w1
      Contact( "数据发送".机械手报警_5[10] )
   END_RUNG wire#w2
   RUNG wire#w1
      Contact( "数据发送".机械手报警_5[11] )
   END_RUNG wire#w2
   RUNG wire#w1
      { S7_Templates := "SrcType := Int" } NE_Contact(in1 := %DB2.DBW16, in2 := 0)
   END_RUNG wire#w2
   RUNG wire#w1
      Contact( "数据接收".手自动状态_5 )
   END_RUNG wire#w2
   RUNG wire#w1
      I_Contact( "数据接收".库位满_9 )
      wire#w4
      Contact( "Clock_2Hz" )
   END_RUNG wire#w3
   RUNG wire#w1
      I_Contact( "数据接收".条码读取状态_9 )
   END_RUNG wire#w4
   // the same network as SCL:
   "14HL41" := "AlwaysTRUE" AND ((("数据发送".机械手报警_5[0] OR "数据发送".机械手报警_5[1] OR "数据发送".机械手报警_5[2] OR "数据发送".机械手报警_5[3] OR "数据发送".机械手报警_5[4] OR "数据发送".机械手报警_5[5] OR "数据发送".机械手报警_5[6] OR "数据发送".机械手报警_5[7] OR "数据发送".机械手报警_5[8] OR "数据发送".机械手报警_5[10] OR "数据发送".机械手报警_5[11] OR (%DB2.DBW16 <> 0) OR "数据接收".手自动状态_5) AND "数据接收".库位满_9 AND "数据接收".条码读取状态_9) OR ((NOT "数据接收".库位满_9 OR NOT "数据接收".条码读取状态_9) AND "Clock_2Hz"));
END_REGION

REGION Network 41: 9号库位绿灯
   RUNG wire#powerrail
      Contact( "AlwaysTRUE" )
      wire#w1
      I_Contact( "14HL41" )
      Contact( "数据接收".库位满_9 )
      wire#w2
      Contact( "数据接收".条码读取状态_9 )
      Coil( "14HL40" )
   END_RUNG
   RUNG wire#w1
      I_Contact( "数据接收".库位满_9 )
      Contact( "Clock_2Hz" )
   END_RUNG wire#w2
   // the same network as SCL:
   "14HL40" := "AlwaysTRUE" AND ((NOT "14HL41" AND "数据接收".库位满_9) OR (NOT "数据接收".库位满_9 AND "Clock_2Hz")) AND "数据接收".条码读取状态_9;
END_REGION

REGION Network 42: 10号库位红灯
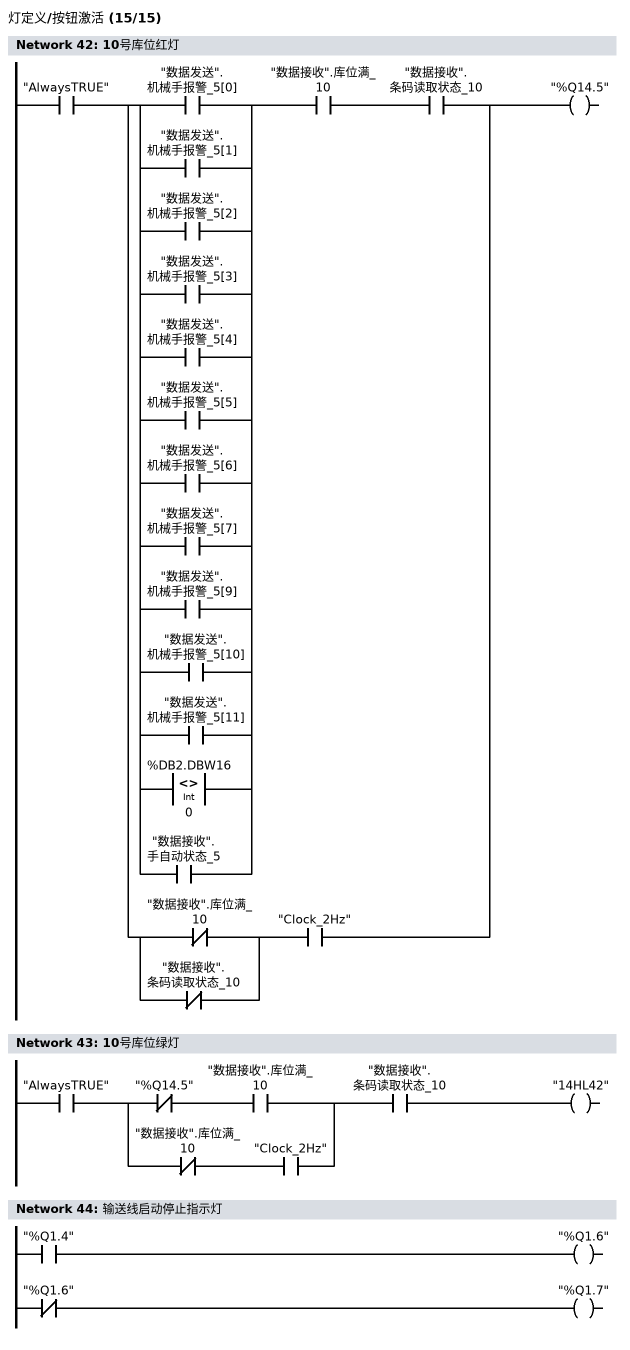
   RUNG wire#powerrail
      Contact( "AlwaysTRUE" )
      wire#w1
      Contact( "数据发送".机械手报警_5[0] )
      wire#w2
      Contact( "数据接收".库位满_10 )
      Contact( "数据接收".条码读取状态_10 )
      wire#w3
      Coil( "%Q14.5" )
   END_RUNG
   RUNG wire#w1
      Contact( "数据发送".机械手报警_5[1] )
   END_RUNG wire#w2
   RUNG wire#w1
      Contact( "数据发送".机械手报警_5[2] )
   END_RUNG wire#w2
   RUNG wire#w1
      Contact( "数据发送".机械手报警_5[3] )
   END_RUNG wire#w2
   RUNG wire#w1
      Contact( "数据发送".机械手报警_5[4] )
   END_RUNG wire#w2
   RUNG wire#w1
      Contact( "数据发送".机械手报警_5[5] )
   END_RUNG wire#w2
   RUNG wire#w1
      Contact( "数据发送".机械手报警_5[6] )
   END_RUNG wire#w2
   RUNG wire#w1
      Contact( "数据发送".机械手报警_5[7] )
   END_RUNG wire#w2
   RUNG wire#w1
      Contact( "数据发送".机械手报警_5[9] )
   END_RUNG wire#w2
   RUNG wire#w1
      Contact( "数据发送".机械手报警_5[10] )
   END_RUNG wire#w2
   RUNG wire#w1
      Contact( "数据发送".机械手报警_5[11] )
   END_RUNG wire#w2
   RUNG wire#w1
      { S7_Templates := "SrcType := Int" } NE_Contact(in1 := %DB2.DBW16, in2 := 0)
   END_RUNG wire#w2
   RUNG wire#w1
      Contact( "数据接收".手自动状态_5 )
   END_RUNG wire#w2
   RUNG wire#w1
      I_Contact( "数据接收".库位满_10 )
      wire#w4
      Contact( "Clock_2Hz" )
   END_RUNG wire#w3
   RUNG wire#w1
      I_Contact( "数据接收".条码读取状态_10 )
   END_RUNG wire#w4
   // the same network as SCL:
   "%Q14.5" := "AlwaysTRUE" AND ((("数据发送".机械手报警_5[0] OR "数据发送".机械手报警_5[1] OR "数据发送".机械手报警_5[2] OR "数据发送".机械手报警_5[3] OR "数据发送".机械手报警_5[4] OR "数据发送".机械手报警_5[5] OR "数据发送".机械手报警_5[6] OR "数据发送".机械手报警_5[7] OR "数据发送".机械手报警_5[9] OR "数据发送".机械手报警_5[10] OR "数据发送".机械手报警_5[11] OR (%DB2.DBW16 <> 0) OR "数据接收".手自动状态_5) AND "数据接收".库位满_10 AND "数据接收".条码读取状态_10) OR ((NOT "数据接收".库位满_10 OR NOT "数据接收".条码读取状态_10) AND "Clock_2Hz"));
END_REGION

REGION Network 43: 10号库位绿灯
   RUNG wire#powerrail
      Contact( "AlwaysTRUE" )
      wire#w1
      I_Contact( "%Q14.5" )
      Contact( "数据接收".库位满_10 )
      wire#w2
      Contact( "数据接收".条码读取状态_10 )
      Coil( "14HL42" )
   END_RUNG
   RUNG wire#w1
      I_Contact( "数据接收".库位满_10 )
      Contact( "Clock_2Hz" )
   END_RUNG wire#w2
   // the same network as SCL:
   "14HL42" := "AlwaysTRUE" AND ((NOT "%Q14.5" AND "数据接收".库位满_10) OR (NOT "数据接收".库位满_10 AND "Clock_2Hz")) AND "数据接收".条码读取状态_10;
END_REGION

REGION Network 44: 输送线启动停止指示灯
   RUNG wire#powerrail
      Contact( "%Q1.4" )
      Coil( "%Q1.6" )
   END_RUNG
   RUNG wire#powerrail
      I_Contact( "%Q1.6" )
      Coil( "%Q1.7" )
   END_RUNG
   // the same network as SCL:
   "%Q1.6" := "%Q1.4";
   "%Q1.7" := NOT "%Q1.6";
END_REGION
END_FUNCTION

FUNCTION "5#手" : Void   // FC19, LAD
{ S7_Optimized_Access := 'TRUE' }
VERSION : 0.1
   VAR_TEMP   // added for the SCL form of the ladder/FBD networks
      _w1 : Bool;
   END_VAR
BEGIN

REGION Network 1: 5#机械手库位动作流程
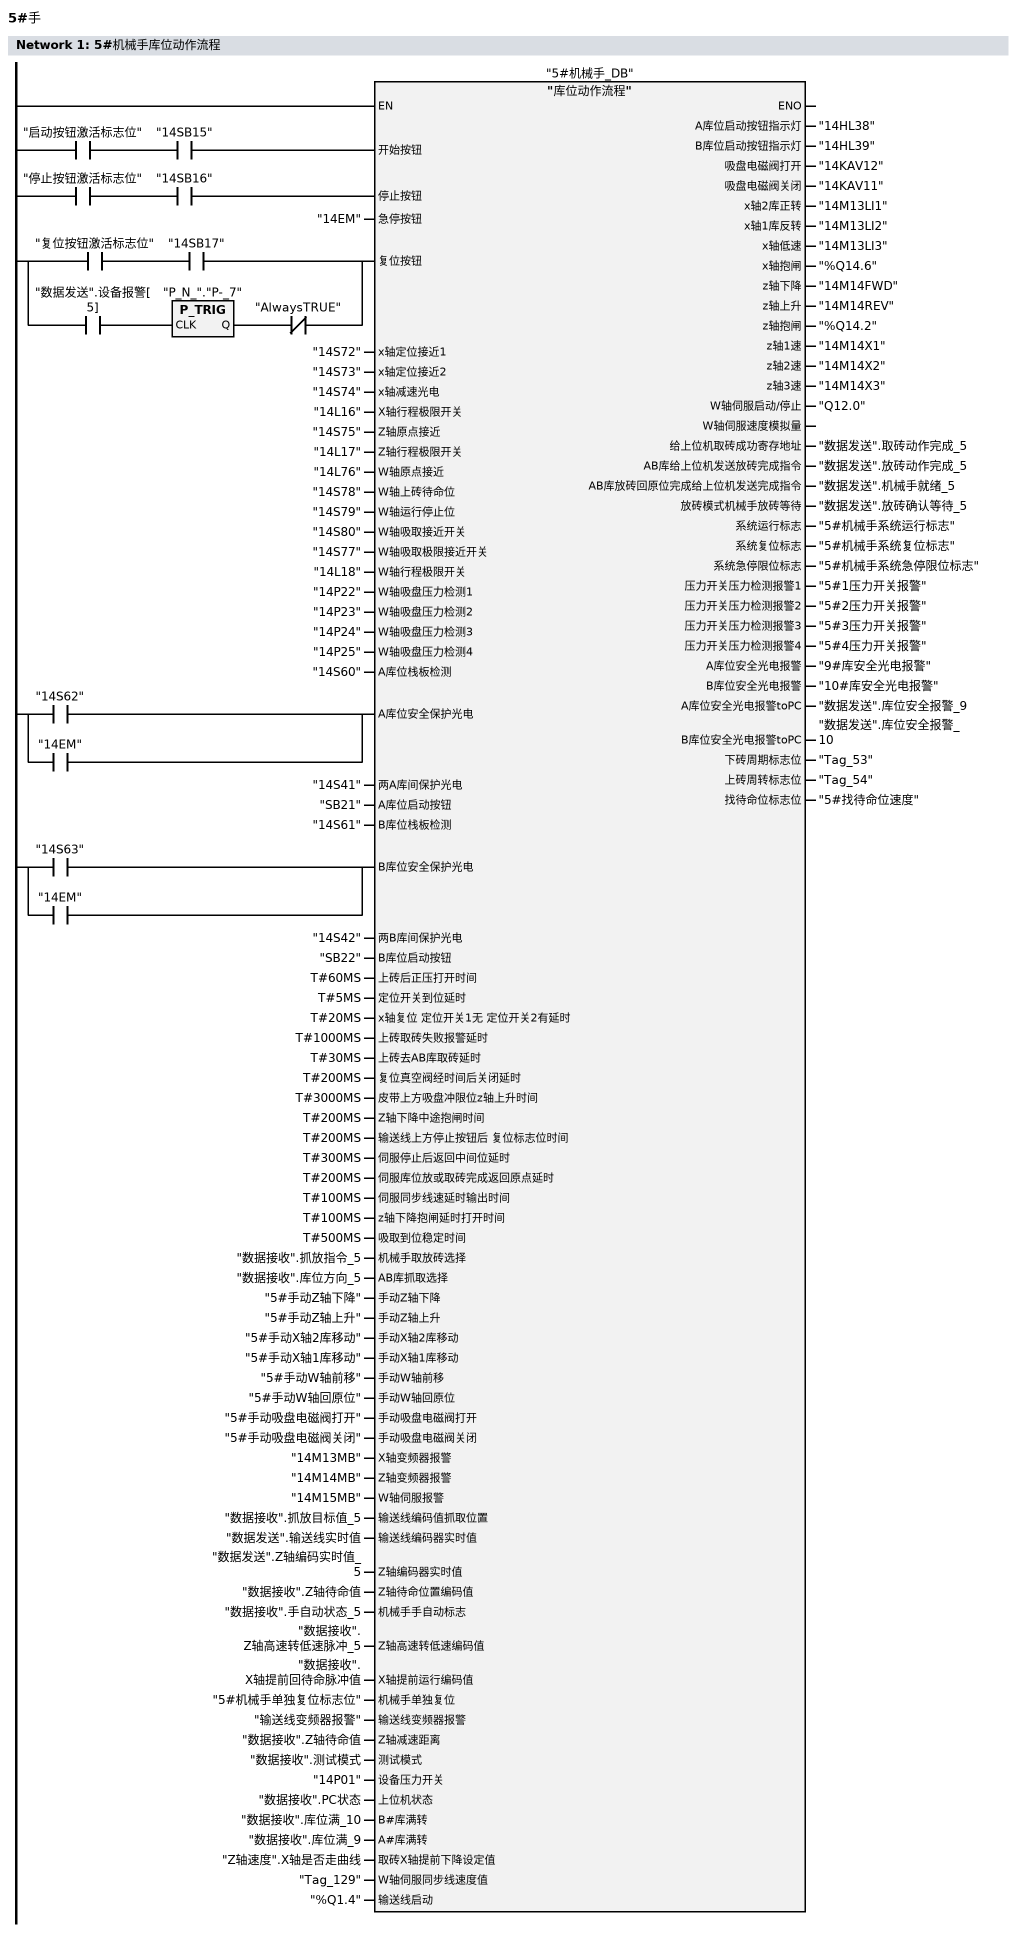
   RUNG wire#powerrail
      "5#机械手_DB"(开始按钮 := wire#w1, 停止按钮 := wire#w2, 复位按钮 := wire#w3, A库位安全保护光电 := wire#w4, B库位安全保护光电 := wire#w5, 急停按钮 := "14EM", x轴定位接近1 := "14S72", x轴定位接近2 := "14S73", x轴减速光电 := "14S74", X轴行程极限开关 := "14L16", Z轴原点接近 := "14S75", Z轴行程极限开关 := "14L17", W轴原点接近 := "14L76", W轴上砖待命位 := "14S78", W轴运行停止位 := "14S79", W轴吸取接近开关 := "14S80", W轴吸取极限接近开关 := "14S77", W轴行程极限开关 := "14L18", W轴吸盘压力检测1 := "14P22", W轴吸盘压力检测2 := "14P23", W轴吸盘压力检测3 := "14P24", W轴吸盘压力检测4 := "14P25", A库位栈板检测 := "14S60", 两A库间保护光电 := "14S41", A库位启动按钮 := "SB21", B库位栈板检测 := "14S61", 两B库间保护光电 := "14S42", B库位启动按钮 := "SB22", 上砖后正压打开时间 := T#60MS, 定位开关到位延时 := T#5MS, "x轴复位 定位开关1无 定位开关2有延时" := T#20MS, 上砖取砖失败报警延时 := T#1000MS, 上砖去AB库取砖延时 := T#30MS, 复位真空阀经时间后关闭延时 := T#200MS, 皮带上方吸盘冲限位z轴上升时间 := T#3000MS, Z轴下降中途抱闸时间 := T#200MS, "输送线上方停止按钮后 复位标志位时间" := T#200MS, 伺服停止后返回中间位延时 := T#300MS, 伺服库位放或取砖完成返回原点延时 := T#200MS, 伺服同步线速延时输出时间 := T#100MS, z轴下降抱闸延时打开时间 := T#100MS, 吸取到位稳定时间 := T#500MS, 机械手取放砖选择 := "数据接收".抓放指令_5, AB库抓取选择 := "数据接收".库位方向_5, 手动Z轴下降 := "5#手动Z轴下降", 手动Z轴上升 := "5#手动Z轴上升", 手动X轴2库移动 := "5#手动X轴2库移动", 手动X轴1库移动 := "5#手动X轴1库移动", 手动W轴前移 := "5#手动W轴前移", 手动W轴回原位 := "5#手动W轴回原位", 手动吸盘电磁阀打开 := "5#手动吸盘电磁阀打开", 手动吸盘电磁阀关闭 := "5#手动吸盘电磁阀关闭", X轴变频器报警 := "14M13MB", Z轴变频器报警 := "14M14MB", W轴伺服报警 := "14M15MB", 输送线编码值抓取位置 := "数据接收".抓放目标值_5, 输送线编码器实时值 := "数据发送".输送线实时值, Z轴编码器实时值 := "数据发送".Z轴编码实时值_5, Z轴待命位置编码值 := "数据接收".Z轴待命值, 机械手手自动标志 := "数据接收".手自动状态_5, Z轴高速转低速编码值 := "数据接收".Z轴高速转低速脉冲_5, X轴提前运行编码值 := "数据接收".X轴提前回待命脉冲值, 机械手单独复位 := "5#机械手单独复位标志位", 输送线变频器报警 := "输送线变频器报警", Z轴减速距离 := "数据接收".Z轴待命值, 测试模式 := "数据接收".测试模式, 设备压力开关 := "14P01", 上位机状态 := "数据接收".PC状态, "B#库满转" := "数据接收".库位满_10, "A#库满转" := "数据接收".库位满_9, 取砖X轴提前下降设定值 := "Z轴速度".X轴是否走曲线, W轴伺服同步线速度值 := "Tag_129", 输送线启动 := "%Q1.4", A库位启动按钮指示灯 => "14HL38", B库位启动按钮指示灯 => "14HL39", 吸盘电磁阀打开 => "14KAV12", 吸盘电磁阀关闭 => "14KAV11", x轴2库正转 => "14M13LI1", x轴1库反转 => "14M13LI2", x轴低速 => "14M13LI3", x轴抱闸 => "%Q14.6", z轴下降 => "14M14FWD", z轴上升 => "14M14REV", z轴抱闸 => "%Q14.2", z轴1速 => "14M14X1", z轴2速 => "14M14X2", z轴3速 => "14M14X3", "W轴伺服启动/停止" => "Q12.0", W轴伺服速度模拟量 =>, 给上位机取砖成功寄存地址 => "数据发送".取砖动作完成_5, AB库给上位机发送放砖完成指令 => "数据发送".放砖动作完成_5, AB库放砖回原位完成给上位机发送完成指令 => "数据发送".机械手就绪_5, 放砖模式机械手放砖等待 => "数据发送".放砖确认等待_5, 系统运行标志 => "5#机械手系统运行标志", 系统复位标志 => "5#机械手系统复位标志", 系统急停限位标志 => "5#机械手系统急停限位标志", 压力开关压力检测报警1 => "5#1压力开关报警", 压力开关压力检测报警2 => "5#2压力开关报警", 压力开关压力检测报警3 => "5#3压力开关报警", 压力开关压力检测报警4 => "5#4压力开关报警", A库位安全光电报警 => "9#库安全光电报警", B库位安全光电报警 => "10#库安全光电报警", A库位安全光电报警toPC => "数据发送".库位安全报警_9, B库位安全光电报警toPC => "数据发送".库位安全报警_10, 下砖周期标志位 => "Tag_53", 上砖周转标志位 => "Tag_54", 找待命位标志位 => "5#找待命位速度")
   END_RUNG
   RUNG wire#powerrail
      Contact( "启动按钮激活标志位" )
      Contact( "14SB15" )
   END_RUNG wire#w1
   RUNG wire#powerrail
      Contact( "停止按钮激活标志位" )
      Contact( "14SB16" )
   END_RUNG wire#w2
   RUNG wire#powerrail
      Contact( "复位按钮激活标志位" )
      Contact( "14SB17" )
   END_RUNG wire#w3
   RUNG wire#powerrail
      Contact( "数据发送".设备报警[5] )
      P_Trig( "P_N_"."P-_7" )
      I_Contact( "AlwaysTRUE" )
   END_RUNG wire#w3
   RUNG wire#powerrail
      Contact( "14S62" )
   END_RUNG wire#w4
   RUNG wire#powerrail
      Contact( "14EM" )
   END_RUNG wire#w4
   RUNG wire#powerrail
      Contact( "14S63" )
   END_RUNG wire#w5
   RUNG wire#powerrail
      Contact( "14EM" )
   END_RUNG wire#w5
   // the same network as SCL:
   #_w1 := "数据发送".设备报警[5] AND NOT "P_N_"."P-_7";   // rising edge
   "P_N_"."P-_7" := "数据发送".设备报警[5];
   "5#机械手_DB"(开始按钮 := "启动按钮激活标志位" AND "14SB15",   // "库位动作流程"
              停止按钮 := "停止按钮激活标志位" AND "14SB16",
              急停按钮 := "14EM",
              复位按钮 := ("复位按钮激活标志位" AND "14SB17") OR (#_w1 AND NOT "AlwaysTRUE"),
              x轴定位接近1 := "14S72",
              x轴定位接近2 := "14S73",
              x轴减速光电 := "14S74",
              X轴行程极限开关 := "14L16",
              Z轴原点接近 := "14S75",
              Z轴行程极限开关 := "14L17",
              W轴原点接近 := "14L76",
              W轴上砖待命位 := "14S78",
              W轴运行停止位 := "14S79",
              W轴吸取接近开关 := "14S80",
              W轴吸取极限接近开关 := "14S77",
              W轴行程极限开关 := "14L18",
              W轴吸盘压力检测1 := "14P22",
              W轴吸盘压力检测2 := "14P23",
              W轴吸盘压力检测3 := "14P24",
              W轴吸盘压力检测4 := "14P25",
              A库位栈板检测 := "14S60",
              A库位安全保护光电 := "14S62" OR "14EM",
              两A库间保护光电 := "14S41",
              A库位启动按钮 := "SB21",
              B库位栈板检测 := "14S61",
              B库位安全保护光电 := "14S63" OR "14EM",
              两B库间保护光电 := "14S42",
              B库位启动按钮 := "SB22",
              上砖后正压打开时间 := T#60MS,
              定位开关到位延时 := T#5MS,
              "x轴复位 定位开关1无 定位开关2有延时" := T#20MS,
              上砖取砖失败报警延时 := T#1000MS,
              上砖去AB库取砖延时 := T#30MS,
              复位真空阀经时间后关闭延时 := T#200MS,
              皮带上方吸盘冲限位z轴上升时间 := T#3000MS,
              Z轴下降中途抱闸时间 := T#200MS,
              "输送线上方停止按钮后 复位标志位时间" := T#200MS,
              伺服停止后返回中间位延时 := T#300MS,
              伺服库位放或取砖完成返回原点延时 := T#200MS,
              伺服同步线速延时输出时间 := T#100MS,
              z轴下降抱闸延时打开时间 := T#100MS,
              吸取到位稳定时间 := T#500MS,
              机械手取放砖选择 := "数据接收".抓放指令_5,
              AB库抓取选择 := "数据接收".库位方向_5,
              手动Z轴下降 := "5#手动Z轴下降",
              手动Z轴上升 := "5#手动Z轴上升",
              手动X轴2库移动 := "5#手动X轴2库移动",
              手动X轴1库移动 := "5#手动X轴1库移动",
              手动W轴前移 := "5#手动W轴前移",
              手动W轴回原位 := "5#手动W轴回原位",
              手动吸盘电磁阀打开 := "5#手动吸盘电磁阀打开",
              手动吸盘电磁阀关闭 := "5#手动吸盘电磁阀关闭",
              X轴变频器报警 := "14M13MB",
              Z轴变频器报警 := "14M14MB",
              W轴伺服报警 := "14M15MB",
              输送线编码值抓取位置 := "数据接收".抓放目标值_5,
              输送线编码器实时值 := "数据发送".输送线实时值,
              Z轴编码器实时值 := "数据发送".Z轴编码实时值_5,
              Z轴待命位置编码值 := "数据接收".Z轴待命值,
              机械手手自动标志 := "数据接收".手自动状态_5,
              Z轴高速转低速编码值 := "数据接收".Z轴高速转低速脉冲_5,
              X轴提前运行编码值 := "数据接收".X轴提前回待命脉冲值,
              机械手单独复位 := "5#机械手单独复位标志位",
              输送线变频器报警 := "输送线变频器报警",
              Z轴减速距离 := "数据接收".Z轴待命值,
              测试模式 := "数据接收".测试模式,
              设备压力开关 := "14P01",
              上位机状态 := "数据接收".PC状态,
              "B#库满转" := "数据接收".库位满_10,
              "A#库满转" := "数据接收".库位满_9,
              取砖X轴提前下降设定值 := "Z轴速度".X轴是否走曲线,
              W轴伺服同步线速度值 := "Tag_129",
              输送线启动 := "%Q1.4",
              A库位启动按钮指示灯 => "14HL38",
              B库位启动按钮指示灯 => "14HL39",
              吸盘电磁阀打开 => "14KAV12",
              吸盘电磁阀关闭 => "14KAV11",
              x轴2库正转 => "14M13LI1",
              x轴1库反转 => "14M13LI2",
              x轴低速 => "14M13LI3",
              x轴抱闸 => "%Q14.6",
              z轴下降 => "14M14FWD",
              z轴上升 => "14M14REV",
              z轴抱闸 => "%Q14.2",
              z轴1速 => "14M14X1",
              z轴2速 => "14M14X2",
              z轴3速 => "14M14X3",
              "W轴伺服启动/停止" => "Q12.0",
              给上位机取砖成功寄存地址 => "数据发送".取砖动作完成_5,
              AB库给上位机发送放砖完成指令 => "数据发送".放砖动作完成_5,
              AB库放砖回原位完成给上位机发送完成指令 => "数据发送".机械手就绪_5,
              放砖模式机械手放砖等待 => "数据发送".放砖确认等待_5,
              系统运行标志 => "5#机械手系统运行标志",
              系统复位标志 => "5#机械手系统复位标志",
              系统急停限位标志 => "5#机械手系统急停限位标志",
              压力开关压力检测报警1 => "5#1压力开关报警",
              压力开关压力检测报警2 => "5#2压力开关报警",
              压力开关压力检测报警3 => "5#3压力开关报警",
              压力开关压力检测报警4 => "5#4压力开关报警",
              A库位安全光电报警 => "9#库安全光电报警",
              B库位安全光电报警 => "10#库安全光电报警",
              A库位安全光电报警toPC => "数据发送".库位安全报警_9,
              B库位安全光电报警toPC => "数据发送".库位安全报警_10,
              下砖周期标志位 => "Tag_53",
              上砖周转标志位 => "Tag_54",
              找待命位标志位 => "5#找待命位速度");
END_REGION
END_FUNCTION

// folder: 通讯

FUNCTION "PLC <=> PC" : Void   // FC16, LAD
{ S7_Optimized_Access := 'TRUE' }
VERSION : 0.1
   VAR_TEMP   // added for the SCL form of the ladder/FBD networks
      _w1 : Bool;
      _w2 : Bool;
      _w3 : Bool;
      _w4 : Bool;
      _w5 : Bool;
      _w6 : Bool;
      _w7 : Bool;
      _w8 : Bool;
   END_VAR
BEGIN

REGION Network 1: PLC TO PC 系统状态
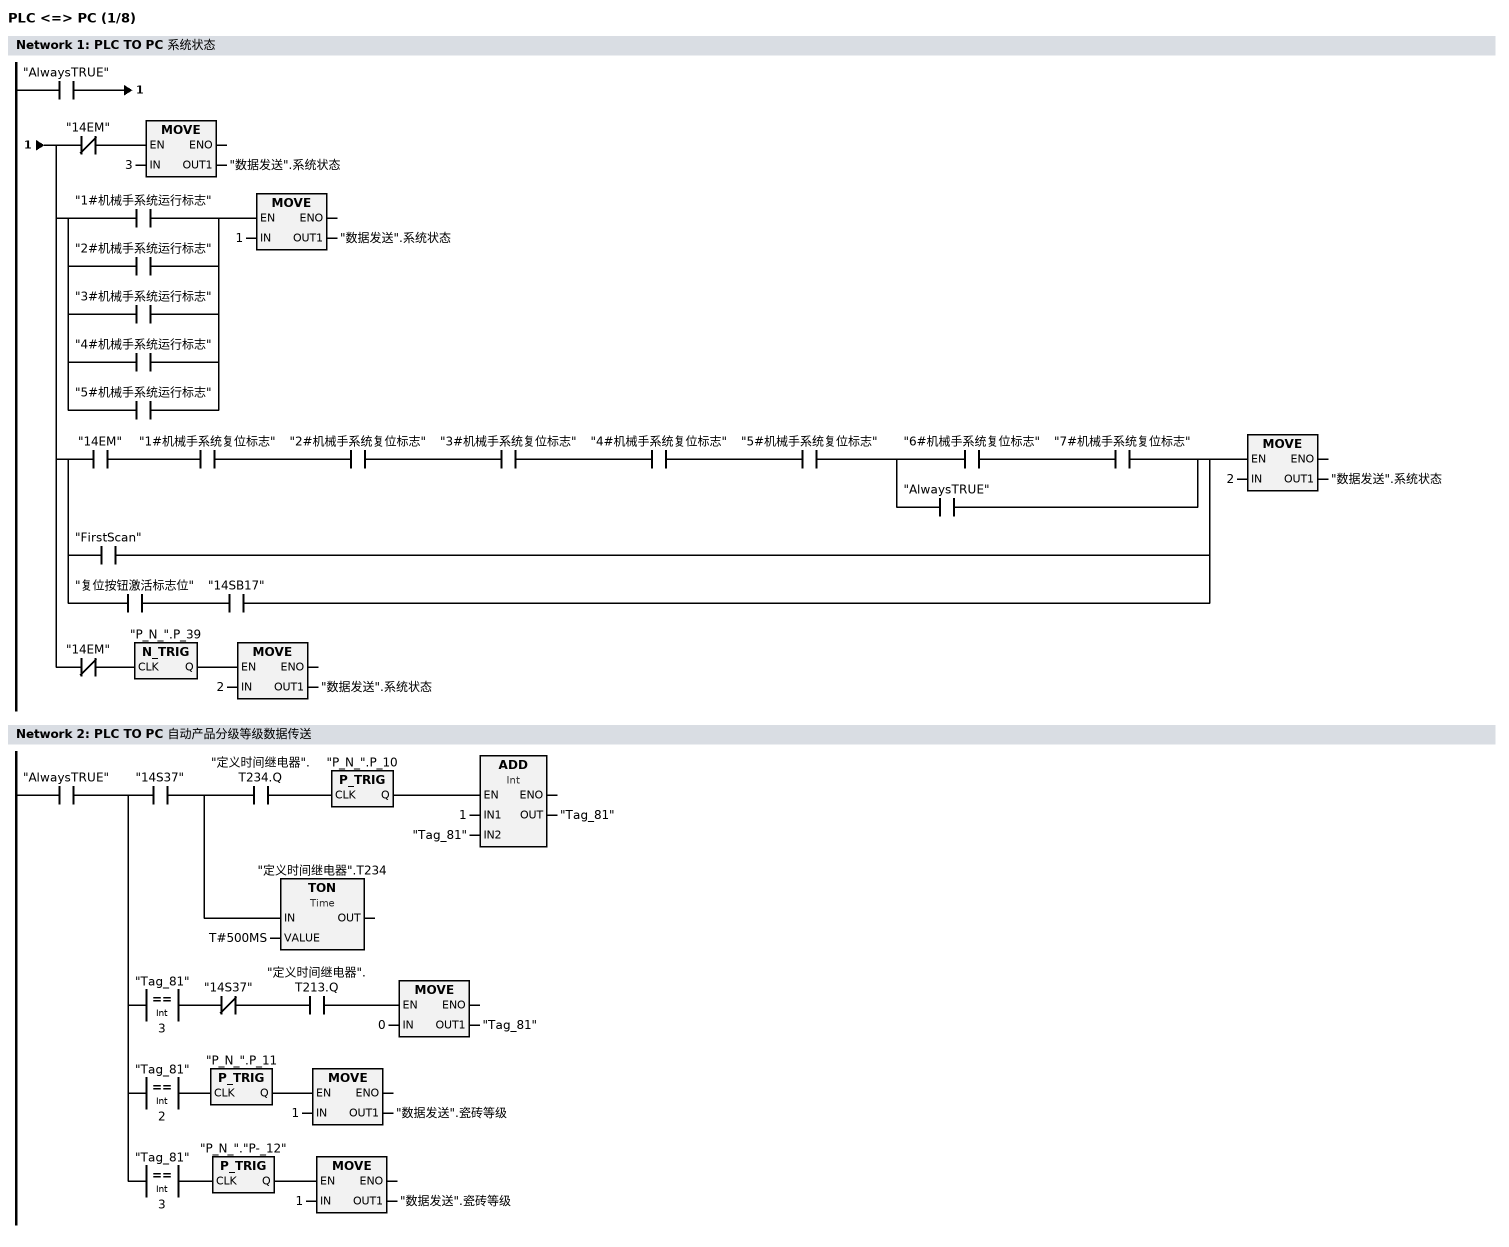
   RUNG wire#powerrail
      Contact( "AlwaysTRUE" )
      wire#w1
      I_Contact( "14EM" )
      Move(in := 3, out1 => "数据发送".系统状态)
   END_RUNG
   RUNG wire#w1
      Contact( "1#机械手系统运行标志" )
      wire#w2
      Move(in := 1, out1 => "数据发送".系统状态)
   END_RUNG
   RUNG wire#w1
      Contact( "2#机械手系统运行标志" )
   END_RUNG wire#w2
   RUNG wire#w1
      Contact( "3#机械手系统运行标志" )
   END_RUNG wire#w2
   RUNG wire#w1
      Contact( "4#机械手系统运行标志" )
   END_RUNG wire#w2
   RUNG wire#w1
      Contact( "5#机械手系统运行标志" )
   END_RUNG wire#w2
   RUNG wire#w1
      Contact( "14EM" )
      Contact( "1#机械手系统复位标志" )
      Contact( "2#机械手系统复位标志" )
      Contact( "3#机械手系统复位标志" )
      Contact( "4#机械手系统复位标志" )
      Contact( "5#机械手系统复位标志" )
      wire#w3
      Contact( "6#机械手系统复位标志" )
      Contact( "7#机械手系统复位标志" )
      wire#w4
      Move(in := 2, out1 => "数据发送".系统状态)
   END_RUNG
   RUNG wire#w3
      Contact( "AlwaysTRUE" )
   END_RUNG wire#w4
   RUNG wire#w1
      Contact( "FirstScan" )
   END_RUNG wire#w4
   RUNG wire#w1
      Contact( "复位按钮激活标志位" )
      Contact( "14SB17" )
   END_RUNG wire#w4
   RUNG wire#w1
      I_Contact( "14EM" )
      N_Trig( "P_N_".P_39 )
      Move(in := 2, out1 => "数据发送".系统状态)
   END_RUNG
   // the same network as SCL:
   IF "AlwaysTRUE" AND NOT "14EM" THEN "数据发送".系统状态 := 3; END_IF;
   IF "AlwaysTRUE" AND ("1#机械手系统运行标志" OR "2#机械手系统运行标志" OR "3#机械手系统运行标志" OR "4#机械手系统运行标志" OR "5#机械手系统运行标志") THEN
       "数据发送".系统状态 := 1;
   END_IF;
   IF "AlwaysTRUE" AND (("14EM" AND "1#机械手系统复位标志" AND "2#机械手系统复位标志" AND "3#机械手系统复位标志" AND "4#机械手系统复位标志" AND "5#机械手系统复位标志" AND (("6#机械手系统复位标志" AND "7#机械手系统复位标志") OR "AlwaysTRUE")) OR "FirstScan" OR ("复位按钮激活标志位" AND "14SB17")) THEN
       "数据发送".系统状态 := 2;
   END_IF;
   #_w1 := "AlwaysTRUE" AND NOT "14EM";
   #_w2 := NOT #_w1 AND "P_N_".P_39;   // falling edge
   "P_N_".P_39 := #_w1;
   IF #_w2 THEN "数据发送".系统状态 := 2; END_IF;
END_REGION

REGION Network 2: PLC TO PC 自动产品分级等级数据传送
   #_w1 := "AlwaysTRUE" AND "14S37";
   #_w2 := #_w1 AND "定义时间继电器".T234.Q;
   #_w3 := #_w2 AND NOT "P_N_".P_10;   // rising edge
   "P_N_".P_10 := #_w2;
   IF #_w3 THEN "Tag_81" := 1 + "Tag_81"; END_IF;
   "定义时间继电器".T234.TON(IN := #_w1, PT := T#500MS);   // TON coil
   IF "AlwaysTRUE" AND ("Tag_81" = 3) AND NOT "14S37" AND "定义时间继电器".T213.Q THEN "Tag_81" := 0; END_IF;
   #_w4 := "AlwaysTRUE" AND ("Tag_81" = 2);
   #_w5 := #_w4 AND NOT "P_N_".P_11;   // rising edge
   "P_N_".P_11 := #_w4;
   IF #_w5 THEN "数据发送".瓷砖等级 := 1; END_IF;
   #_w6 := "AlwaysTRUE" AND ("Tag_81" = 3);
   #_w7 := #_w6 AND NOT "P_N_"."P-_12";   // rising edge
   "P_N_"."P-_12" := #_w6;
   IF #_w7 THEN "数据发送".瓷砖等级 := 1; END_IF;
END_REGION

REGION Network 3: PLC TO PC 按钮产品分级等级数据传送
